REGION Network 22: J_Button_1
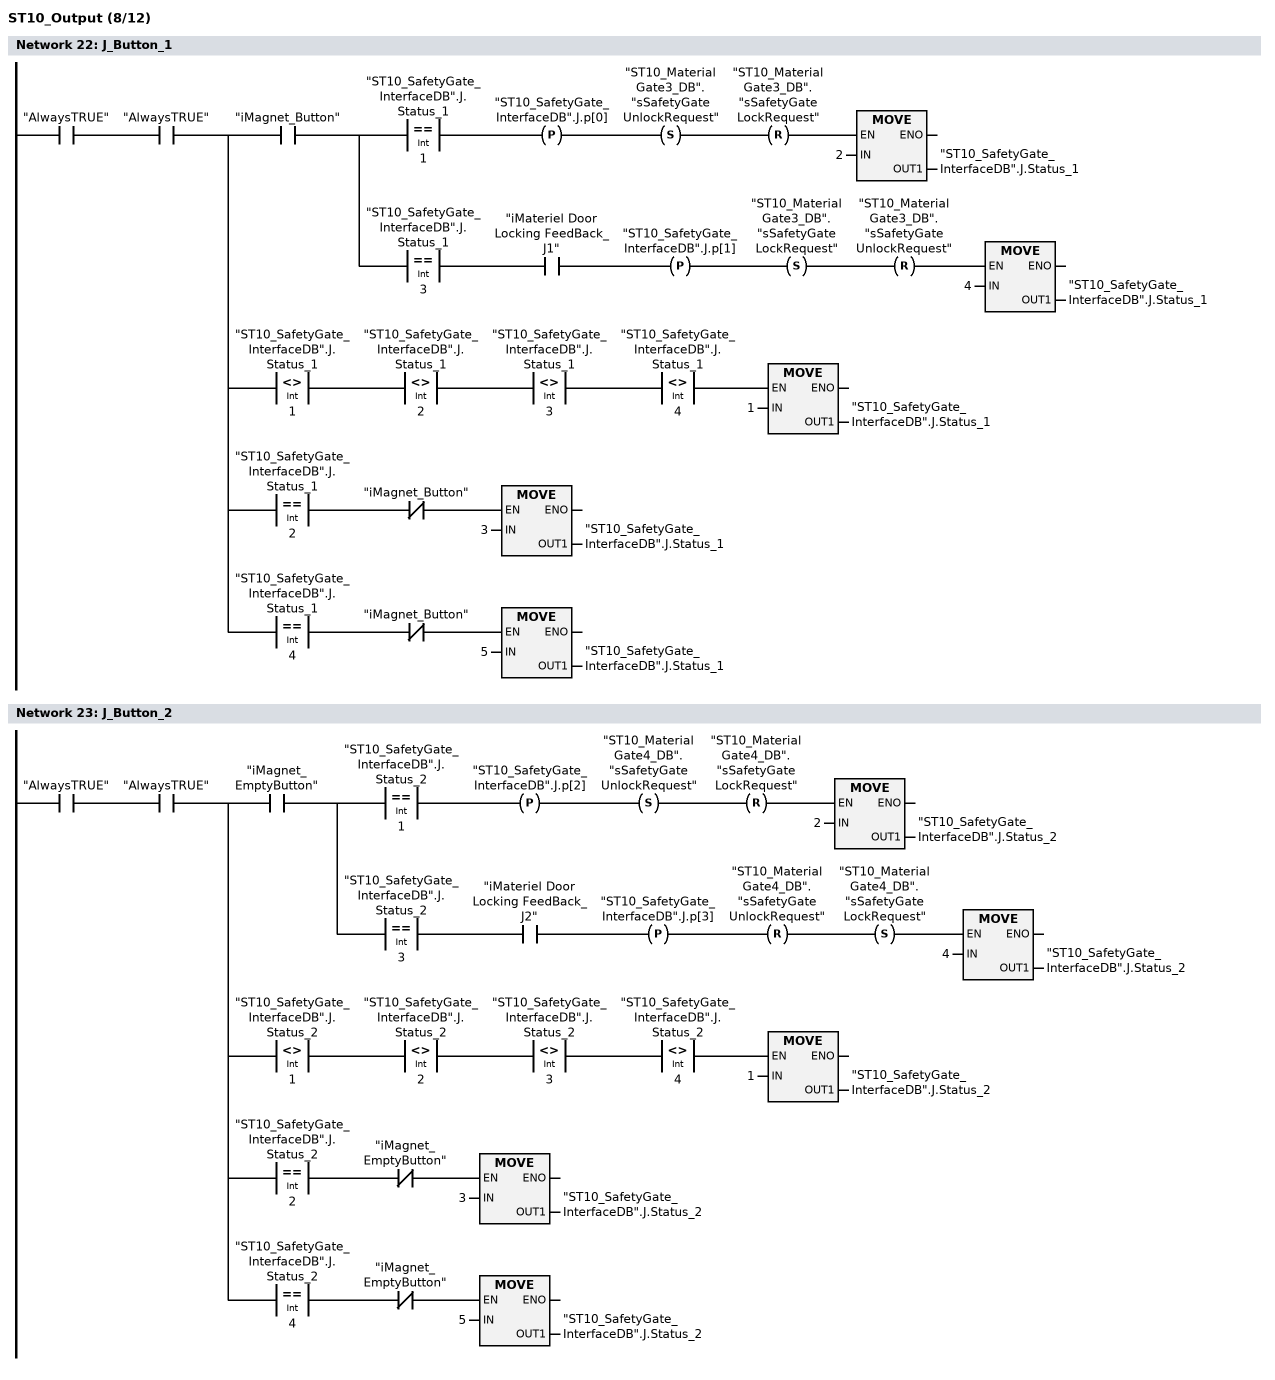
   RUNG wire#powerrail
      Contact( "AlwaysTRUE" )
      Contact( "AlwaysTRUE" )
      wire#w1
      Contact( "iMagnet_Button" )
      wire#w2
      { S7_Templates := "SrcType := Int" } EQ_Contact(in1 := "ST10_SafetyGate_InterfaceDB".J.Status_1, in2 := 1)
      P_Trig( "ST10_SafetyGate_InterfaceDB".J.p[0] )
      S_Coil( "ST10_MaterialGate3_DB"."sSafetyGate UnlockRequest" )
      R_Coil( "ST10_MaterialGate3_DB"."sSafetyGate LockRequest" )
      Move(in := 2, out1 => "ST10_SafetyGate_InterfaceDB".J.Status_1)
   END_RUNG
   RUNG wire#w2
      { S7_Templates := "SrcType := Int" } EQ_Contact(in1 := "ST10_SafetyGate_InterfaceDB".J.Status_1, in2 := 3)
      Contact( "iMateriel Door Locking FeedBack_J1" )
      P_Trig( "ST10_SafetyGate_InterfaceDB".J.p[1] )
      S_Coil( "ST10_MaterialGate3_DB"."sSafetyGate LockRequest" )
      R_Coil( "ST10_MaterialGate3_DB"."sSafetyGate UnlockRequest" )
      Move(in := 4, out1 => "ST10_SafetyGate_InterfaceDB".J.Status_1)
   END_RUNG
   RUNG wire#w1
      { S7_Templates := "SrcType := Int" } NE_Contact(in1 := "ST10_SafetyGate_InterfaceDB".J.Status_1, in2 := 1)
      { S7_Templates := "SrcType := Int" } NE_Contact(in1 := "ST10_SafetyGate_InterfaceDB".J.Status_1, in2 := 2)
      { S7_Templates := "SrcType := Int" } NE_Contact(in1 := "ST10_SafetyGate_InterfaceDB".J.Status_1, in2 := 3)
      { S7_Templates := "SrcType := Int" } NE_Contact(in1 := "ST10_SafetyGate_InterfaceDB".J.Status_1, in2 := 4)
      Move(in := 1, out1 => "ST10_SafetyGate_InterfaceDB".J.Status_1)
   END_RUNG
   RUNG wire#w1
      { S7_Templates := "SrcType := Int" } EQ_Contact(in1 := "ST10_SafetyGate_InterfaceDB".J.Status_1, in2 := 2)
      I_Contact( "iMagnet_Button" )
      Move(in := 3, out1 => "ST10_SafetyGate_InterfaceDB".J.Status_1)
   END_RUNG
   RUNG wire#w1
      { S7_Templates := "SrcType := Int" } EQ_Contact(in1 := "ST10_SafetyGate_InterfaceDB".J.Status_1, in2 := 4)
      I_Contact( "iMagnet_Button" )
      Move(in := 5, out1 => "ST10_SafetyGate_InterfaceDB".J.Status_1)
   END_RUNG
   // the same network as SCL:
   #_w1 := "AlwaysTRUE" AND "AlwaysTRUE";
   #_w2 := #_w1 AND "iMagnet_Button";
   #_w3 := #_w2 AND ("ST10_SafetyGate_InterfaceDB".J.Status_1 = 1);
   #_w4 := #_w3 AND NOT "ST10_SafetyGate_InterfaceDB".J.p[0];   // rising edge
   "ST10_SafetyGate_InterfaceDB".J.p[0] := #_w3;
   IF #_w4 THEN
       "ST10_MaterialGate3_DB"."sSafetyGate UnlockRequest" := TRUE;
       "ST10_MaterialGate3_DB"."sSafetyGate LockRequest" := FALSE;
       "ST10_SafetyGate_InterfaceDB".J.Status_1 := 2;
   END_IF;
   #_w5 := #_w2 AND ("ST10_SafetyGate_InterfaceDB".J.Status_1 = 3) AND "iMateriel Door Locking FeedBack_J1";
   #_w6 := #_w5 AND NOT "ST10_SafetyGate_InterfaceDB".J.p[1];   // rising edge
   "ST10_SafetyGate_InterfaceDB".J.p[1] := #_w5;
   IF #_w6 THEN
       "ST10_MaterialGate3_DB"."sSafetyGate LockRequest" := TRUE;
       "ST10_MaterialGate3_DB"."sSafetyGate UnlockRequest" := FALSE;
       "ST10_SafetyGate_InterfaceDB".J.Status_1 := 4;
   END_IF;
   IF #_w1 AND ("ST10_SafetyGate_InterfaceDB".J.Status_1 <> 1) AND ("ST10_SafetyGate_InterfaceDB".J.Status_1 <> 2) AND ("ST10_SafetyGate_InterfaceDB".J.Status_1 <> 3) AND ("ST10_SafetyGate_InterfaceDB".J.Status_1 <> 4) THEN
       "ST10_SafetyGate_InterfaceDB".J.Status_1 := 1;
   END_IF;
   IF #_w1 AND ("ST10_SafetyGate_InterfaceDB".J.Status_1 = 2) AND NOT "iMagnet_Button" THEN
       "ST10_SafetyGate_InterfaceDB".J.Status_1 := 3;
   END_IF;
   IF #_w1 AND ("ST10_SafetyGate_InterfaceDB".J.Status_1 = 4) AND NOT "iMagnet_Button" THEN
       "ST10_SafetyGate_InterfaceDB".J.Status_1 := 5;
   END_IF;
END_REGION

REGION Network 23: J_Button_2
   RUNG wire#powerrail
      Contact( "AlwaysTRUE" )
      Contact( "AlwaysTRUE" )
      wire#w1
      Contact( "iMagnet_EmptyButton" )
      wire#w2
      { S7_Templates := "SrcType := Int" } EQ_Contact(in1 := "ST10_SafetyGate_InterfaceDB".J.Status_2, in2 := 1)
      P_Trig( "ST10_SafetyGate_InterfaceDB".J.p[2] )
      S_Coil( "ST10_MaterialGate4_DB"."sSafetyGate UnlockRequest" )
      R_Coil( "ST10_MaterialGate4_DB"."sSafetyGate LockRequest" )
      Move(in := 2, out1 => "ST10_SafetyGate_InterfaceDB".J.Status_2)
   END_RUNG
   RUNG wire#w2
      { S7_Templates := "SrcType := Int" } EQ_Contact(in1 := "ST10_SafetyGate_InterfaceDB".J.Status_2, in2 := 3)
      Contact( "iMateriel Door Locking FeedBack_J2" )
      P_Trig( "ST10_SafetyGate_InterfaceDB".J.p[3] )
      R_Coil( "ST10_MaterialGate4_DB"."sSafetyGate UnlockRequest" )
      S_Coil( "ST10_MaterialGate4_DB"."sSafetyGate LockRequest" )
      Move(in := 4, out1 => "ST10_SafetyGate_InterfaceDB".J.Status_2)
   END_RUNG
   RUNG wire#w1
      { S7_Templates := "SrcType := Int" } NE_Contact(in1 := "ST10_SafetyGate_InterfaceDB".J.Status_2, in2 := 1)
      { S7_Templates := "SrcType := Int" } NE_Contact(in1 := "ST10_SafetyGate_InterfaceDB".J.Status_2, in2 := 2)
      { S7_Templates := "SrcType := Int" } NE_Contact(in1 := "ST10_SafetyGate_InterfaceDB".J.Status_2, in2 := 3)
      { S7_Templates := "SrcType := Int" } NE_Contact(in1 := "ST10_SafetyGate_InterfaceDB".J.Status_2, in2 := 4)
      Move(in := 1, out1 => "ST10_SafetyGate_InterfaceDB".J.Status_2)
   END_RUNG
   RUNG wire#w1
      { S7_Templates := "SrcType := Int" } EQ_Contact(in1 := "ST10_SafetyGate_InterfaceDB".J.Status_2, in2 := 2)
      I_Contact( "iMagnet_EmptyButton" )
      Move(in := 3, out1 => "ST10_SafetyGate_InterfaceDB".J.Status_2)
   END_RUNG
   RUNG wire#w1
      { S7_Templates := "SrcType := Int" } EQ_Contact(in1 := "ST10_SafetyGate_InterfaceDB".J.Status_2, in2 := 4)
      I_Contact( "iMagnet_EmptyButton" )
      Move(in := 5, out1 => "ST10_SafetyGate_InterfaceDB".J.Status_2)
   END_RUNG
   // the same network as SCL:
   #_w1 := "AlwaysTRUE" AND "AlwaysTRUE";
   #_w2 := #_w1 AND "iMagnet_EmptyButton";
   #_w3 := #_w2 AND ("ST10_SafetyGate_InterfaceDB".J.Status_2 = 1);
   #_w4 := #_w3 AND NOT "ST10_SafetyGate_InterfaceDB".J.p[2];   // rising edge
   "ST10_SafetyGate_InterfaceDB".J.p[2] := #_w3;
   IF #_w4 THEN
       "ST10_MaterialGate4_DB"."sSafetyGate UnlockRequest" := TRUE;
       "ST10_MaterialGate4_DB"."sSafetyGate LockRequest" := FALSE;
       "ST10_SafetyGate_InterfaceDB".J.Status_2 := 2;
   END_IF;
   #_w5 := #_w2 AND ("ST10_SafetyGate_InterfaceDB".J.Status_2 = 3) AND "iMateriel Door Locking FeedBack_J2";
   #_w6 := #_w5 AND NOT "ST10_SafetyGate_InterfaceDB".J.p[3];   // rising edge
   "ST10_SafetyGate_InterfaceDB".J.p[3] := #_w5;
   IF #_w6 THEN
       "ST10_MaterialGate4_DB"."sSafetyGate UnlockRequest" := FALSE;
       "ST10_MaterialGate4_DB"."sSafetyGate LockRequest" := TRUE;
       "ST10_SafetyGate_InterfaceDB".J.Status_2 := 4;
   END_IF;
   IF #_w1 AND ("ST10_SafetyGate_InterfaceDB".J.Status_2 <> 1) AND ("ST10_SafetyGate_InterfaceDB".J.Status_2 <> 2) AND ("ST10_SafetyGate_InterfaceDB".J.Status_2 <> 3) AND ("ST10_SafetyGate_InterfaceDB".J.Status_2 <> 4) THEN
       "ST10_SafetyGate_InterfaceDB".J.Status_2 := 1;
   END_IF;
   IF #_w1 AND ("ST10_SafetyGate_InterfaceDB".J.Status_2 = 2) AND NOT "iMagnet_EmptyButton" THEN
       "ST10_SafetyGate_InterfaceDB".J.Status_2 := 3;
   END_IF;
   IF #_w1 AND ("ST10_SafetyGate_InterfaceDB".J.Status_2 = 4) AND NOT "iMagnet_EmptyButton" THEN
       "ST10_SafetyGate_InterfaceDB".J.Status_2 := 5;
   END_IF;
END_REGION

REGION Network 24: J_Button_3 DOOR7
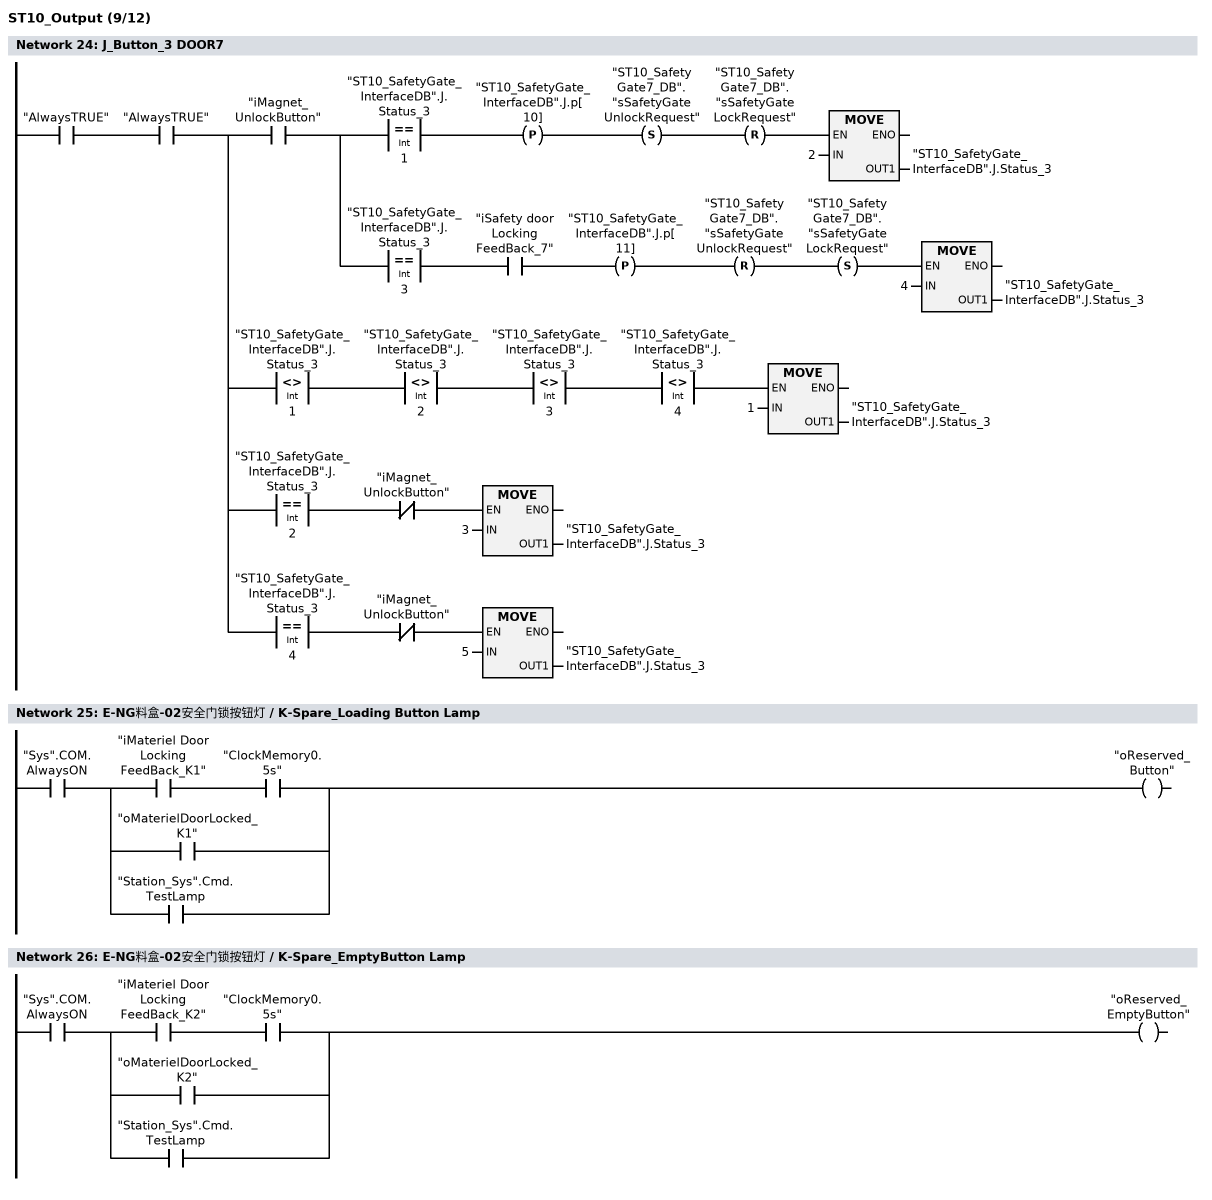
   RUNG wire#powerrail
      Contact( "AlwaysTRUE" )
      Contact( "AlwaysTRUE" )
      wire#w1
      Contact( "iMagnet_UnlockButton" )
      wire#w2
      { S7_Templates := "SrcType := Int" } EQ_Contact(in1 := "ST10_SafetyGate_InterfaceDB".J.Status_3, in2 := 1)
      P_Trig( "ST10_SafetyGate_InterfaceDB".J.p[10] )
      S_Coil( "ST10_SafetyGate7_DB"."sSafetyGate UnlockRequest" )
      R_Coil( "ST10_SafetyGate7_DB"."sSafetyGate LockRequest" )
      Move(in := 2, out1 => "ST10_SafetyGate_InterfaceDB".J.Status_3)
   END_RUNG
   RUNG wire#w2
      { S7_Templates := "SrcType := Int" } EQ_Contact(in1 := "ST10_SafetyGate_InterfaceDB".J.Status_3, in2 := 3)
      Contact( "iSafety door Locking FeedBack_7" )
      P_Trig( "ST10_SafetyGate_InterfaceDB".J.p[11] )
      R_Coil( "ST10_SafetyGate7_DB"."sSafetyGate UnlockRequest" )
      S_Coil( "ST10_SafetyGate7_DB"."sSafetyGate LockRequest" )
      Move(in := 4, out1 => "ST10_SafetyGate_InterfaceDB".J.Status_3)
   END_RUNG
   RUNG wire#w1
      { S7_Templates := "SrcType := Int" } NE_Contact(in1 := "ST10_SafetyGate_InterfaceDB".J.Status_3, in2 := 1)
      { S7_Templates := "SrcType := Int" } NE_Contact(in1 := "ST10_SafetyGate_InterfaceDB".J.Status_3, in2 := 2)
      { S7_Templates := "SrcType := Int" } NE_Contact(in1 := "ST10_SafetyGate_InterfaceDB".J.Status_3, in2 := 3)
      { S7_Templates := "SrcType := Int" } NE_Contact(in1 := "ST10_SafetyGate_InterfaceDB".J.Status_3, in2 := 4)
      Move(in := 1, out1 => "ST10_SafetyGate_InterfaceDB".J.Status_3)
   END_RUNG
   RUNG wire#w1
      { S7_Templates := "SrcType := Int" } EQ_Contact(in1 := "ST10_SafetyGate_InterfaceDB".J.Status_3, in2 := 2)
      I_Contact( "iMagnet_UnlockButton" )
      Move(in := 3, out1 => "ST10_SafetyGate_InterfaceDB".J.Status_3)
   END_RUNG
   RUNG wire#w1
      { S7_Templates := "SrcType := Int" } EQ_Contact(in1 := "ST10_SafetyGate_InterfaceDB".J.Status_3, in2 := 4)
      I_Contact( "iMagnet_UnlockButton" )
      Move(in := 5, out1 => "ST10_SafetyGate_InterfaceDB".J.Status_3)
   END_RUNG
   // the same network as SCL:
   #_w1 := "AlwaysTRUE" AND "AlwaysTRUE";
   #_w2 := #_w1 AND "iMagnet_UnlockButton";
   #_w3 := #_w2 AND ("ST10_SafetyGate_InterfaceDB".J.Status_3 = 1);
   #_w4 := #_w3 AND NOT "ST10_SafetyGate_InterfaceDB".J.p[10];   // rising edge
   "ST10_SafetyGate_InterfaceDB".J.p[10] := #_w3;
   IF #_w4 THEN
       "ST10_SafetyGate7_DB"."sSafetyGate UnlockRequest" := TRUE;
       "ST10_SafetyGate7_DB"."sSafetyGate LockRequest" := FALSE;
       "ST10_SafetyGate_InterfaceDB".J.Status_3 := 2;
   END_IF;
   #_w5 := #_w2 AND ("ST10_SafetyGate_InterfaceDB".J.Status_3 = 3) AND "iSafety door Locking FeedBack_7";
   #_w6 := #_w5 AND NOT "ST10_SafetyGate_InterfaceDB".J.p[11];   // rising edge
   "ST10_SafetyGate_InterfaceDB".J.p[11] := #_w5;
   IF #_w6 THEN
       "ST10_SafetyGate7_DB"."sSafetyGate UnlockRequest" := FALSE;
       "ST10_SafetyGate7_DB"."sSafetyGate LockRequest" := TRUE;
       "ST10_SafetyGate_InterfaceDB".J.Status_3 := 4;
   END_IF;
   IF #_w1 AND ("ST10_SafetyGate_InterfaceDB".J.Status_3 <> 1) AND ("ST10_SafetyGate_InterfaceDB".J.Status_3 <> 2) AND ("ST10_SafetyGate_InterfaceDB".J.Status_3 <> 3) AND ("ST10_SafetyGate_InterfaceDB".J.Status_3 <> 4) THEN
       "ST10_SafetyGate_InterfaceDB".J.Status_3 := 1;
   END_IF;
   IF #_w1 AND ("ST10_SafetyGate_InterfaceDB".J.Status_3 = 2) AND NOT "iMagnet_UnlockButton" THEN
       "ST10_SafetyGate_InterfaceDB".J.Status_3 := 3;
   END_IF;
   IF #_w1 AND ("ST10_SafetyGate_InterfaceDB".J.Status_3 = 4) AND NOT "iMagnet_UnlockButton" THEN
       "ST10_SafetyGate_InterfaceDB".J.Status_3 := 5;
   END_IF;
END_REGION

REGION Network 25: E-NG料盒-02安全门锁按钮灯 / K-Spare_Loading Button Lamp
   RUNG wire#powerrail
      Contact( "Sys".COM.AlwaysON )
      wire#w1
      Contact( "iMateriel Door Locking FeedBack_K1" )
      Contact( "ClockMemory0.5s" )
      wire#w2
      Coil( "oReserved_Button" )
   END_RUNG
   RUNG wire#w1
      Contact( "oMaterielDoorLocked_K1" )
   END_RUNG wire#w2
   RUNG wire#w1
      Contact( "Station_Sys".Cmd.TestLamp )
   END_RUNG wire#w2
   // the same network as SCL:
   "oReserved_Button" := "Sys".COM.AlwaysON AND (("iMateriel Door Locking FeedBack_K1" AND "ClockMemory0.5s") OR "oMaterielDoorLocked_K1" OR "Station_Sys".Cmd.TestLamp);
END_REGION

REGION Network 26: E-NG料盒-02安全门锁按钮灯 / K-Spare_EmptyButton Lamp
   RUNG wire#powerrail
      Contact( "Sys".COM.AlwaysON )
      wire#w1
      Contact( "iMateriel Door Locking FeedBack_K2" )
      Contact( "ClockMemory0.5s" )
      wire#w2
      Coil( "oReserved_EmptyButton" )
   END_RUNG
   RUNG wire#w1
      Contact( "oMaterielDoorLocked_K2" )
   END_RUNG wire#w2
   RUNG wire#w1
      Contact( "Station_Sys".Cmd.TestLamp )
   END_RUNG wire#w2
   // the same network as SCL:
   "oReserved_EmptyButton" := "Sys".COM.AlwaysON AND (("iMateriel Door Locking FeedBack_K2" AND "ClockMemory0.5s") OR "oMaterielDoorLocked_K2" OR "Station_Sys".Cmd.TestLamp);
END_REGION

REGION Network 27: E-NG料盒-02安全门锁按钮灯 / K_Loading DoorButton Lamp 8
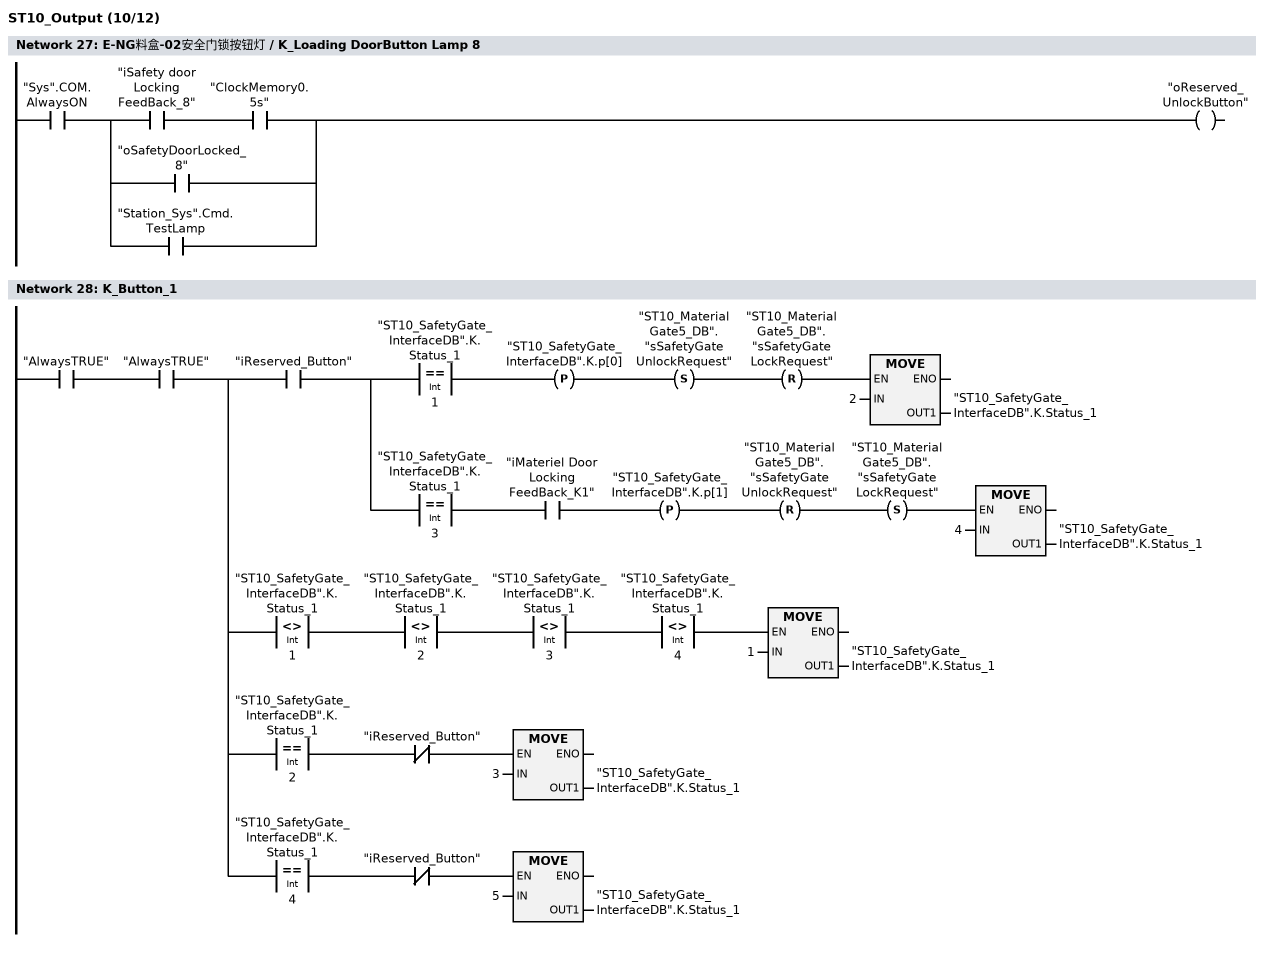
   RUNG wire#powerrail
      Contact( "Sys".COM.AlwaysON )
      wire#w1
      Contact( "iSafety door Locking FeedBack_8" )
      Contact( "ClockMemory0.5s" )
      wire#w2
      Coil( "oReserved_UnlockButton" )
   END_RUNG
   RUNG wire#w1
      Contact( "oSafetyDoorLocked_8" )
   END_RUNG wire#w2
   RUNG wire#w1
      Contact( "Station_Sys".Cmd.TestLamp )
   END_RUNG wire#w2
   // the same network as SCL:
   "oReserved_UnlockButton" := "Sys".COM.AlwaysON AND (("iSafety door Locking FeedBack_8" AND "ClockMemory0.5s") OR "oSafetyDoorLocked_8" OR "Station_Sys".Cmd.TestLamp);
END_REGION

REGION Network 28: K_Button_1
   RUNG wire#powerrail
      Contact( "AlwaysTRUE" )
      Contact( "AlwaysTRUE" )
      wire#w1
      Contact( "iReserved_Button" )
      wire#w2
      { S7_Templates := "SrcType := Int" } EQ_Contact(in1 := "ST10_SafetyGate_InterfaceDB".K.Status_1, in2 := 1)
      P_Trig( "ST10_SafetyGate_InterfaceDB".K.p[0] )
      S_Coil( "ST10_MaterialGate5_DB"."sSafetyGate UnlockRequest" )
      R_Coil( "ST10_MaterialGate5_DB"."sSafetyGate LockRequest" )
      Move(in := 2, out1 => "ST10_SafetyGate_InterfaceDB".K.Status_1)
   END_RUNG
   RUNG wire#w2
      { S7_Templates := "SrcType := Int" } EQ_Contact(in1 := "ST10_SafetyGate_InterfaceDB".K.Status_1, in2 := 3)
      Contact( "iMateriel Door Locking FeedBack_K1" )
      P_Trig( "ST10_SafetyGate_InterfaceDB".K.p[1] )
      R_Coil( "ST10_MaterialGate5_DB"."sSafetyGate UnlockRequest" )
      S_Coil( "ST10_MaterialGate5_DB"."sSafetyGate LockRequest" )
      Move(in := 4, out1 => "ST10_SafetyGate_InterfaceDB".K.Status_1)
   END_RUNG
   RUNG wire#w1
      { S7_Templates := "SrcType := Int" } NE_Contact(in1 := "ST10_SafetyGate_InterfaceDB".K.Status_1, in2 := 1)
      { S7_Templates := "SrcType := Int" } NE_Contact(in1 := "ST10_SafetyGate_InterfaceDB".K.Status_1, in2 := 2)
      { S7_Templates := "SrcType := Int" } NE_Contact(in1 := "ST10_SafetyGate_InterfaceDB".K.Status_1, in2 := 3)
      { S7_Templates := "SrcType := Int" } NE_Contact(in1 := "ST10_SafetyGate_InterfaceDB".K.Status_1, in2 := 4)
      Move(in := 1, out1 => "ST10_SafetyGate_InterfaceDB".K.Status_1)
   END_RUNG
   RUNG wire#w1
      { S7_Templates := "SrcType := Int" } EQ_Contact(in1 := "ST10_SafetyGate_InterfaceDB".K.Status_1, in2 := 2)
      I_Contact( "iReserved_Button" )
      Move(in := 3, out1 => "ST10_SafetyGate_InterfaceDB".K.Status_1)
   END_RUNG
   RUNG wire#w1
      { S7_Templates := "SrcType := Int" } EQ_Contact(in1 := "ST10_SafetyGate_InterfaceDB".K.Status_1, in2 := 4)
      I_Contact( "iReserved_Button" )
      Move(in := 5, out1 => "ST10_SafetyGate_InterfaceDB".K.Status_1)
   END_RUNG
   // the same network as SCL:
   #_w1 := "AlwaysTRUE" AND "AlwaysTRUE";
   #_w2 := #_w1 AND "iReserved_Button";
   #_w3 := #_w2 AND ("ST10_SafetyGate_InterfaceDB".K.Status_1 = 1);
   #_w4 := #_w3 AND NOT "ST10_SafetyGate_InterfaceDB".K.p[0];   // rising edge
   "ST10_SafetyGate_InterfaceDB".K.p[0] := #_w3;
   IF #_w4 THEN
       "ST10_MaterialGate5_DB"."sSafetyGate UnlockRequest" := TRUE;
       "ST10_MaterialGate5_DB"."sSafetyGate LockRequest" := FALSE;
       "ST10_SafetyGate_InterfaceDB".K.Status_1 := 2;
   END_IF;
   #_w5 := #_w2 AND ("ST10_SafetyGate_InterfaceDB".K.Status_1 = 3) AND "iMateriel Door Locking FeedBack_K1";
   #_w6 := #_w5 AND NOT "ST10_SafetyGate_InterfaceDB".K.p[1];   // rising edge
   "ST10_SafetyGate_InterfaceDB".K.p[1] := #_w5;
   IF #_w6 THEN
       "ST10_MaterialGate5_DB"."sSafetyGate UnlockRequest" := FALSE;
       "ST10_MaterialGate5_DB"."sSafetyGate LockRequest" := TRUE;
       "ST10_SafetyGate_InterfaceDB".K.Status_1 := 4;
   END_IF;
   IF #_w1 AND ("ST10_SafetyGate_InterfaceDB".K.Status_1 <> 1) AND ("ST10_SafetyGate_InterfaceDB".K.Status_1 <> 2) AND ("ST10_SafetyGate_InterfaceDB".K.Status_1 <> 3) AND ("ST10_SafetyGate_InterfaceDB".K.Status_1 <> 4) THEN
       "ST10_SafetyGate_InterfaceDB".K.Status_1 := 1;
   END_IF;
   IF #_w1 AND ("ST10_SafetyGate_InterfaceDB".K.Status_1 = 2) AND NOT "iReserved_Button" THEN
       "ST10_SafetyGate_InterfaceDB".K.Status_1 := 3;
   END_IF;
   IF #_w1 AND ("ST10_SafetyGate_InterfaceDB".K.Status_1 = 4) AND NOT "iReserved_Button" THEN
       "ST10_SafetyGate_InterfaceDB".K.Status_1 := 5;
   END_IF;
END_REGION

REGION Network 29: K_Button_2
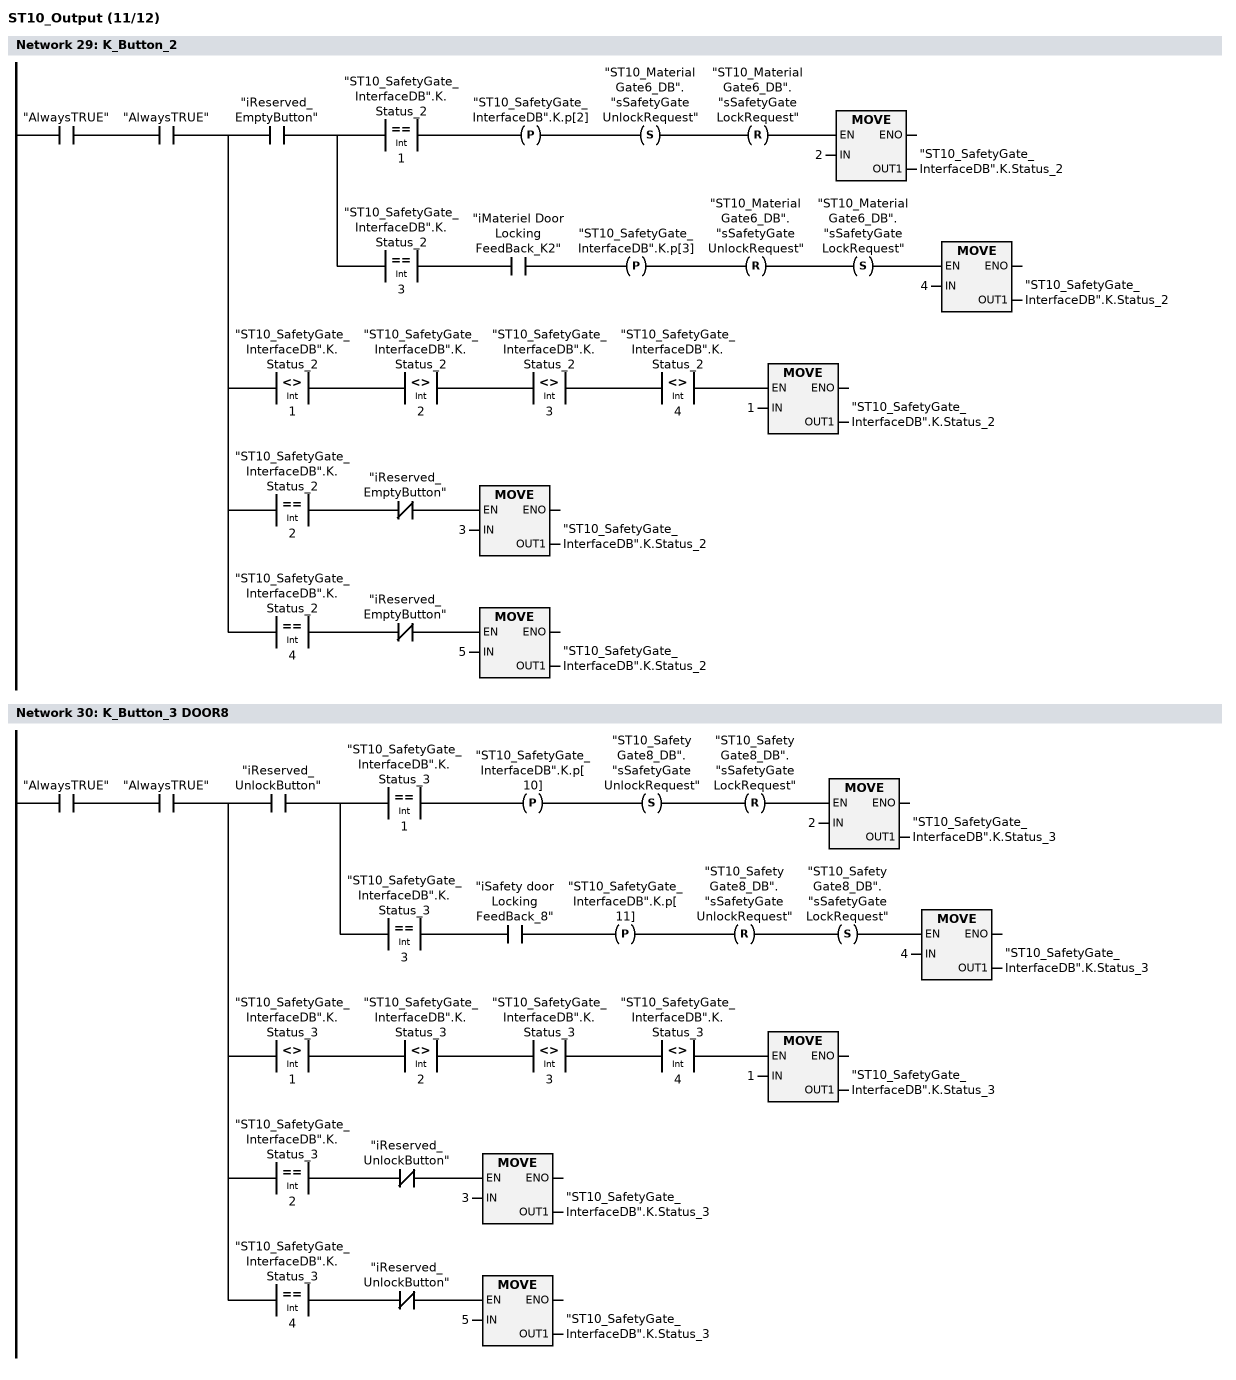
   RUNG wire#powerrail
      Contact( "AlwaysTRUE" )
      Contact( "AlwaysTRUE" )
      wire#w1
      Contact( "iReserved_EmptyButton" )
      wire#w2
      { S7_Templates := "SrcType := Int" } EQ_Contact(in1 := "ST10_SafetyGate_InterfaceDB".K.Status_2, in2 := 1)
      P_Trig( "ST10_SafetyGate_InterfaceDB".K.p[2] )
      S_Coil( "ST10_MaterialGate6_DB"."sSafetyGate UnlockRequest" )
      R_Coil( "ST10_MaterialGate6_DB"."sSafetyGate LockRequest" )
      Move(in := 2, out1 => "ST10_SafetyGate_InterfaceDB".K.Status_2)
   END_RUNG
   RUNG wire#w2
      { S7_Templates := "SrcType := Int" } EQ_Contact(in1 := "ST10_SafetyGate_InterfaceDB".K.Status_2, in2 := 3)
      Contact( "iMateriel Door Locking FeedBack_K2" )
      P_Trig( "ST10_SafetyGate_InterfaceDB".K.p[3] )
      R_Coil( "ST10_MaterialGate6_DB"."sSafetyGate UnlockRequest" )
      S_Coil( "ST10_MaterialGate6_DB"."sSafetyGate LockRequest" )
      Move(in := 4, out1 => "ST10_SafetyGate_InterfaceDB".K.Status_2)
   END_RUNG
   RUNG wire#w1
      { S7_Templates := "SrcType := Int" } NE_Contact(in1 := "ST10_SafetyGate_InterfaceDB".K.Status_2, in2 := 1)
      { S7_Templates := "SrcType := Int" } NE_Contact(in1 := "ST10_SafetyGate_InterfaceDB".K.Status_2, in2 := 2)
      { S7_Templates := "SrcType := Int" } NE_Contact(in1 := "ST10_SafetyGate_InterfaceDB".K.Status_2, in2 := 3)
      { S7_Templates := "SrcType := Int" } NE_Contact(in1 := "ST10_SafetyGate_InterfaceDB".K.Status_2, in2 := 4)
      Move(in := 1, out1 => "ST10_SafetyGate_InterfaceDB".K.Status_2)
   END_RUNG
   RUNG wire#w1
      { S7_Templates := "SrcType := Int" } EQ_Contact(in1 := "ST10_SafetyGate_InterfaceDB".K.Status_2, in2 := 2)
      I_Contact( "iReserved_EmptyButton" )
      Move(in := 3, out1 => "ST10_SafetyGate_InterfaceDB".K.Status_2)
   END_RUNG
   RUNG wire#w1
      { S7_Templates := "SrcType := Int" } EQ_Contact(in1 := "ST10_SafetyGate_InterfaceDB".K.Status_2, in2 := 4)
      I_Contact( "iReserved_EmptyButton" )
      Move(in := 5, out1 => "ST10_SafetyGate_InterfaceDB".K.Status_2)
   END_RUNG
   // the same network as SCL:
   #_w1 := "AlwaysTRUE" AND "AlwaysTRUE";
   #_w2 := #_w1 AND "iReserved_EmptyButton";
   #_w3 := #_w2 AND ("ST10_SafetyGate_InterfaceDB".K.Status_2 = 1);
   #_w4 := #_w3 AND NOT "ST10_SafetyGate_InterfaceDB".K.p[2];   // rising edge
   "ST10_SafetyGate_InterfaceDB".K.p[2] := #_w3;
   IF #_w4 THEN
       "ST10_MaterialGate6_DB"."sSafetyGate UnlockRequest" := TRUE;
       "ST10_MaterialGate6_DB"."sSafetyGate LockRequest" := FALSE;
       "ST10_SafetyGate_InterfaceDB".K.Status_2 := 2;
   END_IF;
   #_w5 := #_w2 AND ("ST10_SafetyGate_InterfaceDB".K.Status_2 = 3) AND "iMateriel Door Locking FeedBack_K2";
   #_w6 := #_w5 AND NOT "ST10_SafetyGate_InterfaceDB".K.p[3];   // rising edge
   "ST10_SafetyGate_InterfaceDB".K.p[3] := #_w5;
   IF #_w6 THEN
       "ST10_MaterialGate6_DB"."sSafetyGate UnlockRequest" := FALSE;
       "ST10_MaterialGate6_DB"."sSafetyGate LockRequest" := TRUE;
       "ST10_SafetyGate_InterfaceDB".K.Status_2 := 4;
   END_IF;
   IF #_w1 AND ("ST10_SafetyGate_InterfaceDB".K.Status_2 <> 1) AND ("ST10_SafetyGate_InterfaceDB".K.Status_2 <> 2) AND ("ST10_SafetyGate_InterfaceDB".K.Status_2 <> 3) AND ("ST10_SafetyGate_InterfaceDB".K.Status_2 <> 4) THEN
       "ST10_SafetyGate_InterfaceDB".K.Status_2 := 1;
   END_IF;
   IF #_w1 AND ("ST10_SafetyGate_InterfaceDB".K.Status_2 = 2) AND NOT "iReserved_EmptyButton" THEN
       "ST10_SafetyGate_InterfaceDB".K.Status_2 := 3;
   END_IF;
   IF #_w1 AND ("ST10_SafetyGate_InterfaceDB".K.Status_2 = 4) AND NOT "iReserved_EmptyButton" THEN
       "ST10_SafetyGate_InterfaceDB".K.Status_2 := 5;
   END_IF;
END_REGION

REGION Network 30: K_Button_3 DOOR8
   RUNG wire#powerrail
      Contact( "AlwaysTRUE" )
      Contact( "AlwaysTRUE" )
      wire#w1
      Contact( "iReserved_UnlockButton" )
      wire#w2
      { S7_Templates := "SrcType := Int" } EQ_Contact(in1 := "ST10_SafetyGate_InterfaceDB".K.Status_3, in2 := 1)
      P_Trig( "ST10_SafetyGate_InterfaceDB".K.p[10] )
      S_Coil( "ST10_SafetyGate8_DB"."sSafetyGate UnlockRequest" )
      R_Coil( "ST10_SafetyGate8_DB"."sSafetyGate LockRequest" )
      Move(in := 2, out1 => "ST10_SafetyGate_InterfaceDB".K.Status_3)
   END_RUNG
   RUNG wire#w2
      { S7_Templates := "SrcType := Int" } EQ_Contact(in1 := "ST10_SafetyGate_InterfaceDB".K.Status_3, in2 := 3)
      Contact( "iSafety door Locking FeedBack_8" )
      P_Trig( "ST10_SafetyGate_InterfaceDB".K.p[11] )
      R_Coil( "ST10_SafetyGate8_DB"."sSafetyGate UnlockRequest" )
      S_Coil( "ST10_SafetyGate8_DB"."sSafetyGate LockRequest" )
      Move(in := 4, out1 => "ST10_SafetyGate_InterfaceDB".K.Status_3)
   END_RUNG
   RUNG wire#w1
      { S7_Templates := "SrcType := Int" } NE_Contact(in1 := "ST10_SafetyGate_InterfaceDB".K.Status_3, in2 := 1)
      { S7_Templates := "SrcType := Int" } NE_Contact(in1 := "ST10_SafetyGate_InterfaceDB".K.Status_3, in2 := 2)
      { S7_Templates := "SrcType := Int" } NE_Contact(in1 := "ST10_SafetyGate_InterfaceDB".K.Status_3, in2 := 3)
      { S7_Templates := "SrcType := Int" } NE_Contact(in1 := "ST10_SafetyGate_InterfaceDB".K.Status_3, in2 := 4)
      Move(in := 1, out1 => "ST10_SafetyGate_InterfaceDB".K.Status_3)
   END_RUNG
   RUNG wire#w1
      { S7_Templates := "SrcType := Int" } EQ_Contact(in1 := "ST10_SafetyGate_InterfaceDB".K.Status_3, in2 := 2)
      I_Contact( "iReserved_UnlockButton" )
      Move(in := 3, out1 => "ST10_SafetyGate_InterfaceDB".K.Status_3)
   END_RUNG
   RUNG wire#w1
      { S7_Templates := "SrcType := Int" } EQ_Contact(in1 := "ST10_SafetyGate_InterfaceDB".K.Status_3, in2 := 4)
      I_Contact( "iReserved_UnlockButton" )
      Move(in := 5, out1 => "ST10_SafetyGate_InterfaceDB".K.Status_3)
   END_RUNG
   // the same network as SCL:
   #_w1 := "AlwaysTRUE" AND "AlwaysTRUE";
   #_w2 := #_w1 AND "iReserved_UnlockButton";
   #_w3 := #_w2 AND ("ST10_SafetyGate_InterfaceDB".K.Status_3 = 1);
   #_w4 := #_w3 AND NOT "ST10_SafetyGate_InterfaceDB".K.p[10];   // rising edge
   "ST10_SafetyGate_InterfaceDB".K.p[10] := #_w3;
   IF #_w4 THEN
       "ST10_SafetyGate8_DB"."sSafetyGate UnlockRequest" := TRUE;
       "ST10_SafetyGate8_DB"."sSafetyGate LockRequest" := FALSE;
       "ST10_SafetyGate_InterfaceDB".K.Status_3 := 2;
   END_IF;
   #_w5 := #_w2 AND ("ST10_SafetyGate_InterfaceDB".K.Status_3 = 3) AND "iSafety door Locking FeedBack_8";
   #_w6 := #_w5 AND NOT "ST10_SafetyGate_InterfaceDB".K.p[11];   // rising edge
   "ST10_SafetyGate_InterfaceDB".K.p[11] := #_w5;
   IF #_w6 THEN
       "ST10_SafetyGate8_DB"."sSafetyGate UnlockRequest" := FALSE;
       "ST10_SafetyGate8_DB"."sSafetyGate LockRequest" := TRUE;
       "ST10_SafetyGate_InterfaceDB".K.Status_3 := 4;
   END_IF;
   IF #_w1 AND ("ST10_SafetyGate_InterfaceDB".K.Status_3 <> 1) AND ("ST10_SafetyGate_InterfaceDB".K.Status_3 <> 2) AND ("ST10_SafetyGate_InterfaceDB".K.Status_3 <> 3) AND ("ST10_SafetyGate_InterfaceDB".K.Status_3 <> 4) THEN
       "ST10_SafetyGate_InterfaceDB".K.Status_3 := 1;
   END_IF;
   IF #_w1 AND ("ST10_SafetyGate_InterfaceDB".K.Status_3 = 2) AND NOT "iReserved_UnlockButton" THEN
       "ST10_SafetyGate_InterfaceDB".K.Status_3 := 3;
   END_IF;
   IF #_w1 AND ("ST10_SafetyGate_InterfaceDB".K.Status_3 = 4) AND NOT "iReserved_UnlockButton" THEN
       "ST10_SafetyGate_InterfaceDB".K.Status_3 := 5;
   END_IF;
END_REGION

REGION Network 31: E-NG料盒-02安全门锁按钮灯 / L-Unloading_LoadingButton Lamp
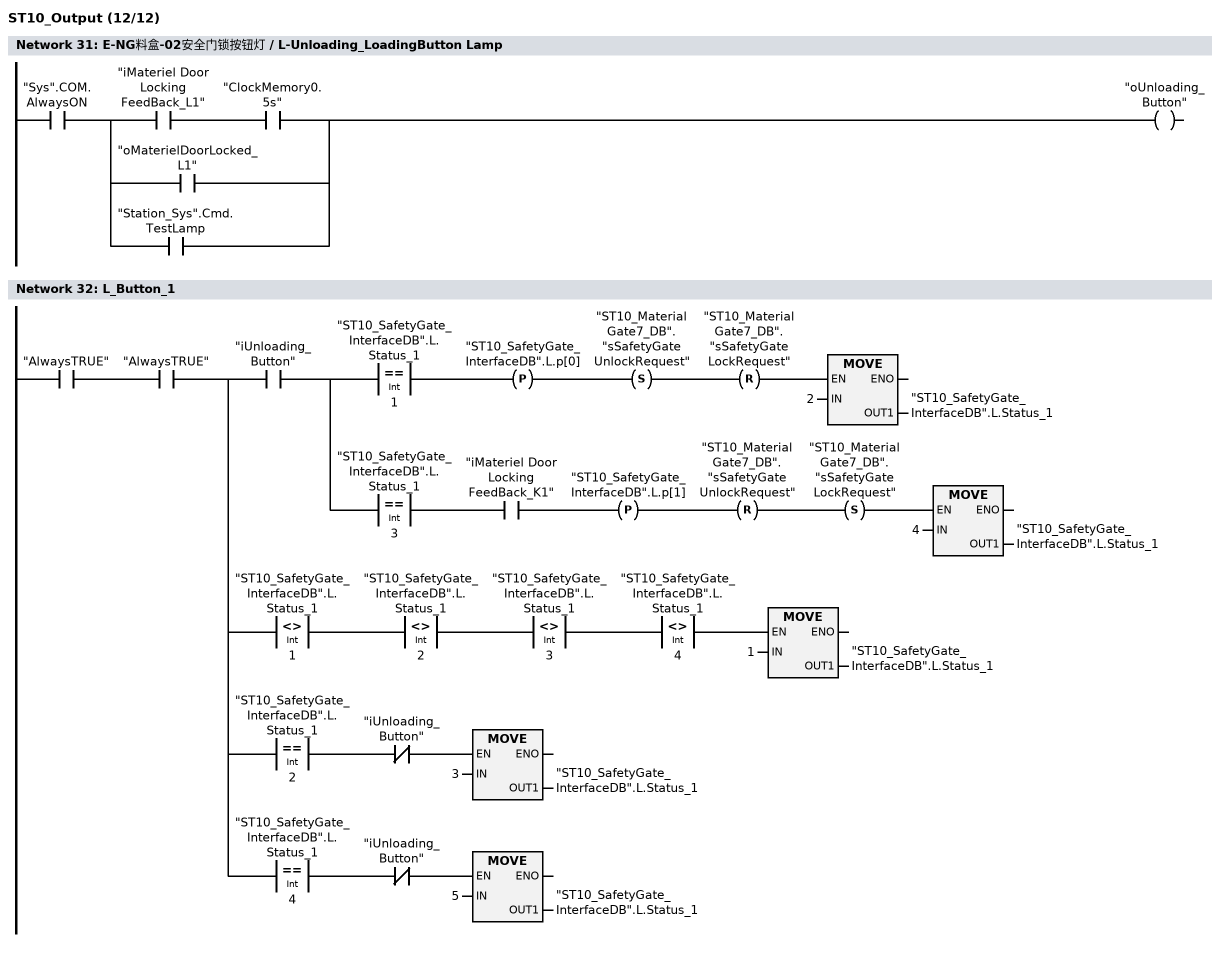
   RUNG wire#powerrail
      Contact( "Sys".COM.AlwaysON )
      wire#w1
      Contact( "iMateriel Door Locking FeedBack_L1" )
      Contact( "ClockMemory0.5s" )
      wire#w2
      Coil( "oUnloading_Button" )
   END_RUNG
   RUNG wire#w1
      Contact( "oMaterielDoorLocked_L1" )
   END_RUNG wire#w2
   RUNG wire#w1
      Contact( "Station_Sys".Cmd.TestLamp )
   END_RUNG wire#w2
   // the same network as SCL:
   "oUnloading_Button" := "Sys".COM.AlwaysON AND (("iMateriel Door Locking FeedBack_L1" AND "ClockMemory0.5s") OR "oMaterielDoorLocked_L1" OR "Station_Sys".Cmd.TestLamp);
END_REGION

REGION Network 32: L_Button_1
   RUNG wire#powerrail
      Contact( "AlwaysTRUE" )
      Contact( "AlwaysTRUE" )
      wire#w1
      Contact( "iUnloading_Button" )
      wire#w2
      { S7_Templates := "SrcType := Int" } EQ_Contact(in1 := "ST10_SafetyGate_InterfaceDB".L.Status_1, in2 := 1)
      P_Trig( "ST10_SafetyGate_InterfaceDB".L.p[0] )
      S_Coil( "ST10_MaterialGate7_DB"."sSafetyGate UnlockRequest" )
      R_Coil( "ST10_MaterialGate7_DB"."sSafetyGate LockRequest" )
      Move(in := 2, out1 => "ST10_SafetyGate_InterfaceDB".L.Status_1)
   END_RUNG
   RUNG wire#w2
      { S7_Templates := "SrcType := Int" } EQ_Contact(in1 := "ST10_SafetyGate_InterfaceDB".L.Status_1, in2 := 3)
      Contact( "iMateriel Door Locking FeedBack_K1" )
      P_Trig( "ST10_SafetyGate_InterfaceDB".L.p[1] )
      R_Coil( "ST10_MaterialGate7_DB"."sSafetyGate UnlockRequest" )
      S_Coil( "ST10_MaterialGate7_DB"."sSafetyGate LockRequest" )
      Move(in := 4, out1 => "ST10_SafetyGate_InterfaceDB".L.Status_1)
   END_RUNG
   RUNG wire#w1
      { S7_Templates := "SrcType := Int" } NE_Contact(in1 := "ST10_SafetyGate_InterfaceDB".L.Status_1, in2 := 1)
      { S7_Templates := "SrcType := Int" } NE_Contact(in1 := "ST10_SafetyGate_InterfaceDB".L.Status_1, in2 := 2)
      { S7_Templates := "SrcType := Int" } NE_Contact(in1 := "ST10_SafetyGate_InterfaceDB".L.Status_1, in2 := 3)
      { S7_Templates := "SrcType := Int" } NE_Contact(in1 := "ST10_SafetyGate_InterfaceDB".L.Status_1, in2 := 4)
      Move(in := 1, out1 => "ST10_SafetyGate_InterfaceDB".L.Status_1)
   END_RUNG
   RUNG wire#w1
      { S7_Templates := "SrcType := Int" } EQ_Contact(in1 := "ST10_SafetyGate_InterfaceDB".L.Status_1, in2 := 2)
      I_Contact( "iUnloading_Button" )
      Move(in := 3, out1 => "ST10_SafetyGate_InterfaceDB".L.Status_1)
   END_RUNG
   RUNG wire#w1
      { S7_Templates := "SrcType := Int" } EQ_Contact(in1 := "ST10_SafetyGate_InterfaceDB".L.Status_1, in2 := 4)
      I_Contact( "iUnloading_Button" )
      Move(in := 5, out1 => "ST10_SafetyGate_InterfaceDB".L.Status_1)
   END_RUNG
   // the same network as SCL:
   #_w1 := "AlwaysTRUE" AND "AlwaysTRUE";
   #_w2 := #_w1 AND "iUnloading_Button";
   #_w3 := #_w2 AND ("ST10_SafetyGate_InterfaceDB".L.Status_1 = 1);
   #_w4 := #_w3 AND NOT "ST10_SafetyGate_InterfaceDB".L.p[0];   // rising edge
   "ST10_SafetyGate_InterfaceDB".L.p[0] := #_w3;
   IF #_w4 THEN
       "ST10_MaterialGate7_DB"."sSafetyGate UnlockRequest" := TRUE;
       "ST10_MaterialGate7_DB"."sSafetyGate LockRequest" := FALSE;
       "ST10_SafetyGate_InterfaceDB".L.Status_1 := 2;
   END_IF;
   #_w5 := #_w2 AND ("ST10_SafetyGate_InterfaceDB".L.Status_1 = 3) AND "iMateriel Door Locking FeedBack_K1";
   #_w6 := #_w5 AND NOT "ST10_SafetyGate_InterfaceDB".L.p[1];   // rising edge
   "ST10_SafetyGate_InterfaceDB".L.p[1] := #_w5;
   IF #_w6 THEN
       "ST10_MaterialGate7_DB"."sSafetyGate UnlockRequest" := FALSE;
       "ST10_MaterialGate7_DB"."sSafetyGate LockRequest" := TRUE;
       "ST10_SafetyGate_InterfaceDB".L.Status_1 := 4;
   END_IF;
   IF #_w1 AND ("ST10_SafetyGate_InterfaceDB".L.Status_1 <> 1) AND ("ST10_SafetyGate_InterfaceDB".L.Status_1 <> 2) AND ("ST10_SafetyGate_InterfaceDB".L.Status_1 <> 3) AND ("ST10_SafetyGate_InterfaceDB".L.Status_1 <> 4) THEN
       "ST10_SafetyGate_InterfaceDB".L.Status_1 := 1;
   END_IF;
   IF #_w1 AND ("ST10_SafetyGate_InterfaceDB".L.Status_1 = 2) AND NOT "iUnloading_Button" THEN
       "ST10_SafetyGate_InterfaceDB".L.Status_1 := 3;
   END_IF;
   IF #_w1 AND ("ST10_SafetyGate_InterfaceDB".L.Status_1 = 4) AND NOT "iUnloading_Button" THEN
       "ST10_SafetyGate_InterfaceDB".L.Status_1 := 5;
   END_IF;
END_REGION

REGION Network 33: H
END_REGION
END_FUNCTION

FUNCTION_BLOCK "FB_Tower_4Lamp"   // FB5050, LAD
{ S7_Optimized_Access := 'TRUE' }
// stored: AutoNumber false, MemoryReserve 100, SetENOAutomatically false
   VAR_INPUT
      iReady : Bool;   // 系统OK
      iManual_Mode : Bool;
      iAuto_Mode : Bool;
      iAuto_Running : Bool;   // 自动运行信号
      iCheck_Mode : Bool;
      iIdle : Bool;   // 自动运行中空闲信号
      iWarning : Bool;
      iFault : Bool;
      "i0.5s_Pulse" : Bool;   // 0.5S脉冲
      i1s_Pulse : Bool;   // 1S脉冲
      i2s_Pulse : Bool;   // 2S脉冲
      iResetButton : Bool;   // 复位按钮
      "iE-StopButtonOK" : Bool;   // 急停按钮未按下
      iSafetyGateClosed : Bool;   // 安全门关闭信号
      iSafetyGateRelayOK : Bool;   // 安全门继电器输出OK
      iPowerOn : Bool;   // 系统上电信号
      iMachineHomePos : Bool;   // 所有设备在原始位
      iWorkAreaLightButton : Bool;   // HMI工作区域照明按钮
      iTest_Lamp : Bool;   // 灯测试按钮
   END_VAR
   VAR_OUTPUT
      oRed_Lamp : Bool;   // 塔灯-红色
      oYellow_Lamp : Bool;   // 塔灯-黄色
      oGreen_Lamp : Bool;   // 塔灯-绿色
      oBlue_Lamp : Bool;   // 塔灯-蓝色 1.蓝灯常亮表示设备在原位;2.蓝灯闪烁表示工位缺料等待上料
      oBuzzer : Bool;   // 塔灯-蜂鸣器
      oPowerOn : Bool;   // 系统上电指示灯
      oResetLamp : Bool;   // 复位按钮指示灯
      oWorkArea1_LightingOn : Bool;   // 工作区域1 照明打开
      oWorkArea2_LightingOn : Bool;   // 工作区域2 照明打开
      oWorkArea3_LightingOn : Bool;   // 工作区域3 照明打开
   END_VAR
   VAR_IN_OUT
      ioStationWaitingLoadPart : Bool;   // 工位等待工位上料
      ioBuzzerON : Bool;   // 蜂鸣器屏蔽开关
      ioBuzzerSetVal : Int;   // 蜂鸣器鸣叫设定值
   END_VAR
   VAR
      TON : Array[0..10] of TON_TIME;
      sRed_Lamp { S7_SetPoint := 'True'} : Bool;
      sResetButtonPressed : Bool;   // 复位按钮已按下
      sBuzzerOnCurrentVal : Int;   // 蜂鸣器鸣叫实际值
      P_TRIG : Array[0..10] of Bool;
      N_TRIG : Array[0..10] of Bool;
   END_VAR
   VAR_TEMP   // added for the SCL form of the ladder/FBD networks
      _w1 : Bool;
      _w2 : Bool;
      _w3 : Bool;
      _w4 : Bool;
      _w5 : Bool;
      _w6 : Bool;
   END_VAR
BEGIN

REGION Network 1: 塔灯-红色 / TowerLamp_Red
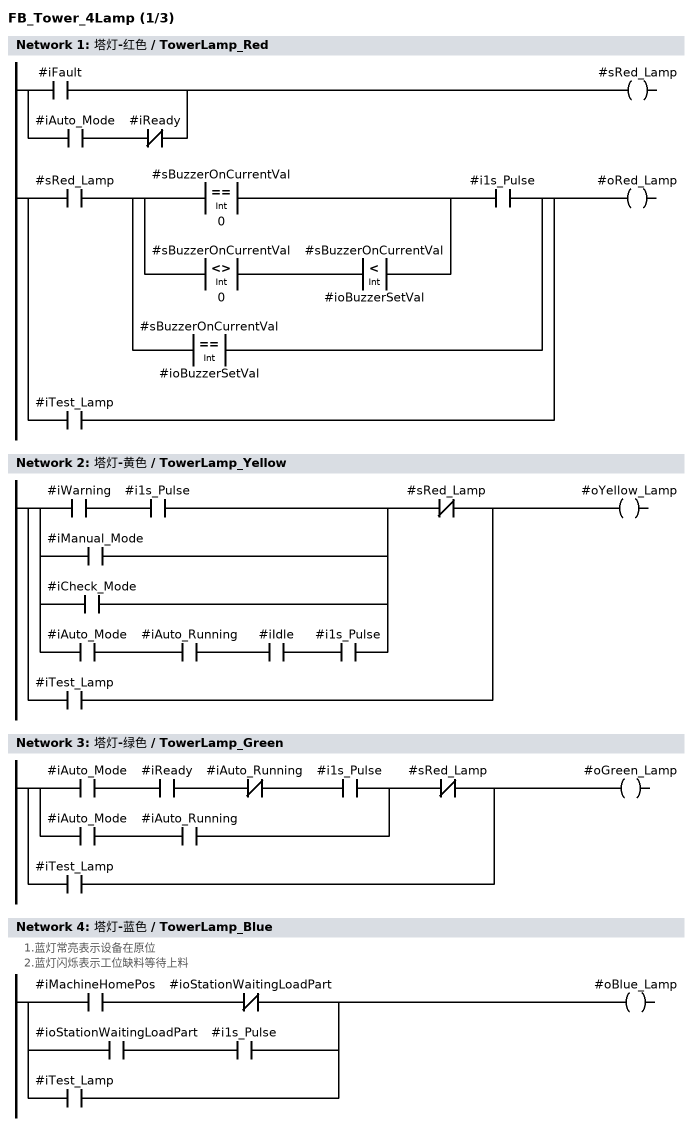
   RUNG wire#powerrail
      Contact( #iFault )
      wire#w1
      Coil( #sRed_Lamp )
   END_RUNG
   RUNG wire#powerrail
      Contact( #iAuto_Mode )
      I_Contact( #iReady )
   END_RUNG wire#w1
   RUNG wire#powerrail
      Contact( #sRed_Lamp )
      wire#w2
      { S7_Templates := "SrcType := Int" } EQ_Contact(in1 := #sBuzzerOnCurrentVal, in2 := 0)
      wire#w3
      Contact( #i1s_Pulse )
      wire#w4
      Coil( #oRed_Lamp )
   END_RUNG
   RUNG wire#w2
      { S7_Templates := "SrcType := Int" } NE_Contact(in1 := #sBuzzerOnCurrentVal, in2 := 0)
      { S7_Templates := "SrcType := Int" } LT_Contact(in1 := #sBuzzerOnCurrentVal, in2 := #ioBuzzerSetVal)
   END_RUNG wire#w3
   RUNG wire#w2
      { S7_Templates := "SrcType := Int" } EQ_Contact(in1 := #sBuzzerOnCurrentVal, in2 := #ioBuzzerSetVal)
   END_RUNG wire#w4
   RUNG wire#powerrail
      Contact( #iTest_Lamp )
   END_RUNG wire#w4
   // the same network as SCL:
   #sRed_Lamp := #iFault OR (#iAuto_Mode AND NOT #iReady);
   #oRed_Lamp := (#sRed_Lamp AND ((((#sBuzzerOnCurrentVal = 0) OR ((#sBuzzerOnCurrentVal <> 0) AND (#sBuzzerOnCurrentVal < #ioBuzzerSetVal))) AND #i1s_Pulse) OR (#sBuzzerOnCurrentVal = #ioBuzzerSetVal))) OR #iTest_Lamp;
END_REGION

REGION Network 2: 塔灯-黄色 / TowerLamp_Yellow
   RUNG wire#powerrail
      Contact( #iWarning )
      Contact( #i1s_Pulse )
      wire#w1
      I_Contact( #sRed_Lamp )
      wire#w2
      Coil( #oYellow_Lamp )
   END_RUNG
   RUNG wire#powerrail
      Contact( #iManual_Mode )
   END_RUNG wire#w1
   RUNG wire#powerrail
      Contact( #iCheck_Mode )
   END_RUNG wire#w1
   RUNG wire#powerrail
      Contact( #iAuto_Mode )
      Contact( #iAuto_Running )
      Contact( #iIdle )
      Contact( #i1s_Pulse )
   END_RUNG wire#w1
   RUNG wire#powerrail
      Contact( #iTest_Lamp )
   END_RUNG wire#w2
   // the same network as SCL:
   #oYellow_Lamp := (((#iWarning AND #i1s_Pulse) OR #iManual_Mode OR #iCheck_Mode OR (#iAuto_Mode AND #iAuto_Running AND #iIdle AND #i1s_Pulse)) AND NOT #sRed_Lamp) OR #iTest_Lamp;
END_REGION

REGION Network 3: 塔灯-绿色 / TowerLamp_Green
   RUNG wire#powerrail
      Contact( #iAuto_Mode )
      Contact( #iReady )
      I_Contact( #iAuto_Running )
      Contact( #i1s_Pulse )
      wire#w1
      I_Contact( #sRed_Lamp )
      wire#w2
      Coil( #oGreen_Lamp )
   END_RUNG
   RUNG wire#powerrail
      Contact( #iAuto_Mode )
      Contact( #iAuto_Running )
   END_RUNG wire#w1
   RUNG wire#powerrail
      Contact( #iTest_Lamp )
   END_RUNG wire#w2
   // the same network as SCL:
   #oGreen_Lamp := (((#iAuto_Mode AND #iReady AND NOT #iAuto_Running AND #i1s_Pulse) OR (#iAuto_Mode AND #iAuto_Running)) AND NOT #sRed_Lamp) OR #iTest_Lamp;
END_REGION

REGION Network 4: 塔灯-蓝色 / TowerLamp_Blue
   // 1.蓝灯常亮表示设备在原位
   // 2.蓝灯闪烁表示工位缺料等待上料
   RUNG wire#powerrail
      Contact( #iMachineHomePos )
      I_Contact( #ioStationWaitingLoadPart )
      wire#w1
      Coil( #oBlue_Lamp )
   END_RUNG
   RUNG wire#powerrail
      Contact( #ioStationWaitingLoadPart )
      Contact( #i1s_Pulse )
   END_RUNG wire#w1
   RUNG wire#powerrail
      Contact( #iTest_Lamp )
   END_RUNG wire#w1
   // the same network as SCL:
   #oBlue_Lamp := (#iMachineHomePos AND NOT #ioStationWaitingLoadPart) OR (#ioStationWaitingLoadPart AND #i1s_Pulse) OR #iTest_Lamp;
END_REGION

REGION Network 5: 蜂鸣器蜂鸣次数 / Number of buzzer buzzes
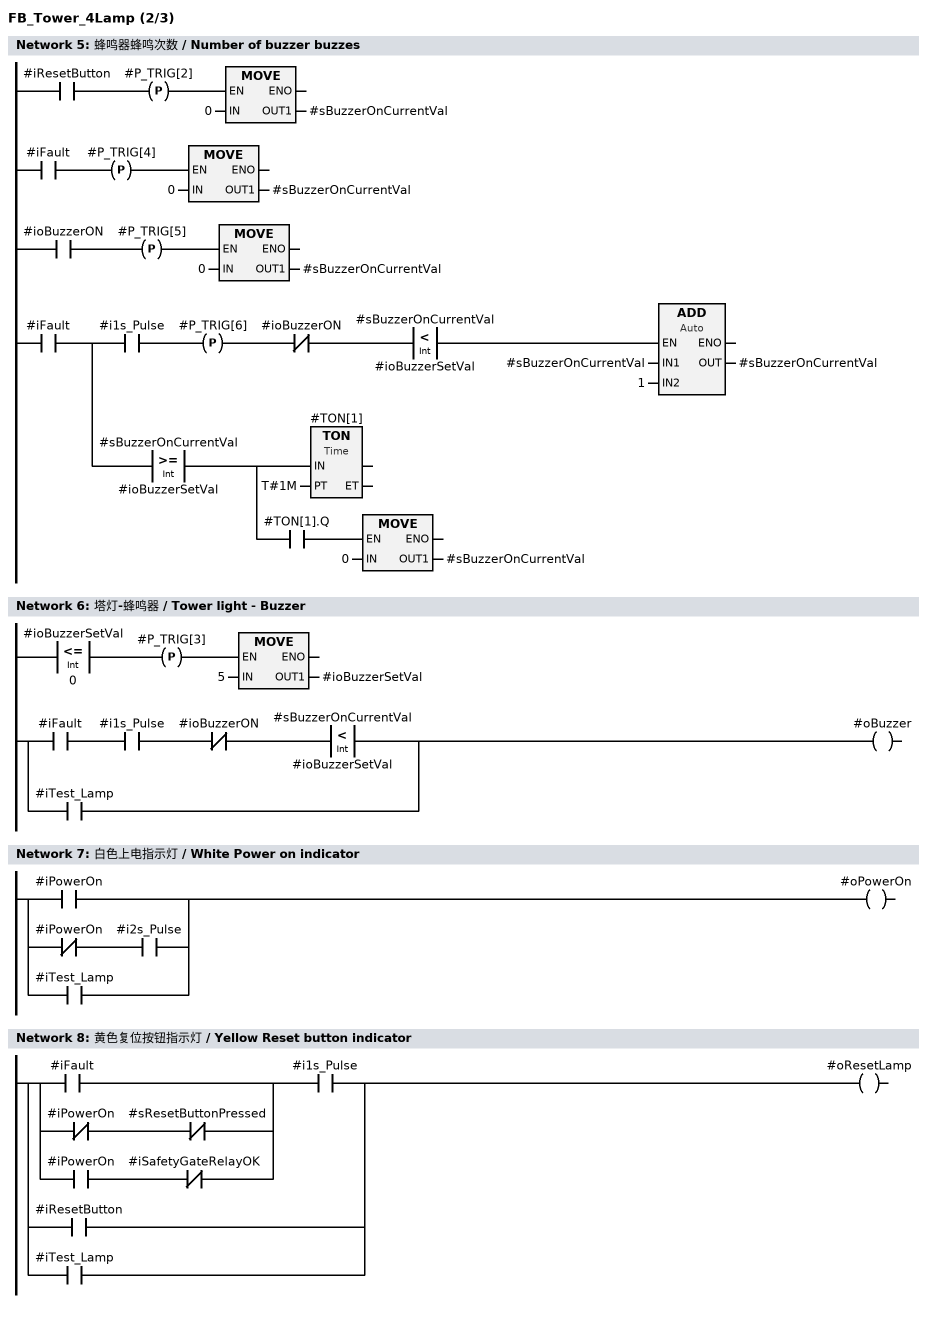
   RUNG wire#powerrail
      Contact( #iResetButton )
      P_Trig( #P_TRIG[2] )
      Move(in := 0, out1 => #sBuzzerOnCurrentVal)
   END_RUNG
   RUNG wire#powerrail
      Contact( #iFault )
      P_Trig( #P_TRIG[4] )
      Move(in := 0, out1 => #sBuzzerOnCurrentVal)
   END_RUNG
   RUNG wire#powerrail
      Contact( #ioBuzzerON )
      P_Trig( #P_TRIG[5] )
      Move(in := 0, out1 => #sBuzzerOnCurrentVal)
   END_RUNG
   RUNG wire#powerrail
      Contact( #iFault )
      wire#w1
      Contact( #i1s_Pulse )
      P_Trig( #P_TRIG[6] )
      I_Contact( #ioBuzzerON )
      { S7_Templates := "SrcType := Int" } LT_Contact(in1 := #sBuzzerOnCurrentVal, in2 := #ioBuzzerSetVal)
      Add(in1 := #sBuzzerOnCurrentVal, in2 := 1, out => #sBuzzerOnCurrentVal)
   END_RUNG
   RUNG wire#w1
      { S7_Templates := "SrcType := Int" } GE_Contact(in1 := #sBuzzerOnCurrentVal, in2 := #ioBuzzerSetVal)
      wire#w2
      { S7_Templates := "time_type := Time" } #TON[1].TON(pt := T#1M, et =>)
   END_RUNG
   RUNG wire#w2
      Contact( #TON[1].Q )
      Move(in := 0, out1 => #sBuzzerOnCurrentVal)
   END_RUNG
   // the same network as SCL:
   #_w1 := #iResetButton AND NOT #P_TRIG[2];   // rising edge
   #P_TRIG[2] := #iResetButton;
   IF #_w1 THEN #sBuzzerOnCurrentVal := 0; END_IF;
   #_w2 := #iFault AND NOT #P_TRIG[4];   // rising edge
   #P_TRIG[4] := #iFault;
   IF #_w2 THEN #sBuzzerOnCurrentVal := 0; END_IF;
   #_w3 := #ioBuzzerON AND NOT #P_TRIG[5];   // rising edge
   #P_TRIG[5] := #ioBuzzerON;
   IF #_w3 THEN #sBuzzerOnCurrentVal := 0; END_IF;
   #_w4 := #iFault AND #i1s_Pulse;
   #_w5 := #_w4 AND NOT #P_TRIG[6];   // rising edge
   #P_TRIG[6] := #_w4;
   IF #_w5 AND NOT #ioBuzzerON AND (#sBuzzerOnCurrentVal < #ioBuzzerSetVal) THEN
       #sBuzzerOnCurrentVal := #sBuzzerOnCurrentVal + 1;
   END_IF;
   #_w6 := #iFault AND (#sBuzzerOnCurrentVal >= #ioBuzzerSetVal);
   #TON[1].TON(IN := #_w6, PT := T#1M);
   IF #_w6 AND #TON[1].Q THEN #sBuzzerOnCurrentVal := 0; END_IF;
END_REGION

REGION Network 6: 塔灯-蜂鸣器 / Tower light - Buzzer
   RUNG wire#powerrail
      { S7_Templates := "SrcType := Int" } LE_Contact(in1 := #ioBuzzerSetVal, in2 := 0)
      P_Trig( #P_TRIG[3] )
      Move(in := 5, out1 => #ioBuzzerSetVal)
   END_RUNG
   RUNG wire#powerrail
      Contact( #iFault )
      Contact( #i1s_Pulse )
      I_Contact( #ioBuzzerON )
      { S7_Templates := "SrcType := Int" } LT_Contact(in1 := #sBuzzerOnCurrentVal, in2 := #ioBuzzerSetVal)
      wire#w1
      Coil( #oBuzzer )
   END_RUNG
   RUNG wire#powerrail
      Contact( #iTest_Lamp )
   END_RUNG wire#w1
   // the same network as SCL:
   #_w1 := #ioBuzzerSetVal <= 0;
   #_w2 := #_w1 AND NOT #P_TRIG[3];   // rising edge
   #P_TRIG[3] := #_w1;
   IF #_w2 THEN #ioBuzzerSetVal := 5; END_IF;
   #oBuzzer := (#iFault AND #i1s_Pulse AND NOT #ioBuzzerON AND (#sBuzzerOnCurrentVal < #ioBuzzerSetVal)) OR #iTest_Lamp;
END_REGION

REGION Network 7: 白色上电指示灯 / White Power on indicator
   RUNG wire#powerrail
      Contact( #iPowerOn )
      wire#w1
      Coil( #oPowerOn )
   END_RUNG
   RUNG wire#powerrail
      I_Contact( #iPowerOn )
      Contact( #i2s_Pulse )
   END_RUNG wire#w1
   RUNG wire#powerrail
      Contact( #iTest_Lamp )
   END_RUNG wire#w1
   // the same network as SCL:
   #oPowerOn := #iPowerOn OR (NOT #iPowerOn AND #i2s_Pulse) OR #iTest_Lamp;
END_REGION

REGION Network 8: 黄色复位按钮指示灯 / Yellow Reset button indicator
   RUNG wire#powerrail
      Contact( #iFault )
      wire#w1
      Contact( #i1s_Pulse )
      wire#w2
      Coil( #oResetLamp )
   END_RUNG
   RUNG wire#powerrail
      I_Contact( #iPowerOn )
      I_Contact( #sResetButtonPressed )
   END_RUNG wire#w1
   RUNG wire#powerrail
      Contact( #iPowerOn )
      I_Contact( #iSafetyGateRelayOK )
   END_RUNG wire#w1
   RUNG wire#powerrail
      Contact( #iResetButton )
   END_RUNG wire#w2
   RUNG wire#powerrail
      Contact( #iTest_Lamp )
   END_RUNG wire#w2
   // the same network as SCL:
   #oResetLamp := ((#iFault OR (NOT #iPowerOn AND NOT #sResetButtonPressed) OR (#iPowerOn AND NOT #iSafetyGateRelayOK)) AND #i1s_Pulse) OR #iResetButton OR #iTest_Lamp;
END_REGION

REGION Network 9: 复位按钮已按下 / The reset button has been pressed
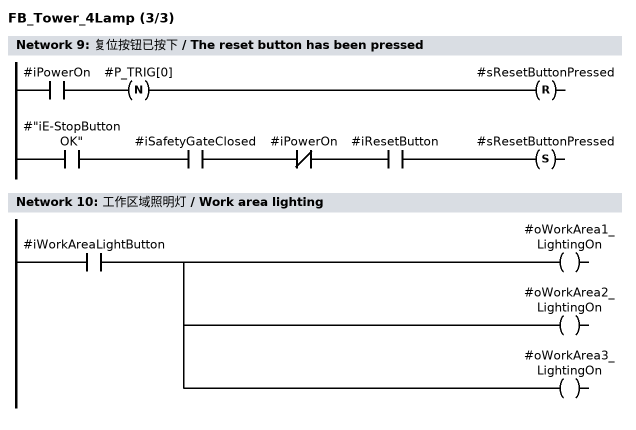
   RUNG wire#powerrail
      Contact( #iPowerOn )
      N_Trig( #P_TRIG[0] )
      R_Coil( #sResetButtonPressed )
   END_RUNG
   RUNG wire#powerrail
      Contact( #"iE-StopButtonOK" )
      Contact( #iSafetyGateClosed )
      I_Contact( #iPowerOn )
      Contact( #iResetButton )
      S_Coil( #sResetButtonPressed )
   END_RUNG
   // the same network as SCL:
   #_w1 := NOT #iPowerOn AND #P_TRIG[0];   // falling edge
   #P_TRIG[0] := #iPowerOn;
   IF #_w1 THEN #sResetButtonPressed := FALSE; END_IF;
   IF #"iE-StopButtonOK" AND #iSafetyGateClosed AND NOT #iPowerOn AND #iResetButton THEN
       #sResetButtonPressed := TRUE;
   END_IF;
END_REGION

REGION Network 10: 工作区域照明灯 / Work area lighting
   RUNG wire#powerrail
      Contact( #iWorkAreaLightButton )
      wire#w1
      Coil( #oWorkArea1_LightingOn )
   END_RUNG
   RUNG wire#w1
      Coil( #oWorkArea2_LightingOn )
   END_RUNG
   RUNG wire#w1
      Coil( #oWorkArea3_LightingOn )
   END_RUNG
   // the same network as SCL:
   #oWorkArea1_LightingOn := #iWorkAreaLightButton;
   #oWorkArea2_LightingOn := #iWorkAreaLightButton;
   #oWorkArea3_LightingOn := #iWorkAreaLightButton;
END_REGION
END_FUNCTION_BLOCK

FUNCTION "ST10_Auto" : Void   // FC1003, LAD
{ S7_Optimized_Access := 'FALSE' }
// stored: AutoNumber false, SetENOAutomatically false
   VAR_INPUT
      iSysMode : "RCS_SysComInterface_V1";
   END_VAR
   VAR_TEMP
      i : Int;
      tBool : Bool;
      FlankWord : Int;
   END_VAR
   VAR_TEMP   // added for the SCL form of the ladder/FBD networks
      _w1 : Bool;
      _w2 : Bool;
      _w3 : Bool;
      _w4 : Bool;
      _w5 : Bool;
      _w6 : Bool;
   END_VAR
BEGIN

REGION Network 1
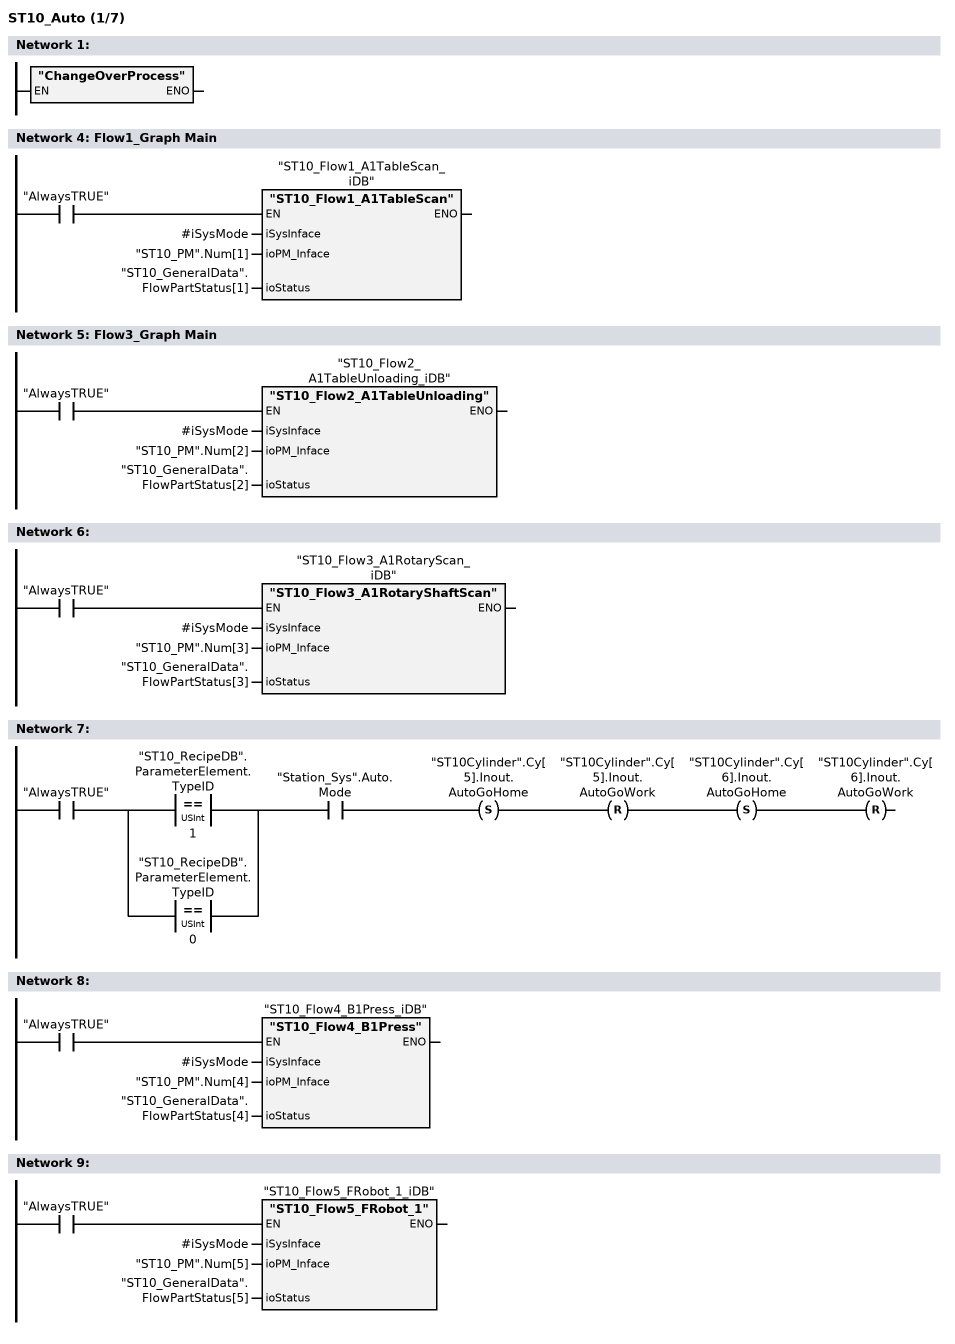
   RUNG wire#powerrail
      "ChangeOverProcess"()
   END_RUNG
   // the same network as SCL:
   "ChangeOverProcess"();
END_REGION

NETWORK
TITLE = AutoMain//自动
//Autorunning is not allowed in manual mode
      A     "Station_Sys".Manual.Mode;
      R     "Station_Sys".Auto.Running;
//one cycle interface
      A     "Station_Sys".Cmd.OneCycle;
      =     "ST10_PM".Num[1].TriggerOneCycle;
      =     "ST10_PM".Num[2].TriggerOneCycle;
      =     "ST10_PM".Num[3].TriggerOneCycle;
      =     "ST10_PM".Num[4].TriggerOneCycle;
      =     "ST10_PM".Num[5].TriggerOneCycle;
      =     "ST10_PM".Num[6].TriggerOneCycle;
      =     "ST10_PM".Num[7].TriggerOneCycle;
      =     "ST10_PM".Num[8].TriggerOneCycle;
      =     "ST10_PM".Num[11].TriggerOneCycle;
      =     "ST10_PM".Num[12].TriggerOneCycle;
      =     "ST10_PM".Num[14].TriggerOneCycle;
      =     "ST10_PM".Num[15].TriggerOneCycle;
      =     "ST10_PM".Num[16].TriggerOneCycle;
      =     "ST10_PM".Num[21].TriggerOneCycle;
      =     "ST10_PM".Num[22].TriggerOneCycle;
      =     "ST10_PM".Num[23].TriggerOneCycle;
      =     "ST10_PM".Num[24].TriggerOneCycle;


NETWORK
TITLE = InitialStatus-初始化状态
//Initilizing
      O     "ST10_PM".Num[1].InitialRun;
      O     "ST10_PM".Num[2].InitialRun;
      O     "ST10_PM".Num[3].InitialRun;
      O     "ST10_PM".Num[4].InitialRun;
      O     "ST10_PM".Num[5].InitialRun;
      O     "ST10_PM".Num[6].InitialRun;
      O     "ST10_PM".Num[7].InitialRun;
      O     "ST10_PM".Num[8].InitialRun;
      O     "ST10_PM".Num[11].InitialRun;
      O     "ST10_PM".Num[12].InitialRun;
      O     "ST10_PM".Num[14].InitialRun;
      O     "ST10_PM".Num[15].InitialRun;
      O     "ST10_PM".Num[21].InitialRun;
      O     "ST10_PM".Num[22].InitialRun;
      O     "ST10_PM".Num[23].InitialRun;
      O     "ST10_PM".Num[24].InitialRun;
      =     "Station_Sys".Initial.Running;
//Initilize ok

      A     "ST10_PM".Num[1].InitialOK;
      A     "ST10_PM".Num[2].InitialOK;
      A     "ST10_PM".Num[3].InitialOK;
      A     "ST10_PM".Num[4].InitialOK;
      A     "ST10_PM".Num[5].InitialOK;
      A     "ST10_PM".Num[6].InitialOK;
      A     "ST10_PM".Num[7].InitialOK;
      A     "ST10_PM".Num[8].InitialOK;
      A     "ST10_PM".Num[11].InitialOK;
      A     "ST10_PM".Num[12].InitialOK;
      A     "ST10_PM".Num[14].InitialOK;
      A     "ST10_PM".Num[15].InitialOK;

      A     "ST10_PM".Num[21].InitialOK;
      A     "ST10_PM".Num[22].InitialOK;
      A     "ST10_PM".Num[23].InitialOK;
      A     "ST10_PM".Num[24].InitialOK;
      =     "Station_Sys".Initial.OK;

//Auto running
      A     "Station_Sys".Auto.Mode;
      A(;
      O     "ST10_PM".Num[1].Running;
      O     "ST10_PM".Num[2].Running;
      O     "ST10_PM".Num[3].Running;
      O     "ST10_PM".Num[4].Running;
      O     "ST10_PM".Num[5].Running;
      O     "ST10_PM".Num[6].Running;
      O     "ST10_PM".Num[7].Running;
      O     "ST10_PM".Num[8].Running;
      O     "ST10_PM".Num[11].Running;
      O     "ST10_PM".Num[12].Running;
      O     "ST10_PM".Num[14].Running;
      O     "ST10_PM".Num[15].Running;

      O     "ST10_PM".Num[21].Running;
      O     "ST10_PM".Num[22].Running;
      O     "ST10_PM".Num[23].Running;
      O     "ST10_PM".Num[24].Running;
      );
// AN    "Station_Sys".Auto.AllRun
      =     "Station_Sys".Auto.Running;
//All run
      A     "ST10_PM".Num[1].Running;
      A     "ST10_PM".Num[2].Running;
      A     "ST10_PM".Num[3].Running;
      A     "ST10_PM".Num[4].Running;
      A     "ST10_PM".Num[5].Running;
      A     "ST10_PM".Num[6].Running;
      A     "ST10_PM".Num[7].Running;
      A     "ST10_PM".Num[8].Running;
      A     "ST10_PM".Num[11].Running;
      A     "ST10_PM".Num[12].Running;
      A     "ST10_PM".Num[14].Running;
      A     "ST10_PM".Num[15].Running;

      A     "ST10_PM".Num[21].Running;
      A     "ST10_PM".Num[22].Running;
      A     "ST10_PM".Num[23].Running;
      A     "ST10_PM".Num[24].Running;
      =     "Station_Sys".Auto.AllRun;




REGION Network 4: Flow1_Graph Main
   RUNG wire#powerrail
      Contact( "AlwaysTRUE" )
      "ST10_Flow1_A1TableScan_iDB"(iSysInface := #iSysMode, ioPM_Inface := "ST10_PM".Num[1], ioStatus := "ST10_GeneralData".FlowPartStatus[1])
   END_RUNG
   // the same network as SCL:
   IF "AlwaysTRUE" THEN
       "ST10_Flow1_A1TableScan_iDB"(iSysInface := #iSysMode,   // "ST10_Flow1_A1TableScan"
                               ioPM_Inface := "ST10_PM".Num[1],
                               ioStatus := "ST10_GeneralData".FlowPartStatus[1]);
   END_IF;
END_REGION

REGION Network 5: Flow3_Graph Main
   RUNG wire#powerrail
      Contact( "AlwaysTRUE" )
      "ST10_Flow2_A1TableUnloading_iDB"(iSysInface := #iSysMode, ioPM_Inface := "ST10_PM".Num[2], ioStatus := "ST10_GeneralData".FlowPartStatus[2])
   END_RUNG
   // the same network as SCL:
   IF "AlwaysTRUE" THEN
       "ST10_Flow2_A1TableUnloading_iDB"(iSysInface := #iSysMode,   // "ST10_Flow2_A1TableUnloading"
                               ioPM_Inface := "ST10_PM".Num[2],
                               ioStatus := "ST10_GeneralData".FlowPartStatus[2]);
   END_IF;
END_REGION

REGION Network 6
   RUNG wire#powerrail
      Contact( "AlwaysTRUE" )
      "ST10_Flow3_A1RotaryScan_iDB"(iSysInface := #iSysMode, ioPM_Inface := "ST10_PM".Num[3], ioStatus := "ST10_GeneralData".FlowPartStatus[3])
   END_RUNG
   // the same network as SCL:
   IF "AlwaysTRUE" THEN
       "ST10_Flow3_A1RotaryScan_iDB"(iSysInface := #iSysMode,   // "ST10_Flow3_A1RotaryShaftScan"
                               ioPM_Inface := "ST10_PM".Num[3],
                               ioStatus := "ST10_GeneralData".FlowPartStatus[3]);
   END_IF;
END_REGION

REGION Network 7
   RUNG wire#powerrail
      Contact( "AlwaysTRUE" )
      wire#w1
      { S7_Templates := "SrcType := USInt" } EQ_Contact(in1 := "ST10_RecipeDB".ParameterElement.TypeID, in2 := 1)
      wire#w2
      Contact( "Station_Sys".Auto.Mode )
      S_Coil( "ST10Cylinder".Cy[5].Inout.AutoGoHome )
      R_Coil( "ST10Cylinder".Cy[5].Inout.AutoGoWork )
      S_Coil( "ST10Cylinder".Cy[6].Inout.AutoGoHome )
      R_Coil( "ST10Cylinder".Cy[6].Inout.AutoGoWork )
   END_RUNG
   RUNG wire#w1
      { S7_Templates := "SrcType := USInt" } EQ_Contact(in1 := "ST10_RecipeDB".ParameterElement.TypeID, in2 := 0)
   END_RUNG wire#w2
   // the same network as SCL:
   IF "AlwaysTRUE" AND (("ST10_RecipeDB".ParameterElement.TypeID = 1) OR ("ST10_RecipeDB".ParameterElement.TypeID = 0)) AND "Station_Sys".Auto.Mode THEN
       "ST10Cylinder".Cy[5].Inout.AutoGoHome := TRUE;
       "ST10Cylinder".Cy[5].Inout.AutoGoWork := FALSE;
       "ST10Cylinder".Cy[6].Inout.AutoGoHome := TRUE;
       "ST10Cylinder".Cy[6].Inout.AutoGoWork := FALSE;
   END_IF;
END_REGION

REGION Network 8
   RUNG wire#powerrail
      Contact( "AlwaysTRUE" )
      "ST10_Flow4_B1Press_iDB"(iSysInface := #iSysMode, ioPM_Inface := "ST10_PM".Num[4], ioStatus := "ST10_GeneralData".FlowPartStatus[4])
   END_RUNG
   // the same network as SCL:
   IF "AlwaysTRUE" THEN
       "ST10_Flow4_B1Press_iDB"(iSysInface := #iSysMode,   // "ST10_Flow4_B1Press"
                               ioPM_Inface := "ST10_PM".Num[4],
                               ioStatus := "ST10_GeneralData".FlowPartStatus[4]);
   END_IF;
END_REGION

REGION Network 9
   RUNG wire#powerrail
      Contact( "AlwaysTRUE" )
      "ST10_Flow5_FRobot_1_iDB"(iSysInface := #iSysMode, ioPM_Inface := "ST10_PM".Num[5], ioStatus := "ST10_GeneralData".FlowPartStatus[5])
   END_RUNG
   // the same network as SCL:
   IF "AlwaysTRUE" THEN
       "ST10_Flow5_FRobot_1_iDB"(iSysInface := #iSysMode,   // "ST10_Flow5_FRobot_1"
                               ioPM_Inface := "ST10_PM".Num[5],
                               ioStatus := "ST10_GeneralData".FlowPartStatus[5]);
   END_IF;
END_REGION

REGION Network 10
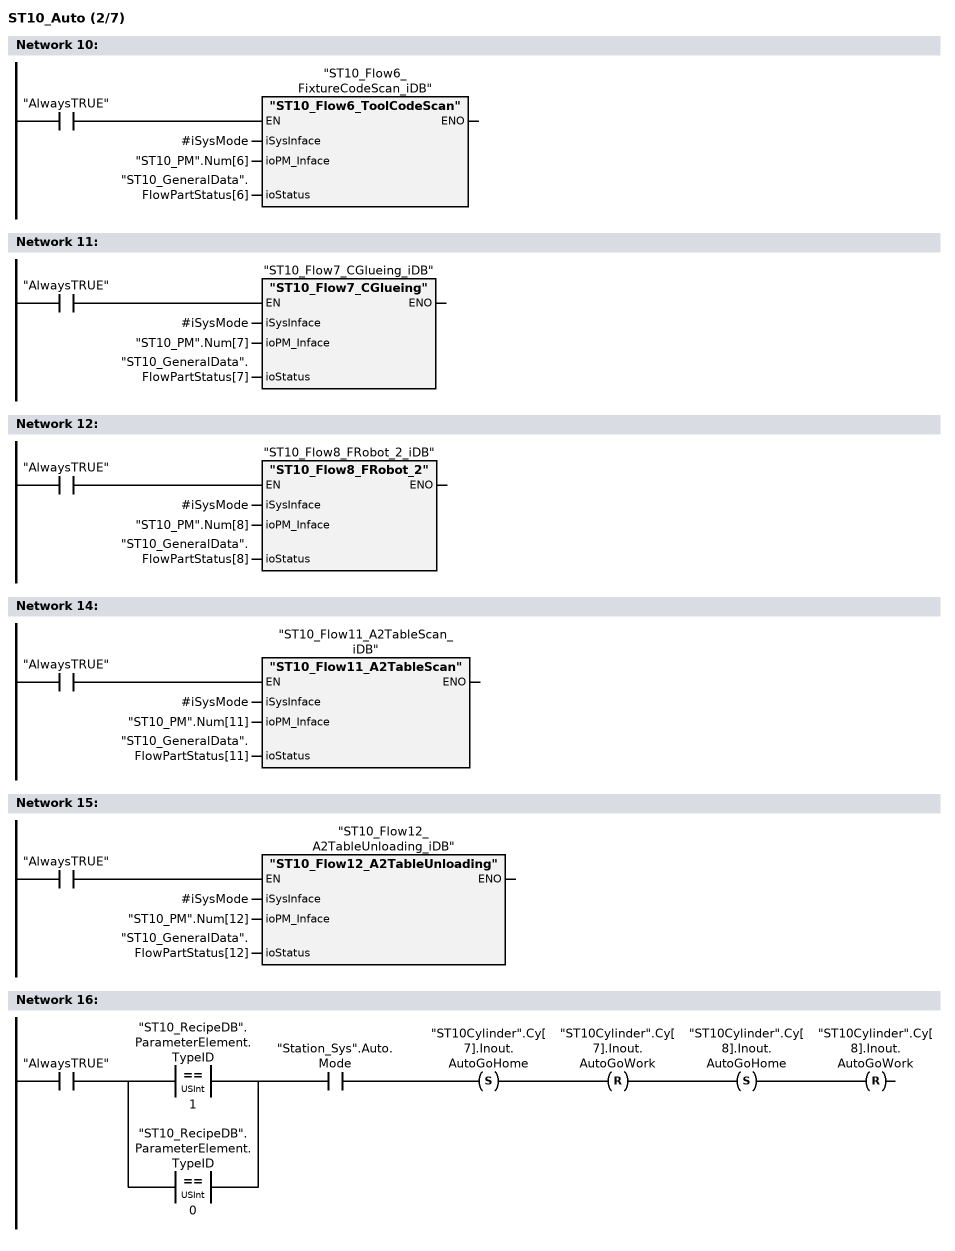
   RUNG wire#powerrail
      Contact( "AlwaysTRUE" )
      "ST10_Flow6_FixtureCodeScan_iDB"(iSysInface := #iSysMode, ioPM_Inface := "ST10_PM".Num[6], ioStatus := "ST10_GeneralData".FlowPartStatus[6])
   END_RUNG
   // the same network as SCL:
   IF "AlwaysTRUE" THEN
       "ST10_Flow6_FixtureCodeScan_iDB"(iSysInface := #iSysMode,   // "ST10_Flow6_ToolCodeScan"
                               ioPM_Inface := "ST10_PM".Num[6],
                               ioStatus := "ST10_GeneralData".FlowPartStatus[6]);
   END_IF;
END_REGION

REGION Network 11
   RUNG wire#powerrail
      Contact( "AlwaysTRUE" )
      "ST10_Flow7_CGlueing_iDB"(iSysInface := #iSysMode, ioPM_Inface := "ST10_PM".Num[7], ioStatus := "ST10_GeneralData".FlowPartStatus[7])
   END_RUNG
   // the same network as SCL:
   IF "AlwaysTRUE" THEN
       "ST10_Flow7_CGlueing_iDB"(iSysInface := #iSysMode,   // "ST10_Flow7_CGlueing"
                               ioPM_Inface := "ST10_PM".Num[7],
                               ioStatus := "ST10_GeneralData".FlowPartStatus[7]);
   END_IF;
END_REGION

REGION Network 12
   RUNG wire#powerrail
      Contact( "AlwaysTRUE" )
      "ST10_Flow8_FRobot_2_iDB"(iSysInface := #iSysMode, ioPM_Inface := "ST10_PM".Num[8], ioStatus := "ST10_GeneralData".FlowPartStatus[8])
   END_RUNG
   // the same network as SCL:
   IF "AlwaysTRUE" THEN
       "ST10_Flow8_FRobot_2_iDB"(iSysInface := #iSysMode,   // "ST10_Flow8_FRobot_2"
                               ioPM_Inface := "ST10_PM".Num[8],
                               ioStatus := "ST10_GeneralData".FlowPartStatus[8]);
   END_IF;
END_REGION

REGION Network 14
   RUNG wire#powerrail
      Contact( "AlwaysTRUE" )
      "ST10_Flow11_A2TableScan_iDB"(iSysInface := #iSysMode, ioPM_Inface := "ST10_PM".Num[11], ioStatus := "ST10_GeneralData".FlowPartStatus[11])
   END_RUNG
   // the same network as SCL:
   IF "AlwaysTRUE" THEN
       "ST10_Flow11_A2TableScan_iDB"(iSysInface := #iSysMode,   // "ST10_Flow11_A2TableScan"
                               ioPM_Inface := "ST10_PM".Num[11],
                               ioStatus := "ST10_GeneralData".FlowPartStatus[11]);
   END_IF;
END_REGION

REGION Network 15
   RUNG wire#powerrail
      Contact( "AlwaysTRUE" )
      "ST10_Flow12_A2TableUnloading_iDB"(iSysInface := #iSysMode, ioPM_Inface := "ST10_PM".Num[12], ioStatus := "ST10_GeneralData".FlowPartStatus[12])
   END_RUNG
   // the same network as SCL:
   IF "AlwaysTRUE" THEN
       "ST10_Flow12_A2TableUnloading_iDB"(iSysInface := #iSysMode,   // "ST10_Flow12_A2TableUnloading"
                               ioPM_Inface := "ST10_PM".Num[12],
                               ioStatus := "ST10_GeneralData".FlowPartStatus[12]);
   END_IF;
END_REGION

REGION Network 16
   RUNG wire#powerrail
      Contact( "AlwaysTRUE" )
      wire#w1
      { S7_Templates := "SrcType := USInt" } EQ_Contact(in1 := "ST10_RecipeDB".ParameterElement.TypeID, in2 := 1)
      wire#w2
      Contact( "Station_Sys".Auto.Mode )
      S_Coil( "ST10Cylinder".Cy[7].Inout.AutoGoHome )
      R_Coil( "ST10Cylinder".Cy[7].Inout.AutoGoWork )
      S_Coil( "ST10Cylinder".Cy[8].Inout.AutoGoHome )
      R_Coil( "ST10Cylinder".Cy[8].Inout.AutoGoWork )
   END_RUNG
   RUNG wire#w1
      { S7_Templates := "SrcType := USInt" } EQ_Contact(in1 := "ST10_RecipeDB".ParameterElement.TypeID, in2 := 0)
   END_RUNG wire#w2
   // the same network as SCL:
   IF "AlwaysTRUE" AND (("ST10_RecipeDB".ParameterElement.TypeID = 1) OR ("ST10_RecipeDB".ParameterElement.TypeID = 0)) AND "Station_Sys".Auto.Mode THEN
       "ST10Cylinder".Cy[7].Inout.AutoGoHome := TRUE;
       "ST10Cylinder".Cy[7].Inout.AutoGoWork := FALSE;
       "ST10Cylinder".Cy[8].Inout.AutoGoHome := TRUE;
       "ST10Cylinder".Cy[8].Inout.AutoGoWork := FALSE;
   END_IF;
END_REGION

REGION Network 17
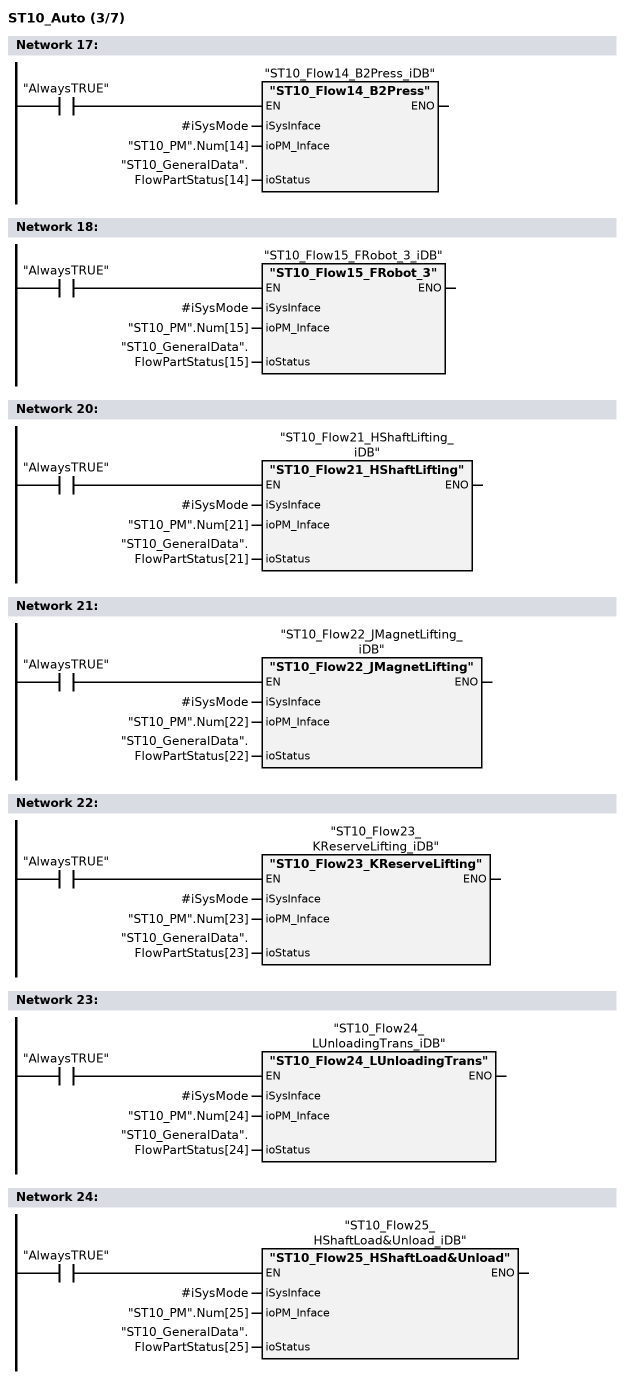
   RUNG wire#powerrail
      Contact( "AlwaysTRUE" )
      "ST10_Flow14_B2Press_iDB"(iSysInface := #iSysMode, ioPM_Inface := "ST10_PM".Num[14], ioStatus := "ST10_GeneralData".FlowPartStatus[14])
   END_RUNG
   // the same network as SCL:
   IF "AlwaysTRUE" THEN
       "ST10_Flow14_B2Press_iDB"(iSysInface := #iSysMode,   // "ST10_Flow14_B2Press"
                               ioPM_Inface := "ST10_PM".Num[14],
                               ioStatus := "ST10_GeneralData".FlowPartStatus[14]);
   END_IF;
END_REGION

REGION Network 18
   RUNG wire#powerrail
      Contact( "AlwaysTRUE" )
      "ST10_Flow15_FRobot_3_iDB"(iSysInface := #iSysMode, ioPM_Inface := "ST10_PM".Num[15], ioStatus := "ST10_GeneralData".FlowPartStatus[15])
   END_RUNG
   // the same network as SCL:
   IF "AlwaysTRUE" THEN
       "ST10_Flow15_FRobot_3_iDB"(iSysInface := #iSysMode,   // "ST10_Flow15_FRobot_3"
                               ioPM_Inface := "ST10_PM".Num[15],
                               ioStatus := "ST10_GeneralData".FlowPartStatus[15]);
   END_IF;
END_REGION

REGION Network 20
   RUNG wire#powerrail
      Contact( "AlwaysTRUE" )
      "ST10_Flow21_HShaftLifting_iDB"(iSysInface := #iSysMode, ioPM_Inface := "ST10_PM".Num[21], ioStatus := "ST10_GeneralData".FlowPartStatus[21])
   END_RUNG
   // the same network as SCL:
   IF "AlwaysTRUE" THEN
       "ST10_Flow21_HShaftLifting_iDB"(iSysInface := #iSysMode,   // "ST10_Flow21_HShaftLifting"
                               ioPM_Inface := "ST10_PM".Num[21],
                               ioStatus := "ST10_GeneralData".FlowPartStatus[21]);
   END_IF;
END_REGION

REGION Network 21
   RUNG wire#powerrail
      Contact( "AlwaysTRUE" )
      "ST10_Flow22_JMagnetLifting_iDB"(iSysInface := #iSysMode, ioPM_Inface := "ST10_PM".Num[22], ioStatus := "ST10_GeneralData".FlowPartStatus[22])
   END_RUNG
   // the same network as SCL:
   IF "AlwaysTRUE" THEN
       "ST10_Flow22_JMagnetLifting_iDB"(iSysInface := #iSysMode,   // "ST10_Flow22_JMagnetLifting"
                               ioPM_Inface := "ST10_PM".Num[22],
                               ioStatus := "ST10_GeneralData".FlowPartStatus[22]);
   END_IF;
END_REGION

REGION Network 22
   RUNG wire#powerrail
      Contact( "AlwaysTRUE" )
      "ST10_Flow23_KReserveLifting_iDB"(iSysInface := #iSysMode, ioPM_Inface := "ST10_PM".Num[23], ioStatus := "ST10_GeneralData".FlowPartStatus[23])
   END_RUNG
   // the same network as SCL:
   IF "AlwaysTRUE" THEN
       "ST10_Flow23_KReserveLifting_iDB"(iSysInface := #iSysMode,   // "ST10_Flow23_KReserveLifting"
                               ioPM_Inface := "ST10_PM".Num[23],
                               ioStatus := "ST10_GeneralData".FlowPartStatus[23]);
   END_IF;
END_REGION

REGION Network 23
   RUNG wire#powerrail
      Contact( "AlwaysTRUE" )
      "ST10_Flow24_LUnloadingTrans_iDB"(iSysInface := #iSysMode, ioPM_Inface := "ST10_PM".Num[24], ioStatus := "ST10_GeneralData".FlowPartStatus[24])
   END_RUNG
   // the same network as SCL:
   IF "AlwaysTRUE" THEN
       "ST10_Flow24_LUnloadingTrans_iDB"(iSysInface := #iSysMode,   // "ST10_Flow24_LUnloadingTrans"
                               ioPM_Inface := "ST10_PM".Num[24],
                               ioStatus := "ST10_GeneralData".FlowPartStatus[24]);
   END_IF;
END_REGION

REGION Network 24
   RUNG wire#powerrail
      Contact( "AlwaysTRUE" )
      "ST10_Flow25_HShaftLoad&Unload_iDB"(iSysInface := #iSysMode, ioPM_Inface := "ST10_PM".Num[25], ioStatus := "ST10_GeneralData".FlowPartStatus[25])
   END_RUNG
   // the same network as SCL:
   IF "AlwaysTRUE" THEN
       "ST10_Flow25_HShaftLoad&Unload_iDB"(iSysInface := #iSysMode,   // "ST10_Flow25_HShaftLoad&Unload"
                               ioPM_Inface := "ST10_PM".Num[25],
                               ioStatus := "ST10_GeneralData".FlowPartStatus[25]);
   END_IF;
END_REGION

REGION Network 25
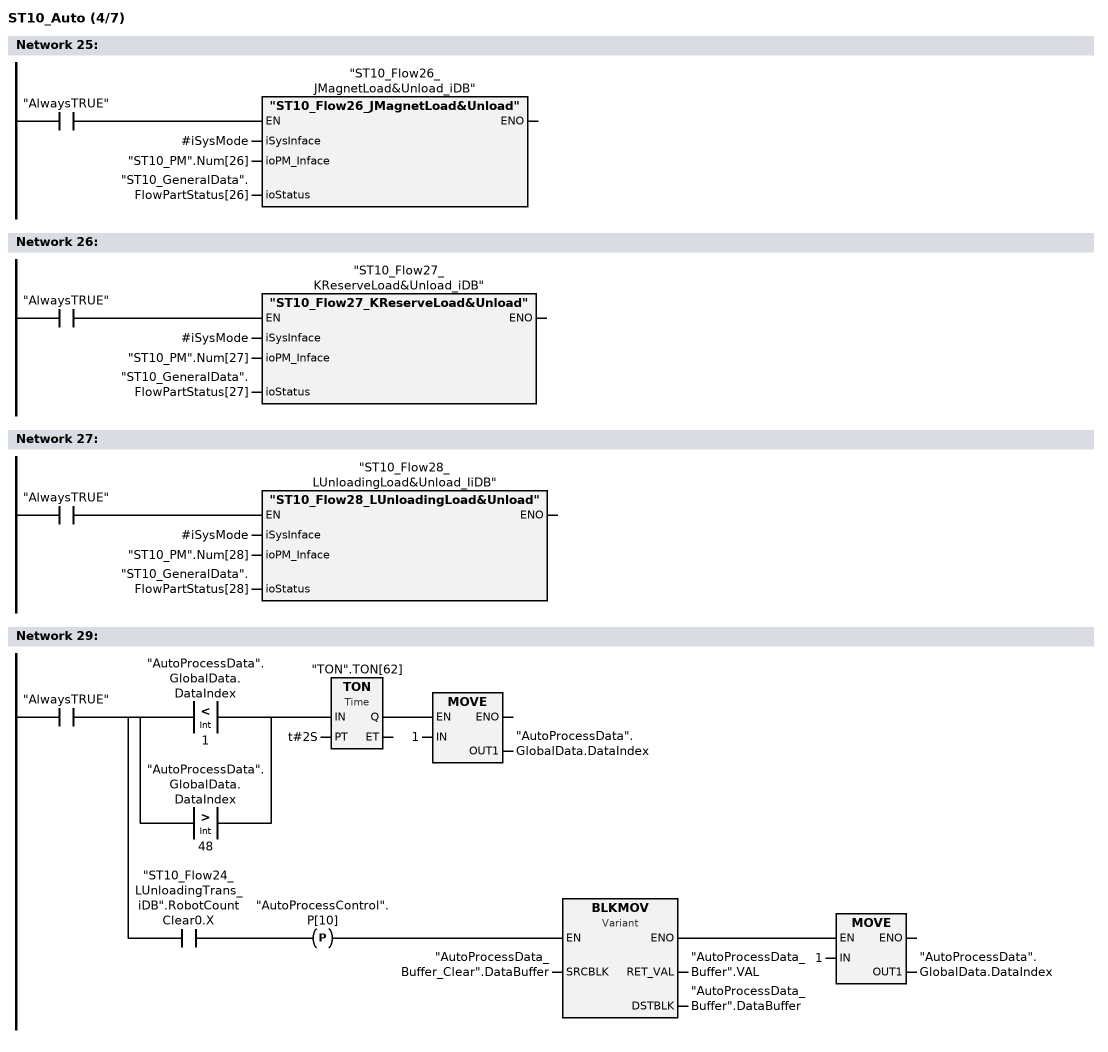
   RUNG wire#powerrail
      Contact( "AlwaysTRUE" )
      "ST10_Flow26_JMagnetLoad&Unload_iDB"(iSysInface := #iSysMode, ioPM_Inface := "ST10_PM".Num[26], ioStatus := "ST10_GeneralData".FlowPartStatus[26])
   END_RUNG
   // the same network as SCL:
   IF "AlwaysTRUE" THEN
       "ST10_Flow26_JMagnetLoad&Unload_iDB"(iSysInface := #iSysMode,   // "ST10_Flow26_JMagnetLoad&Unload"
                               ioPM_Inface := "ST10_PM".Num[26],
                               ioStatus := "ST10_GeneralData".FlowPartStatus[26]);
   END_IF;
END_REGION

REGION Network 26
   RUNG wire#powerrail
      Contact( "AlwaysTRUE" )
      "ST10_Flow27_KReserveLoad&Unload_iDB"(iSysInface := #iSysMode, ioPM_Inface := "ST10_PM".Num[27], ioStatus := "ST10_GeneralData".FlowPartStatus[27])
   END_RUNG
   // the same network as SCL:
   IF "AlwaysTRUE" THEN
       "ST10_Flow27_KReserveLoad&Unload_iDB"(iSysInface := #iSysMode,   // "ST10_Flow27_KReserveLoad&Unload"
                               ioPM_Inface := "ST10_PM".Num[27],
                               ioStatus := "ST10_GeneralData".FlowPartStatus[27]);
   END_IF;
END_REGION

REGION Network 27
   RUNG wire#powerrail
      Contact( "AlwaysTRUE" )
      "ST10_Flow28_LUnloadingLoad&Unload_IiDB"(iSysInface := #iSysMode, ioPM_Inface := "ST10_PM".Num[28], ioStatus := "ST10_GeneralData".FlowPartStatus[28])
   END_RUNG
   // the same network as SCL:
   IF "AlwaysTRUE" THEN
       "ST10_Flow28_LUnloadingLoad&Unload_IiDB"(iSysInface := #iSysMode,   // "ST10_Flow28_LUnloadingLoad&Unload"
                               ioPM_Inface := "ST10_PM".Num[28],
                               ioStatus := "ST10_GeneralData".FlowPartStatus[28]);
   END_IF;
END_REGION

REGION Network 29
   RUNG wire#powerrail
      Contact( "AlwaysTRUE" )
      wire#w1
      { S7_Templates := "SrcType := Int" } LT_Contact(in1 := "AutoProcessData".GlobalData.DataIndex, in2 := 1)
      wire#w2
      { S7_Templates := "time_type := Time" } "TON".TON[62].TON(pt := t#2S, et =>)
      Move(in := 1, out1 => "AutoProcessData".GlobalData.DataIndex)
   END_RUNG
   RUNG wire#w1
      { S7_Templates := "SrcType := Int" } GT_Contact(in1 := "AutoProcessData".GlobalData.DataIndex, in2 := 48)
   END_RUNG wire#w2
   RUNG wire#w1
      Contact( "ST10_Flow24_LUnloadingTrans_iDB".RobotCountClear0.X )
      P_Trig( "AutoProcessControl".P[10] )
      { S7_Templates := "blk_type := Variant" } BLKMOV(SRCBLK := "AutoProcessData_Buffer_Clear".DataBuffer, RET_VAL => "AutoProcessData_Buffer".VAL, DSTBLK => "AutoProcessData_Buffer".DataBuffer)
      Move(in := 1, out1 => "AutoProcessData".GlobalData.DataIndex)
   END_RUNG
   // the same network as SCL:
   "TON".TON[62].TON(IN := "AlwaysTRUE" AND (("AutoProcessData".GlobalData.DataIndex < 1) OR ("AutoProcessData".GlobalData.DataIndex > 48)),
                     PT := t#2S);
   IF "TON".TON[62].Q THEN "AutoProcessData".GlobalData.DataIndex := 1; END_IF;
   #_w1 := "AlwaysTRUE" AND "ST10_Flow24_LUnloadingTrans_iDB".RobotCountClear0.X;
   #_w2 := #_w1 AND NOT "AutoProcessControl".P[10];   // rising edge
   "AutoProcessControl".P[10] := #_w1;
   "AutoProcessData_Buffer".VAL := BLKMOV(EN := #_w2,
                           SRCBLK := "AutoProcessData_Buffer_Clear".DataBuffer,
                           DSTBLK => "AutoProcessData_Buffer".DataBuffer,
                           ENO => #_w3);
   IF #_w3 THEN "AutoProcessData".GlobalData.DataIndex := 1; END_IF;
END_REGION

REGION Network 30
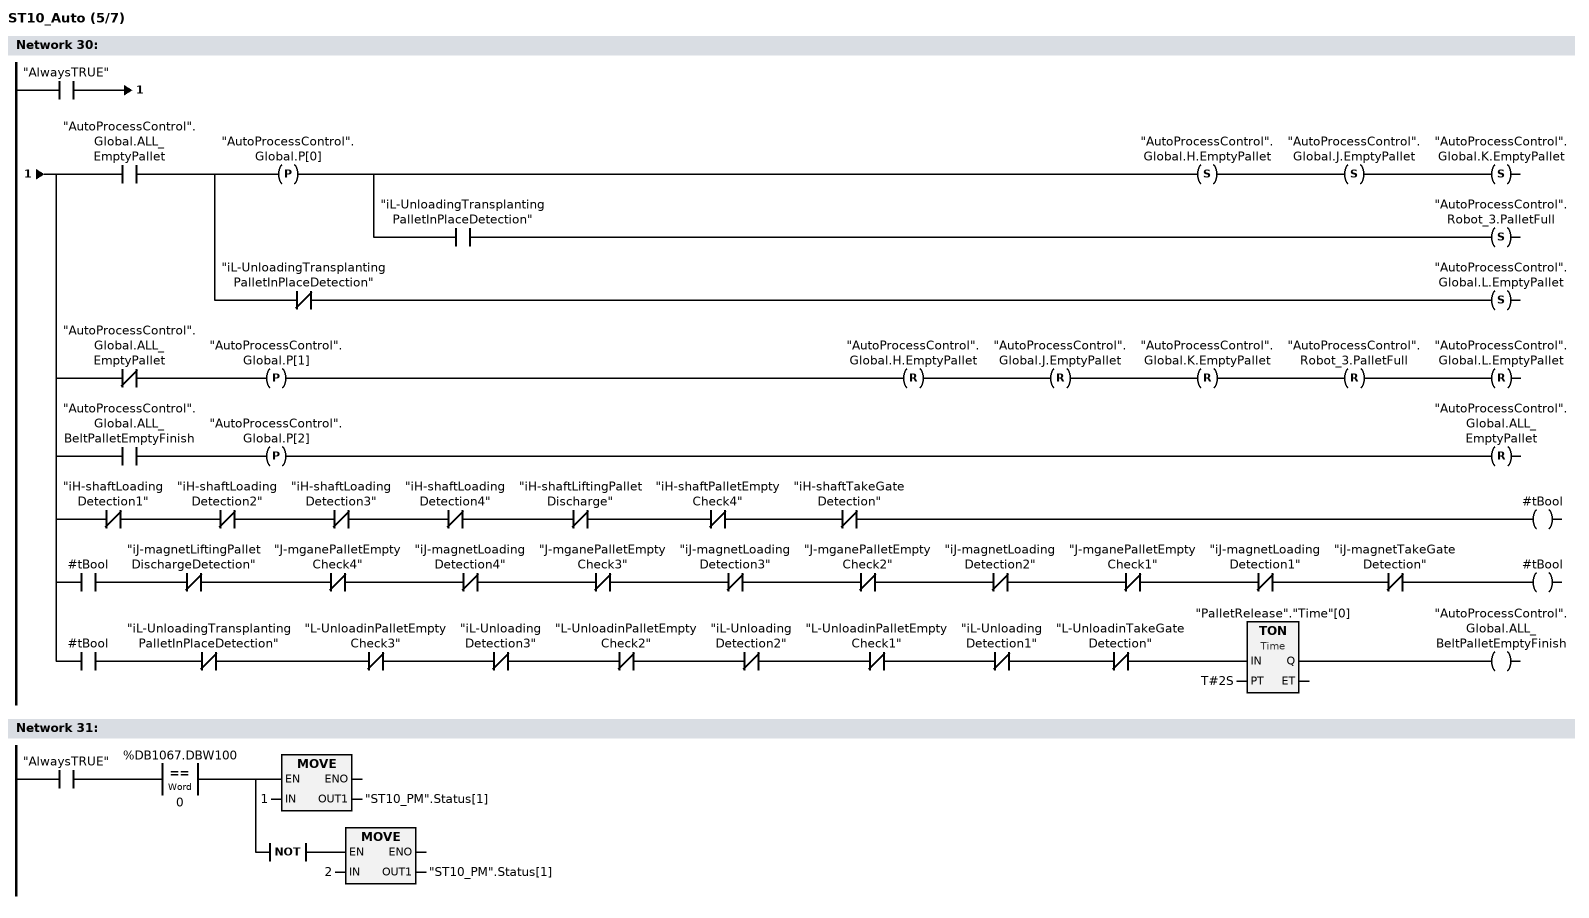
   RUNG wire#powerrail
      Contact( "AlwaysTRUE" )
      wire#w1
      Contact( "AutoProcessControl".Global.ALL_EmptyPallet )
      wire#w2
      P_Trig( "AutoProcessControl".Global.P[0] )
      wire#w3
      S_Coil( "AutoProcessControl".Global.H.EmptyPallet )
      S_Coil( "AutoProcessControl".Global.J.EmptyPallet )
      S_Coil( "AutoProcessControl".Global.K.EmptyPallet )
   END_RUNG
   RUNG wire#w3
      Contact( "iL-UnloadingTransplantingPalletInPlaceDetection" )
      S_Coil( "AutoProcessControl".Robot_3.PalletFull )
   END_RUNG
   RUNG wire#w2
      I_Contact( "iL-UnloadingTransplantingPalletInPlaceDetection" )
      S_Coil( "AutoProcessControl".Global.L.EmptyPallet )
   END_RUNG
   RUNG wire#w1
      I_Contact( "AutoProcessControl".Global.ALL_EmptyPallet )
      P_Trig( "AutoProcessControl".Global.P[1] )
      R_Coil( "AutoProcessControl".Global.H.EmptyPallet )
      R_Coil( "AutoProcessControl".Global.J.EmptyPallet )
      R_Coil( "AutoProcessControl".Global.K.EmptyPallet )
      R_Coil( "AutoProcessControl".Robot_3.PalletFull )
      R_Coil( "AutoProcessControl".Global.L.EmptyPallet )
   END_RUNG
   RUNG wire#w1
      Contact( "AutoProcessControl".Global.ALL_BeltPalletEmptyFinish )
      P_Trig( "AutoProcessControl".Global.P[2] )
      R_Coil( "AutoProcessControl".Global.ALL_EmptyPallet )
   END_RUNG
   RUNG wire#w1
      I_Contact( "iH-shaftLoadingDetection1" )
      I_Contact( "iH-shaftLoadingDetection2" )
      I_Contact( "iH-shaftLoadingDetection3" )
      I_Contact( "iH-shaftLoadingDetection4" )
      I_Contact( "iH-shaftLiftingPalletDischarge" )
      I_Contact( "iH-shaftPalletEmptyCheck4" )
      I_Contact( "iH-shaftTakeGateDetection" )
      Coil( #tBool )
   END_RUNG
   RUNG wire#w1
      Contact( #tBool )
      I_Contact( "iJ-magnetLiftingPalletDischargeDetection" )
      I_Contact( "J-mganePalletEmptyCheck4" )
      I_Contact( "iJ-magnetLoadingDetection4" )
      I_Contact( "J-mganePalletEmptyCheck3" )
      I_Contact( "iJ-magnetLoadingDetection3" )
      I_Contact( "J-mganePalletEmptyCheck2" )
      I_Contact( "iJ-magnetLoadingDetection2" )
      I_Contact( "J-mganePalletEmptyCheck1" )
      I_Contact( "iJ-magnetLoadingDetection1" )
      I_Contact( "iJ-magnetTakeGateDetection" )
      Coil( #tBool )
   END_RUNG
   RUNG wire#w1
      Contact( #tBool )
      I_Contact( "iL-UnloadingTransplantingPalletInPlaceDetection" )
      I_Contact( "L-UnloadinPalletEmptyCheck3" )
      I_Contact( "iL-UnloadingDetection3" )
      I_Contact( "L-UnloadinPalletEmptyCheck2" )
      I_Contact( "iL-UnloadingDetection2" )
      I_Contact( "L-UnloadinPalletEmptyCheck1" )
      I_Contact( "iL-UnloadingDetection1" )
      I_Contact( "L-UnloadinTakeGateDetection" )
      { S7_Templates := "time_type := Time" } "PalletRelease"."Time"[0].TON(pt := T#2S, et =>)
      Coil( "AutoProcessControl".Global.ALL_BeltPalletEmptyFinish )
   END_RUNG
   // the same network as SCL:
   #_w1 := "AlwaysTRUE" AND "AutoProcessControl".Global.ALL_EmptyPallet;
   #_w2 := #_w1 AND NOT "AutoProcessControl".Global.P[0];   // rising edge
   "AutoProcessControl".Global.P[0] := #_w1;
   IF #_w2 THEN
       "AutoProcessControl".Global.H.EmptyPallet := TRUE;
       "AutoProcessControl".Global.J.EmptyPallet := TRUE;
       "AutoProcessControl".Global.K.EmptyPallet := TRUE;
   END_IF;
   IF #_w2 AND "iL-UnloadingTransplantingPalletInPlaceDetection" THEN
       "AutoProcessControl".Robot_3.PalletFull := TRUE;
   END_IF;
   IF #_w1 AND NOT "iL-UnloadingTransplantingPalletInPlaceDetection" THEN
       "AutoProcessControl".Global.L.EmptyPallet := TRUE;
   END_IF;
   #_w3 := "AlwaysTRUE" AND NOT "AutoProcessControl".Global.ALL_EmptyPallet;
   #_w4 := #_w3 AND NOT "AutoProcessControl".Global.P[1];   // rising edge
   "AutoProcessControl".Global.P[1] := #_w3;
   IF #_w4 THEN
       "AutoProcessControl".Global.H.EmptyPallet := FALSE;
       "AutoProcessControl".Global.J.EmptyPallet := FALSE;
       "AutoProcessControl".Global.K.EmptyPallet := FALSE;
       "AutoProcessControl".Robot_3.PalletFull := FALSE;
       "AutoProcessControl".Global.L.EmptyPallet := FALSE;
   END_IF;
   #_w5 := "AlwaysTRUE" AND "AutoProcessControl".Global.ALL_BeltPalletEmptyFinish;
   #_w6 := #_w5 AND NOT "AutoProcessControl".Global.P[2];   // rising edge
   "AutoProcessControl".Global.P[2] := #_w5;
   IF #_w6 THEN "AutoProcessControl".Global.ALL_EmptyPallet := FALSE; END_IF;
   #tBool := "AlwaysTRUE" AND NOT "iH-shaftLoadingDetection1" AND NOT "iH-shaftLoadingDetection2" AND NOT "iH-shaftLoadingDetection3" AND NOT "iH-shaftLoadingDetection4" AND NOT "iH-shaftLiftingPalletDischarge" AND NOT "iH-shaftPalletEmptyCheck4" AND NOT "iH-shaftTakeGateDetection";
   #tBool := "AlwaysTRUE" AND #tBool AND NOT "iJ-magnetLiftingPalletDischargeDetection" AND NOT "J-mganePalletEmptyCheck4" AND NOT "iJ-magnetLoadingDetection4" AND NOT "J-mganePalletEmptyCheck3" AND NOT "iJ-magnetLoadingDetection3" AND NOT "J-mganePalletEmptyCheck2" AND NOT "iJ-magnetLoadingDetection2" AND NOT "J-mganePalletEmptyCheck1" AND NOT "iJ-magnetLoadingDetection1" AND NOT "iJ-magnetTakeGateDetection";
   "PalletRelease"."Time"[0].TON(IN := "AlwaysTRUE" AND #tBool AND NOT "iL-UnloadingTransplantingPalletInPlaceDetection" AND NOT "L-UnloadinPalletEmptyCheck3" AND NOT "iL-UnloadingDetection3" AND NOT "L-UnloadinPalletEmptyCheck2" AND NOT "iL-UnloadingDetection2" AND NOT "L-UnloadinPalletEmptyCheck1" AND NOT "iL-UnloadingDetection1" AND NOT "L-UnloadinTakeGateDetection",
                           PT := T#2S);
   "AutoProcessControl".Global.ALL_BeltPalletEmptyFinish := "PalletRelease"."Time"[0].Q;
END_REGION

REGION Network 31
   RUNG wire#powerrail
      Contact( "AlwaysTRUE" )
      { S7_Templates := "SrcType := Word" } EQ_Contact(in1 := %DB1067.DBW100, in2 := 0)
      wire#w1
      Move(in := 1, out1 => "ST10_PM".Status[1])
   END_RUNG
   RUNG wire#w1
      Not()
      Move(in := 2, out1 => "ST10_PM".Status[1])
   END_RUNG
   // the same network as SCL:
   #_w1 := "AlwaysTRUE" AND (%DB1067.DBW100 = 0);
   IF #_w1 THEN "ST10_PM".Status[1] := 1; END_IF;
   IF NOT #_w1 THEN "ST10_PM".Status[1] := 2; END_IF;
END_REGION

REGION Network 33
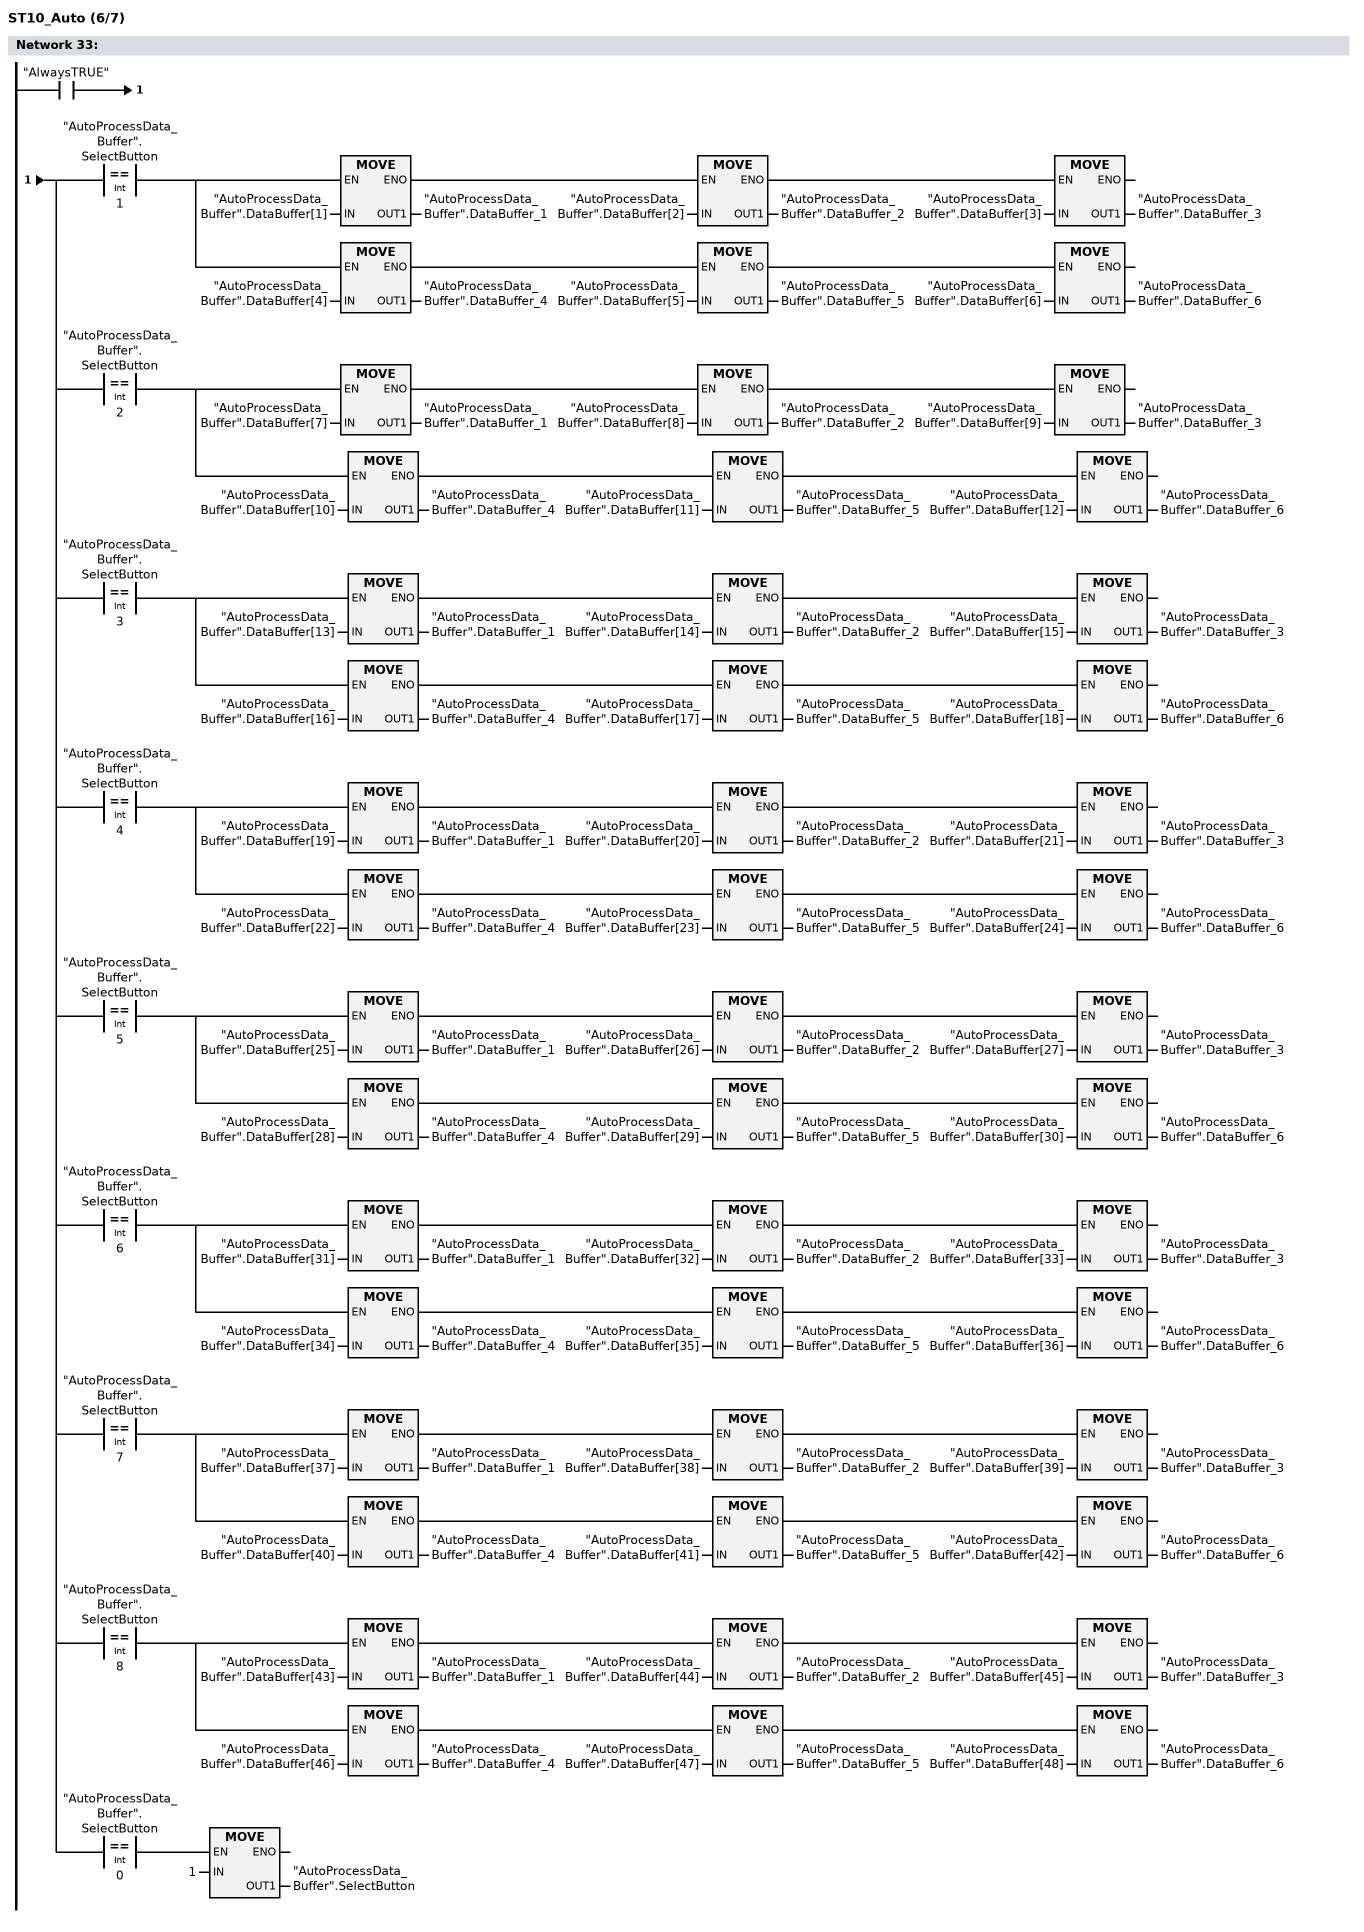
   RUNG wire#powerrail
      Contact( "AlwaysTRUE" )
      wire#w1
      { S7_Templates := "SrcType := Int" } EQ_Contact(in1 := "AutoProcessData_Buffer".SelectButton, in2 := 1)
      wire#w2
      Move(in := "AutoProcessData_Buffer".DataBuffer[1], out1 => "AutoProcessData_Buffer".DataBuffer_1)
      Move(in := "AutoProcessData_Buffer".DataBuffer[2], out1 => "AutoProcessData_Buffer".DataBuffer_2)
      Move(in := "AutoProcessData_Buffer".DataBuffer[3], out1 => "AutoProcessData_Buffer".DataBuffer_3)
   END_RUNG
   RUNG wire#w2
      Move(in := "AutoProcessData_Buffer".DataBuffer[4], out1 => "AutoProcessData_Buffer".DataBuffer_4)
      Move(in := "AutoProcessData_Buffer".DataBuffer[5], out1 => "AutoProcessData_Buffer".DataBuffer_5)
      Move(in := "AutoProcessData_Buffer".DataBuffer[6], out1 => "AutoProcessData_Buffer".DataBuffer_6)
   END_RUNG
   RUNG wire#w1
      { S7_Templates := "SrcType := Int" } EQ_Contact(in1 := "AutoProcessData_Buffer".SelectButton, in2 := 2)
      wire#w3
      Move(in := "AutoProcessData_Buffer".DataBuffer[7], out1 => "AutoProcessData_Buffer".DataBuffer_1)
      Move(in := "AutoProcessData_Buffer".DataBuffer[8], out1 => "AutoProcessData_Buffer".DataBuffer_2)
      Move(in := "AutoProcessData_Buffer".DataBuffer[9], out1 => "AutoProcessData_Buffer".DataBuffer_3)
   END_RUNG
   RUNG wire#w3
      Move(in := "AutoProcessData_Buffer".DataBuffer[10], out1 => "AutoProcessData_Buffer".DataBuffer_4)
      Move(in := "AutoProcessData_Buffer".DataBuffer[11], out1 => "AutoProcessData_Buffer".DataBuffer_5)
      Move(in := "AutoProcessData_Buffer".DataBuffer[12], out1 => "AutoProcessData_Buffer".DataBuffer_6)
   END_RUNG
   RUNG wire#w1
      { S7_Templates := "SrcType := Int" } EQ_Contact(in1 := "AutoProcessData_Buffer".SelectButton, in2 := 3)
      wire#w4
      Move(in := "AutoProcessData_Buffer".DataBuffer[13], out1 => "AutoProcessData_Buffer".DataBuffer_1)
      Move(in := "AutoProcessData_Buffer".DataBuffer[14], out1 => "AutoProcessData_Buffer".DataBuffer_2)
      Move(in := "AutoProcessData_Buffer".DataBuffer[15], out1 => "AutoProcessData_Buffer".DataBuffer_3)
   END_RUNG
   RUNG wire#w4
      Move(in := "AutoProcessData_Buffer".DataBuffer[16], out1 => "AutoProcessData_Buffer".DataBuffer_4)
      Move(in := "AutoProcessData_Buffer".DataBuffer[17], out1 => "AutoProcessData_Buffer".DataBuffer_5)
      Move(in := "AutoProcessData_Buffer".DataBuffer[18], out1 => "AutoProcessData_Buffer".DataBuffer_6)
   END_RUNG
   RUNG wire#w1
      { S7_Templates := "SrcType := Int" } EQ_Contact(in1 := "AutoProcessData_Buffer".SelectButton, in2 := 4)
      wire#w5
      Move(in := "AutoProcessData_Buffer".DataBuffer[19], out1 => "AutoProcessData_Buffer".DataBuffer_1)
      Move(in := "AutoProcessData_Buffer".DataBuffer[20], out1 => "AutoProcessData_Buffer".DataBuffer_2)
      Move(in := "AutoProcessData_Buffer".DataBuffer[21], out1 => "AutoProcessData_Buffer".DataBuffer_3)
   END_RUNG
   RUNG wire#w5
      Move(in := "AutoProcessData_Buffer".DataBuffer[22], out1 => "AutoProcessData_Buffer".DataBuffer_4)
      Move(in := "AutoProcessData_Buffer".DataBuffer[23], out1 => "AutoProcessData_Buffer".DataBuffer_5)
      Move(in := "AutoProcessData_Buffer".DataBuffer[24], out1 => "AutoProcessData_Buffer".DataBuffer_6)
   END_RUNG
   RUNG wire#w1
      { S7_Templates := "SrcType := Int" } EQ_Contact(in1 := "AutoProcessData_Buffer".SelectButton, in2 := 5)
      wire#w6
      Move(in := "AutoProcessData_Buffer".DataBuffer[25], out1 => "AutoProcessData_Buffer".DataBuffer_1)
      Move(in := "AutoProcessData_Buffer".DataBuffer[26], out1 => "AutoProcessData_Buffer".DataBuffer_2)
      Move(in := "AutoProcessData_Buffer".DataBuffer[27], out1 => "AutoProcessData_Buffer".DataBuffer_3)
   END_RUNG
   RUNG wire#w6
      Move(in := "AutoProcessData_Buffer".DataBuffer[28], out1 => "AutoProcessData_Buffer".DataBuffer_4)
      Move(in := "AutoProcessData_Buffer".DataBuffer[29], out1 => "AutoProcessData_Buffer".DataBuffer_5)
      Move(in := "AutoProcessData_Buffer".DataBuffer[30], out1 => "AutoProcessData_Buffer".DataBuffer_6)
   END_RUNG
   RUNG wire#w1
      { S7_Templates := "SrcType := Int" } EQ_Contact(in1 := "AutoProcessData_Buffer".SelectButton, in2 := 6)
      wire#w7
      Move(in := "AutoProcessData_Buffer".DataBuffer[31], out1 => "AutoProcessData_Buffer".DataBuffer_1)
      Move(in := "AutoProcessData_Buffer".DataBuffer[32], out1 => "AutoProcessData_Buffer".DataBuffer_2)
      Move(in := "AutoProcessData_Buffer".DataBuffer[33], out1 => "AutoProcessData_Buffer".DataBuffer_3)
   END_RUNG
   RUNG wire#w7
      Move(in := "AutoProcessData_Buffer".DataBuffer[34], out1 => "AutoProcessData_Buffer".DataBuffer_4)
      Move(in := "AutoProcessData_Buffer".DataBuffer[35], out1 => "AutoProcessData_Buffer".DataBuffer_5)
      Move(in := "AutoProcessData_Buffer".DataBuffer[36], out1 => "AutoProcessData_Buffer".DataBuffer_6)
   END_RUNG
   RUNG wire#w1
      { S7_Templates := "SrcType := Int" } EQ_Contact(in1 := "AutoProcessData_Buffer".SelectButton, in2 := 7)
      wire#w8
      Move(in := "AutoProcessData_Buffer".DataBuffer[37], out1 => "AutoProcessData_Buffer".DataBuffer_1)
      Move(in := "AutoProcessData_Buffer".DataBuffer[38], out1 => "AutoProcessData_Buffer".DataBuffer_2)
      Move(in := "AutoProcessData_Buffer".DataBuffer[39], out1 => "AutoProcessData_Buffer".DataBuffer_3)
   END_RUNG
   RUNG wire#w8
      Move(in := "AutoProcessData_Buffer".DataBuffer[40], out1 => "AutoProcessData_Buffer".DataBuffer_4)
      Move(in := "AutoProcessData_Buffer".DataBuffer[41], out1 => "AutoProcessData_Buffer".DataBuffer_5)
      Move(in := "AutoProcessData_Buffer".DataBuffer[42], out1 => "AutoProcessData_Buffer".DataBuffer_6)
   END_RUNG
   RUNG wire#w1
      { S7_Templates := "SrcType := Int" } EQ_Contact(in1 := "AutoProcessData_Buffer".SelectButton, in2 := 8)
      wire#w9
      Move(in := "AutoProcessData_Buffer".DataBuffer[43], out1 => "AutoProcessData_Buffer".DataBuffer_1)
      Move(in := "AutoProcessData_Buffer".DataBuffer[44], out1 => "AutoProcessData_Buffer".DataBuffer_2)
      Move(in := "AutoProcessData_Buffer".DataBuffer[45], out1 => "AutoProcessData_Buffer".DataBuffer_3)
   END_RUNG
   RUNG wire#w9
      Move(in := "AutoProcessData_Buffer".DataBuffer[46], out1 => "AutoProcessData_Buffer".DataBuffer_4)
      Move(in := "AutoProcessData_Buffer".DataBuffer[47], out1 => "AutoProcessData_Buffer".DataBuffer_5)
      Move(in := "AutoProcessData_Buffer".DataBuffer[48], out1 => "AutoProcessData_Buffer".DataBuffer_6)
   END_RUNG
   RUNG wire#w1
      { S7_Templates := "SrcType := Int" } EQ_Contact(in1 := "AutoProcessData_Buffer".SelectButton, in2 := 0)
      Move(in := 1, out1 => "AutoProcessData_Buffer".SelectButton)
   END_RUNG
   // the same network as SCL:
   IF "AlwaysTRUE" AND ("AutoProcessData_Buffer".SelectButton = 1) THEN
       "AutoProcessData_Buffer".DataBuffer_1 := "AutoProcessData_Buffer".DataBuffer[1];
       "AutoProcessData_Buffer".DataBuffer_2 := "AutoProcessData_Buffer".DataBuffer[2];
       "AutoProcessData_Buffer".DataBuffer_3 := "AutoProcessData_Buffer".DataBuffer[3];
       "AutoProcessData_Buffer".DataBuffer_4 := "AutoProcessData_Buffer".DataBuffer[4];
       "AutoProcessData_Buffer".DataBuffer_5 := "AutoProcessData_Buffer".DataBuffer[5];
       "AutoProcessData_Buffer".DataBuffer_6 := "AutoProcessData_Buffer".DataBuffer[6];
   END_IF;
   IF "AlwaysTRUE" AND ("AutoProcessData_Buffer".SelectButton = 2) THEN
       "AutoProcessData_Buffer".DataBuffer_1 := "AutoProcessData_Buffer".DataBuffer[7];
       "AutoProcessData_Buffer".DataBuffer_2 := "AutoProcessData_Buffer".DataBuffer[8];
       "AutoProcessData_Buffer".DataBuffer_3 := "AutoProcessData_Buffer".DataBuffer[9];
       "AutoProcessData_Buffer".DataBuffer_4 := "AutoProcessData_Buffer".DataBuffer[10];
       "AutoProcessData_Buffer".DataBuffer_5 := "AutoProcessData_Buffer".DataBuffer[11];
       "AutoProcessData_Buffer".DataBuffer_6 := "AutoProcessData_Buffer".DataBuffer[12];
   END_IF;
   IF "AlwaysTRUE" AND ("AutoProcessData_Buffer".SelectButton = 3) THEN
       "AutoProcessData_Buffer".DataBuffer_1 := "AutoProcessData_Buffer".DataBuffer[13];
       "AutoProcessData_Buffer".DataBuffer_2 := "AutoProcessData_Buffer".DataBuffer[14];
       "AutoProcessData_Buffer".DataBuffer_3 := "AutoProcessData_Buffer".DataBuffer[15];
       "AutoProcessData_Buffer".DataBuffer_4 := "AutoProcessData_Buffer".DataBuffer[16];
       "AutoProcessData_Buffer".DataBuffer_5 := "AutoProcessData_Buffer".DataBuffer[17];
       "AutoProcessData_Buffer".DataBuffer_6 := "AutoProcessData_Buffer".DataBuffer[18];
   END_IF;
   IF "AlwaysTRUE" AND ("AutoProcessData_Buffer".SelectButton = 4) THEN
       "AutoProcessData_Buffer".DataBuffer_1 := "AutoProcessData_Buffer".DataBuffer[19];
       "AutoProcessData_Buffer".DataBuffer_2 := "AutoProcessData_Buffer".DataBuffer[20];
       "AutoProcessData_Buffer".DataBuffer_3 := "AutoProcessData_Buffer".DataBuffer[21];
       "AutoProcessData_Buffer".DataBuffer_4 := "AutoProcessData_Buffer".DataBuffer[22];
       "AutoProcessData_Buffer".DataBuffer_5 := "AutoProcessData_Buffer".DataBuffer[23];
       "AutoProcessData_Buffer".DataBuffer_6 := "AutoProcessData_Buffer".DataBuffer[24];
   END_IF;
   IF "AlwaysTRUE" AND ("AutoProcessData_Buffer".SelectButton = 5) THEN
       "AutoProcessData_Buffer".DataBuffer_1 := "AutoProcessData_Buffer".DataBuffer[25];
       "AutoProcessData_Buffer".DataBuffer_2 := "AutoProcessData_Buffer".DataBuffer[26];
       "AutoProcessData_Buffer".DataBuffer_3 := "AutoProcessData_Buffer".DataBuffer[27];
       "AutoProcessData_Buffer".DataBuffer_4 := "AutoProcessData_Buffer".DataBuffer[28];
       "AutoProcessData_Buffer".DataBuffer_5 := "AutoProcessData_Buffer".DataBuffer[29];
       "AutoProcessData_Buffer".DataBuffer_6 := "AutoProcessData_Buffer".DataBuffer[30];
   END_IF;
   IF "AlwaysTRUE" AND ("AutoProcessData_Buffer".SelectButton = 6) THEN
       "AutoProcessData_Buffer".DataBuffer_1 := "AutoProcessData_Buffer".DataBuffer[31];
       "AutoProcessData_Buffer".DataBuffer_2 := "AutoProcessData_Buffer".DataBuffer[32];
       "AutoProcessData_Buffer".DataBuffer_3 := "AutoProcessData_Buffer".DataBuffer[33];
       "AutoProcessData_Buffer".DataBuffer_4 := "AutoProcessData_Buffer".DataBuffer[34];
       "AutoProcessData_Buffer".DataBuffer_5 := "AutoProcessData_Buffer".DataBuffer[35];
       "AutoProcessData_Buffer".DataBuffer_6 := "AutoProcessData_Buffer".DataBuffer[36];
   END_IF;
   IF "AlwaysTRUE" AND ("AutoProcessData_Buffer".SelectButton = 7) THEN
       "AutoProcessData_Buffer".DataBuffer_1 := "AutoProcessData_Buffer".DataBuffer[37];
       "AutoProcessData_Buffer".DataBuffer_2 := "AutoProcessData_Buffer".DataBuffer[38];
       "AutoProcessData_Buffer".DataBuffer_3 := "AutoProcessData_Buffer".DataBuffer[39];
       "AutoProcessData_Buffer".DataBuffer_4 := "AutoProcessData_Buffer".DataBuffer[40];
       "AutoProcessData_Buffer".DataBuffer_5 := "AutoProcessData_Buffer".DataBuffer[41];
       "AutoProcessData_Buffer".DataBuffer_6 := "AutoProcessData_Buffer".DataBuffer[42];
   END_IF;
   IF "AlwaysTRUE" AND ("AutoProcessData_Buffer".SelectButton = 8) THEN
       "AutoProcessData_Buffer".DataBuffer_1 := "AutoProcessData_Buffer".DataBuffer[43];
       "AutoProcessData_Buffer".DataBuffer_2 := "AutoProcessData_Buffer".DataBuffer[44];
       "AutoProcessData_Buffer".DataBuffer_3 := "AutoProcessData_Buffer".DataBuffer[45];
       "AutoProcessData_Buffer".DataBuffer_4 := "AutoProcessData_Buffer".DataBuffer[46];
       "AutoProcessData_Buffer".DataBuffer_5 := "AutoProcessData_Buffer".DataBuffer[47];
       "AutoProcessData_Buffer".DataBuffer_6 := "AutoProcessData_Buffer".DataBuffer[48];
   END_IF;
   IF "AlwaysTRUE" AND ("AutoProcessData_Buffer".SelectButton = 0) THEN
       "AutoProcessData_Buffer".SelectButton := 1;
   END_IF;
END_REGION

REGION Network 34
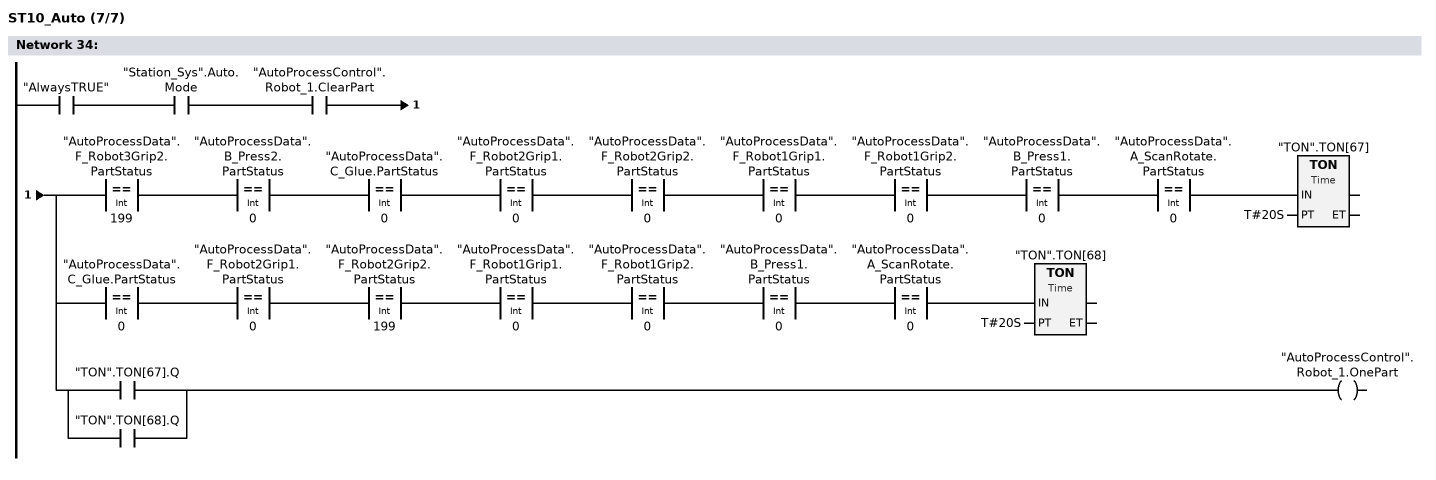
   RUNG wire#powerrail
      Contact( "AlwaysTRUE" )
      Contact( "Station_Sys".Auto.Mode )
      Contact( "AutoProcessControl".Robot_1.ClearPart )
      wire#w1
      { S7_Templates := "SrcType := Int" } EQ_Contact(in1 := "AutoProcessData".F_Robot3Grip2.PartStatus, in2 := 199)
      { S7_Templates := "SrcType := Int" } EQ_Contact(in1 := "AutoProcessData".B_Press2.PartStatus, in2 := 0)
      { S7_Templates := "SrcType := Int" } EQ_Contact(in1 := "AutoProcessData".C_Glue.PartStatus, in2 := 0)
      { S7_Templates := "SrcType := Int" } EQ_Contact(in1 := "AutoProcessData".F_Robot2Grip1.PartStatus, in2 := 0)
      { S7_Templates := "SrcType := Int" } EQ_Contact(in1 := "AutoProcessData".F_Robot2Grip2.PartStatus, in2 := 0)
      { S7_Templates := "SrcType := Int" } EQ_Contact(in1 := "AutoProcessData".F_Robot1Grip1.PartStatus, in2 := 0)
      { S7_Templates := "SrcType := Int" } EQ_Contact(in1 := "AutoProcessData".F_Robot1Grip2.PartStatus, in2 := 0)
      { S7_Templates := "SrcType := Int" } EQ_Contact(in1 := "AutoProcessData".B_Press1.PartStatus, in2 := 0)
      { S7_Templates := "SrcType := Int" } EQ_Contact(in1 := "AutoProcessData".A_ScanRotate.PartStatus, in2 := 0)
      { S7_Templates := "time_type := Time" } "TON".TON[67].TON(pt := T#20S, et =>)
   END_RUNG
   RUNG wire#w1
      { S7_Templates := "SrcType := Int" } EQ_Contact(in1 := "AutoProcessData".C_Glue.PartStatus, in2 := 0)
      { S7_Templates := "SrcType := Int" } EQ_Contact(in1 := "AutoProcessData".F_Robot2Grip1.PartStatus, in2 := 0)
      { S7_Templates := "SrcType := Int" } EQ_Contact(in1 := "AutoProcessData".F_Robot2Grip2.PartStatus, in2 := 199)
      { S7_Templates := "SrcType := Int" } EQ_Contact(in1 := "AutoProcessData".F_Robot1Grip1.PartStatus, in2 := 0)
      { S7_Templates := "SrcType := Int" } EQ_Contact(in1 := "AutoProcessData".F_Robot1Grip2.PartStatus, in2 := 0)
      { S7_Templates := "SrcType := Int" } EQ_Contact(in1 := "AutoProcessData".B_Press1.PartStatus, in2 := 0)
      { S7_Templates := "SrcType := Int" } EQ_Contact(in1 := "AutoProcessData".A_ScanRotate.PartStatus, in2 := 0)
      { S7_Templates := "time_type := Time" } "TON".TON[68].TON(pt := T#20S, et =>)
   END_RUNG
   RUNG wire#w1
      Contact( "TON".TON[67].Q )
      wire#w2
      Coil( "AutoProcessControl".Robot_1.OnePart )
   END_RUNG
   RUNG wire#w1
      Contact( "TON".TON[68].Q )
   END_RUNG wire#w2
   // the same network as SCL:
   #_w1 := "AlwaysTRUE" AND "Station_Sys".Auto.Mode AND "AutoProcessControl".Robot_1.ClearPart;
   "TON".TON[67].TON(IN := #_w1 AND ("AutoProcessData".F_Robot3Grip2.PartStatus = 199) AND ("AutoProcessData".B_Press2.PartStatus = 0) AND ("AutoProcessData".C_Glue.PartStatus = 0) AND ("AutoProcessData".F_Robot2Grip1.PartStatus = 0) AND ("AutoProcessData".F_Robot2Grip2.PartStatus = 0) AND ("AutoProcessData".F_Robot1Grip1.PartStatus = 0) AND ("AutoProcessData".F_Robot1Grip2.PartStatus = 0) AND ("AutoProcessData".B_Press1.PartStatus = 0) AND ("AutoProcessData".A_ScanRotate.PartStatus = 0),
                     PT := T#20S);
   "TON".TON[68].TON(IN := #_w1 AND ("AutoProcessData".C_Glue.PartStatus = 0) AND ("AutoProcessData".F_Robot2Grip1.PartStatus = 0) AND ("AutoProcessData".F_Robot2Grip2.PartStatus = 199) AND ("AutoProcessData".F_Robot1Grip1.PartStatus = 0) AND ("AutoProcessData".F_Robot1Grip2.PartStatus = 0) AND ("AutoProcessData".B_Press1.PartStatus = 0) AND ("AutoProcessData".A_ScanRotate.PartStatus = 0),
                     PT := T#20S);
   "AutoProcessControl".Robot_1.OnePart := #_w1 AND ("TON".TON[67].Q OR "TON".TON[68].Q);
END_REGION

REGION Network 36 (SCL)
   IF "Station_Sys".Initial.Running THEN
       FOR #FlankWord := 1 TO 99 DO
           "GeneralDebug".Debug[#FlankWord] := false;
       END_FOR;
   END_IF;
END_REGION
END_FUNCTION

FUNCTION "ChangeOverProcess" : Void   // FC1000, LAD
{ S7_Optimized_Access := 'TRUE' }
// stored: AutoNumber false, SetENOAutomatically false
   VAR_TEMP
      tBool : Bool;
   END_VAR
   VAR_TEMP   // added for the SCL form of the ladder/FBD networks
      _w1 : Bool;
      _w2 : Bool;
      _w3 : Bool;
      _w4 : Bool;
      _w5 : Bool;
      _w6 : Bool;
      _w7 : Bool;
      _w8 : Bool;
   END_VAR
BEGIN

REGION Network 1: HMI ChangeOver Confirm
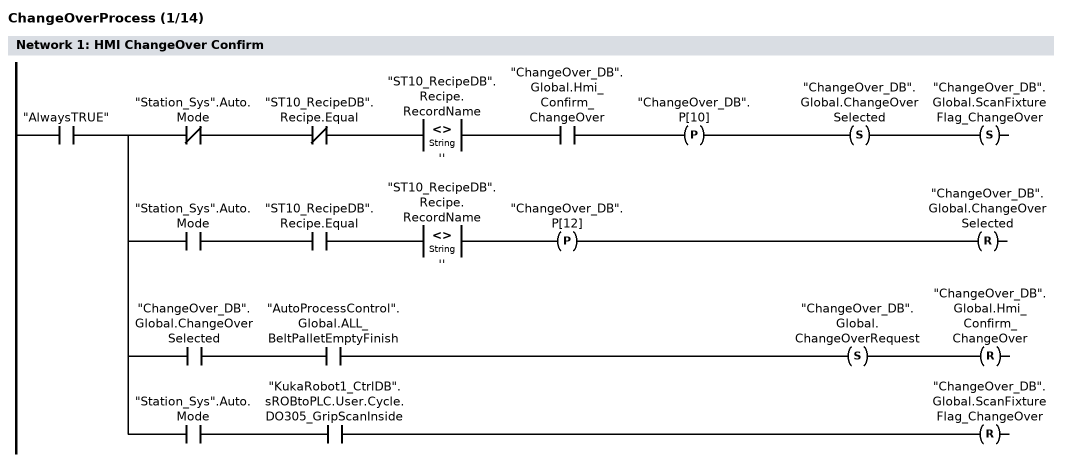
   RUNG wire#powerrail
      Contact( "AlwaysTRUE" )
      wire#w1
      I_Contact( "Station_Sys".Auto.Mode )
      I_Contact( "ST10_RecipeDB".Recipe.Equal )
      { S7_Templates := "SrcType := String" } NE_Contact(in1 := "ST10_RecipeDB".Recipe.RecordName, in2 := '')
      Contact( "ChangeOver_DB".Global.Hmi_Confirm_ChangeOver )
      P_Trig( "ChangeOver_DB".P[10] )
      S_Coil( "ChangeOver_DB".Global.ChangeOverSelected )
      S_Coil( "ChangeOver_DB".Global.ScanFixtureFlag_ChangeOver )
   END_RUNG
   RUNG wire#w1
      Contact( "Station_Sys".Auto.Mode )
      Contact( "ST10_RecipeDB".Recipe.Equal )
      { S7_Templates := "SrcType := String" } NE_Contact(in1 := "ST10_RecipeDB".Recipe.RecordName, in2 := '')
      P_Trig( "ChangeOver_DB".P[12] )
      R_Coil( "ChangeOver_DB".Global.ChangeOverSelected )
   END_RUNG
   RUNG wire#w1
      Contact( "ChangeOver_DB".Global.ChangeOverSelected )
      Contact( "AutoProcessControl".Global.ALL_BeltPalletEmptyFinish )
      S_Coil( "ChangeOver_DB".Global.ChangeOverRequest )
      R_Coil( "ChangeOver_DB".Global.Hmi_Confirm_ChangeOver )
   END_RUNG
   RUNG wire#w1
      Contact( "Station_Sys".Auto.Mode )
      Contact( "KukaRobot1_CtrlDB".sROBtoPLC.User.Cycle.DO305_GripScanInside )
      R_Coil( "ChangeOver_DB".Global.ScanFixtureFlag_ChangeOver )
   END_RUNG
   // the same network as SCL:
   #_w1 := "AlwaysTRUE" AND NOT "Station_Sys".Auto.Mode AND NOT "ST10_RecipeDB".Recipe.Equal AND ("ST10_RecipeDB".Recipe.RecordName <> '') AND "ChangeOver_DB".Global.Hmi_Confirm_ChangeOver;
   #_w2 := #_w1 AND NOT "ChangeOver_DB".P[10];   // rising edge
   "ChangeOver_DB".P[10] := #_w1;
   IF #_w2 THEN
       "ChangeOver_DB".Global.ChangeOverSelected := TRUE;
       "ChangeOver_DB".Global.ScanFixtureFlag_ChangeOver := TRUE;
   END_IF;
   #_w3 := "AlwaysTRUE" AND "Station_Sys".Auto.Mode AND "ST10_RecipeDB".Recipe.Equal AND ("ST10_RecipeDB".Recipe.RecordName <> '');
   #_w4 := #_w3 AND NOT "ChangeOver_DB".P[12];   // rising edge
   "ChangeOver_DB".P[12] := #_w3;
   IF #_w4 THEN "ChangeOver_DB".Global.ChangeOverSelected := FALSE; END_IF;
   IF "AlwaysTRUE" AND "ChangeOver_DB".Global.ChangeOverSelected AND "AutoProcessControl".Global.ALL_BeltPalletEmptyFinish THEN
       "ChangeOver_DB".Global.ChangeOverRequest := TRUE;
       "ChangeOver_DB".Global.Hmi_Confirm_ChangeOver := FALSE;
   END_IF;
   IF "AlwaysTRUE" AND "Station_Sys".Auto.Mode AND "KukaRobot1_CtrlDB".sROBtoPLC.User.Cycle.DO305_GripScanInside THEN
       "ChangeOver_DB".Global.ScanFixtureFlag_ChangeOver := FALSE;
   END_IF;
END_REGION

REGION Network 2: ChangeOverFinish Reset
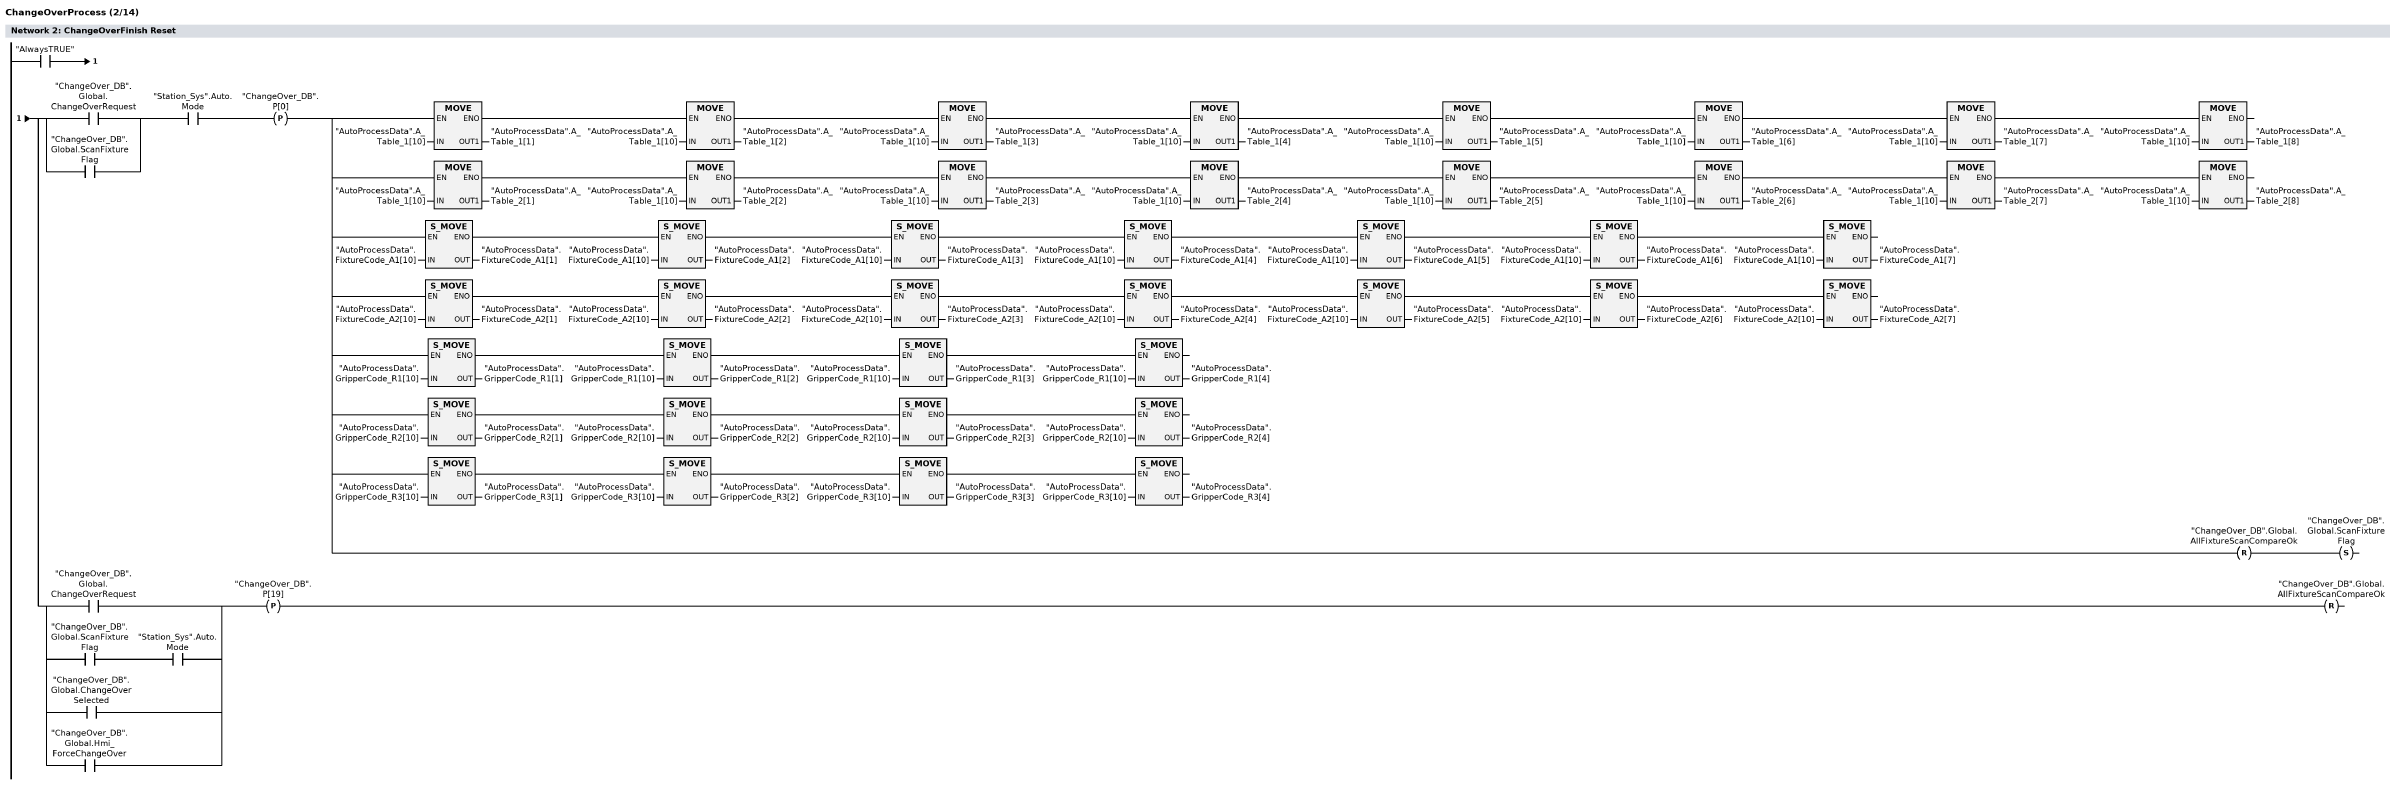
   RUNG wire#powerrail
      Contact( "AlwaysTRUE" )
      wire#w1
      Contact( "ChangeOver_DB".Global.ChangeOverRequest )
      wire#w2
      Contact( "Station_Sys".Auto.Mode )
      P_Trig( "ChangeOver_DB".P[0] )
      wire#w3
      Move(in := "AutoProcessData".A_Table_1[10], out1 => "AutoProcessData".A_Table_1[1])
      Move(in := "AutoProcessData".A_Table_1[10], out1 => "AutoProcessData".A_Table_1[2])
      Move(in := "AutoProcessData".A_Table_1[10], out1 => "AutoProcessData".A_Table_1[3])
      Move(in := "AutoProcessData".A_Table_1[10], out1 => "AutoProcessData".A_Table_1[4])
      Move(in := "AutoProcessData".A_Table_1[10], out1 => "AutoProcessData".A_Table_1[5])
      Move(in := "AutoProcessData".A_Table_1[10], out1 => "AutoProcessData".A_Table_1[6])
      Move(in := "AutoProcessData".A_Table_1[10], out1 => "AutoProcessData".A_Table_1[7])
      Move(in := "AutoProcessData".A_Table_1[10], out1 => "AutoProcessData".A_Table_1[8])
   END_RUNG
   RUNG wire#w1
      Contact( "ChangeOver_DB".Global.ScanFixtureFlag )
   END_RUNG wire#w2
   RUNG wire#w3
      Move(in := "AutoProcessData".A_Table_1[10], out1 => "AutoProcessData".A_Table_2[1])
      Move(in := "AutoProcessData".A_Table_1[10], out1 => "AutoProcessData".A_Table_2[2])
      Move(in := "AutoProcessData".A_Table_1[10], out1 => "AutoProcessData".A_Table_2[3])
      Move(in := "AutoProcessData".A_Table_1[10], out1 => "AutoProcessData".A_Table_2[4])
      Move(in := "AutoProcessData".A_Table_1[10], out1 => "AutoProcessData".A_Table_2[5])
      Move(in := "AutoProcessData".A_Table_1[10], out1 => "AutoProcessData".A_Table_2[6])
      Move(in := "AutoProcessData".A_Table_1[10], out1 => "AutoProcessData".A_Table_2[7])
      Move(in := "AutoProcessData".A_Table_1[10], out1 => "AutoProcessData".A_Table_2[8])
   END_RUNG
   RUNG wire#w3
      S_Move(in := "AutoProcessData".FixtureCode_A1[10], out => "AutoProcessData".FixtureCode_A1[1])
      S_Move(in := "AutoProcessData".FixtureCode_A1[10], out => "AutoProcessData".FixtureCode_A1[2])
      S_Move(in := "AutoProcessData".FixtureCode_A1[10], out => "AutoProcessData".FixtureCode_A1[3])
      S_Move(in := "AutoProcessData".FixtureCode_A1[10], out => "AutoProcessData".FixtureCode_A1[4])
      S_Move(in := "AutoProcessData".FixtureCode_A1[10], out => "AutoProcessData".FixtureCode_A1[5])
      S_Move(in := "AutoProcessData".FixtureCode_A1[10], out => "AutoProcessData".FixtureCode_A1[6])
      S_Move(in := "AutoProcessData".FixtureCode_A1[10], out => "AutoProcessData".FixtureCode_A1[7])
   END_RUNG
   RUNG wire#w3
      S_Move(in := "AutoProcessData".FixtureCode_A2[10], out => "AutoProcessData".FixtureCode_A2[1])
      S_Move(in := "AutoProcessData".FixtureCode_A2[10], out => "AutoProcessData".FixtureCode_A2[2])
      S_Move(in := "AutoProcessData".FixtureCode_A2[10], out => "AutoProcessData".FixtureCode_A2[3])
      S_Move(in := "AutoProcessData".FixtureCode_A2[10], out => "AutoProcessData".FixtureCode_A2[4])
      S_Move(in := "AutoProcessData".FixtureCode_A2[10], out => "AutoProcessData".FixtureCode_A2[5])
      S_Move(in := "AutoProcessData".FixtureCode_A2[10], out => "AutoProcessData".FixtureCode_A2[6])
      S_Move(in := "AutoProcessData".FixtureCode_A2[10], out => "AutoProcessData".FixtureCode_A2[7])
   END_RUNG
   RUNG wire#w3
      S_Move(in := "AutoProcessData".GripperCode_R1[10], out => "AutoProcessData".GripperCode_R1[1])
      S_Move(in := "AutoProcessData".GripperCode_R1[10], out => "AutoProcessData".GripperCode_R1[2])
      S_Move(in := "AutoProcessData".GripperCode_R1[10], out => "AutoProcessData".GripperCode_R1[3])
      S_Move(in := "AutoProcessData".GripperCode_R1[10], out => "AutoProcessData".GripperCode_R1[4])
   END_RUNG
   RUNG wire#w3
      S_Move(in := "AutoProcessData".GripperCode_R2[10], out => "AutoProcessData".GripperCode_R2[1])
      S_Move(in := "AutoProcessData".GripperCode_R2[10], out => "AutoProcessData".GripperCode_R2[2])
      S_Move(in := "AutoProcessData".GripperCode_R2[10], out => "AutoProcessData".GripperCode_R2[3])
      S_Move(in := "AutoProcessData".GripperCode_R2[10], out => "AutoProcessData".GripperCode_R2[4])
   END_RUNG
   RUNG wire#w3
      S_Move(in := "AutoProcessData".GripperCode_R3[10], out => "AutoProcessData".GripperCode_R3[1])
      S_Move(in := "AutoProcessData".GripperCode_R3[10], out => "AutoProcessData".GripperCode_R3[2])
      S_Move(in := "AutoProcessData".GripperCode_R3[10], out => "AutoProcessData".GripperCode_R3[3])
      S_Move(in := "AutoProcessData".GripperCode_R3[10], out => "AutoProcessData".GripperCode_R3[4])
   END_RUNG
   RUNG wire#w3
      R_Coil( "ChangeOver_DB".Global.AllFixtureScanCompareOk )
      S_Coil( "ChangeOver_DB".Global.ScanFixtureFlag )
   END_RUNG
   RUNG wire#w1
      Contact( "ChangeOver_DB".Global.ChangeOverRequest )
      wire#w4
      P_Trig( "ChangeOver_DB".P[19] )
      R_Coil( "ChangeOver_DB".Global.AllFixtureScanCompareOk )
   END_RUNG
   RUNG wire#w1
      Contact( "ChangeOver_DB".Global.ScanFixtureFlag )
      Contact( "Station_Sys".Auto.Mode )
   END_RUNG wire#w4
   RUNG wire#w1
      Contact( "ChangeOver_DB".Global.ChangeOverSelected )
   END_RUNG wire#w4
   RUNG wire#w1
      Contact( "ChangeOver_DB".Global.Hmi_ForceChangeOver )
   END_RUNG wire#w4
   // the same network as SCL:
   #_w1 := "AlwaysTRUE" AND ("ChangeOver_DB".Global.ChangeOverRequest OR "ChangeOver_DB".Global.ScanFixtureFlag) AND "Station_Sys".Auto.Mode;
   #_w2 := #_w1 AND NOT "ChangeOver_DB".P[0];   // rising edge
   "ChangeOver_DB".P[0] := #_w1;
   IF #_w2 THEN
       "AutoProcessData".A_Table_1[1] := "AutoProcessData".A_Table_1[10];
       "AutoProcessData".A_Table_1[2] := "AutoProcessData".A_Table_1[10];
       "AutoProcessData".A_Table_1[3] := "AutoProcessData".A_Table_1[10];
       "AutoProcessData".A_Table_1[4] := "AutoProcessData".A_Table_1[10];
       "AutoProcessData".A_Table_1[5] := "AutoProcessData".A_Table_1[10];
       "AutoProcessData".A_Table_1[6] := "AutoProcessData".A_Table_1[10];
       "AutoProcessData".A_Table_1[7] := "AutoProcessData".A_Table_1[10];
       "AutoProcessData".A_Table_1[8] := "AutoProcessData".A_Table_1[10];
       "AutoProcessData".A_Table_2[1] := "AutoProcessData".A_Table_1[10];
       "AutoProcessData".A_Table_2[2] := "AutoProcessData".A_Table_1[10];
       "AutoProcessData".A_Table_2[3] := "AutoProcessData".A_Table_1[10];
       "AutoProcessData".A_Table_2[4] := "AutoProcessData".A_Table_1[10];
       "AutoProcessData".A_Table_2[5] := "AutoProcessData".A_Table_1[10];
       "AutoProcessData".A_Table_2[6] := "AutoProcessData".A_Table_1[10];
       "AutoProcessData".A_Table_2[7] := "AutoProcessData".A_Table_1[10];
       "AutoProcessData".A_Table_2[8] := "AutoProcessData".A_Table_1[10];
       "AutoProcessData".FixtureCode_A1[1] := "AutoProcessData".FixtureCode_A1[10];
       "AutoProcessData".FixtureCode_A1[2] := "AutoProcessData".FixtureCode_A1[10];
       "AutoProcessData".FixtureCode_A1[3] := "AutoProcessData".FixtureCode_A1[10];
       "AutoProcessData".FixtureCode_A1[4] := "AutoProcessData".FixtureCode_A1[10];
       "AutoProcessData".FixtureCode_A1[5] := "AutoProcessData".FixtureCode_A1[10];
       "AutoProcessData".FixtureCode_A1[6] := "AutoProcessData".FixtureCode_A1[10];
       "AutoProcessData".FixtureCode_A1[7] := "AutoProcessData".FixtureCode_A1[10];
       "AutoProcessData".FixtureCode_A2[1] := "AutoProcessData".FixtureCode_A2[10];
       "AutoProcessData".FixtureCode_A2[2] := "AutoProcessData".FixtureCode_A2[10];
       "AutoProcessData".FixtureCode_A2[3] := "AutoProcessData".FixtureCode_A2[10];
       "AutoProcessData".FixtureCode_A2[4] := "AutoProcessData".FixtureCode_A2[10];
       "AutoProcessData".FixtureCode_A2[5] := "AutoProcessData".FixtureCode_A2[10];
       "AutoProcessData".FixtureCode_A2[6] := "AutoProcessData".FixtureCode_A2[10];
       "AutoProcessData".FixtureCode_A2[7] := "AutoProcessData".FixtureCode_A2[10];
       "AutoProcessData".GripperCode_R1[1] := "AutoProcessData".GripperCode_R1[10];
       "AutoProcessData".GripperCode_R1[2] := "AutoProcessData".GripperCode_R1[10];
       "AutoProcessData".GripperCode_R1[3] := "AutoProcessData".GripperCode_R1[10];
       "AutoProcessData".GripperCode_R1[4] := "AutoProcessData".GripperCode_R1[10];
       "AutoProcessData".GripperCode_R2[1] := "AutoProcessData".GripperCode_R2[10];
       "AutoProcessData".GripperCode_R2[2] := "AutoProcessData".GripperCode_R2[10];
       "AutoProcessData".GripperCode_R2[3] := "AutoProcessData".GripperCode_R2[10];
       "AutoProcessData".GripperCode_R2[4] := "AutoProcessData".GripperCode_R2[10];
       "AutoProcessData".GripperCode_R3[1] := "AutoProcessData".GripperCode_R3[10];
       "AutoProcessData".GripperCode_R3[2] := "AutoProcessData".GripperCode_R3[10];
       "AutoProcessData".GripperCode_R3[3] := "AutoProcessData".GripperCode_R3[10];
       "AutoProcessData".GripperCode_R3[4] := "AutoProcessData".GripperCode_R3[10];
       "ChangeOver_DB".Global.AllFixtureScanCompareOk := FALSE;
       "ChangeOver_DB".Global.ScanFixtureFlag := TRUE;
   END_IF;
   #_w3 := "AlwaysTRUE" AND ("ChangeOver_DB".Global.ChangeOverRequest OR ("ChangeOver_DB".Global.ScanFixtureFlag AND "Station_Sys".Auto.Mode) OR "ChangeOver_DB".Global.ChangeOverSelected OR "ChangeOver_DB".Global.Hmi_ForceChangeOver);
   #_w4 := #_w3 AND NOT "ChangeOver_DB".P[19];   // rising edge
   "ChangeOver_DB".P[19] := #_w3;
   IF #_w4 THEN "ChangeOver_DB".Global.AllFixtureScanCompareOk := FALSE; END_IF;
END_REGION

REGION Network 3: ManualModeFlag
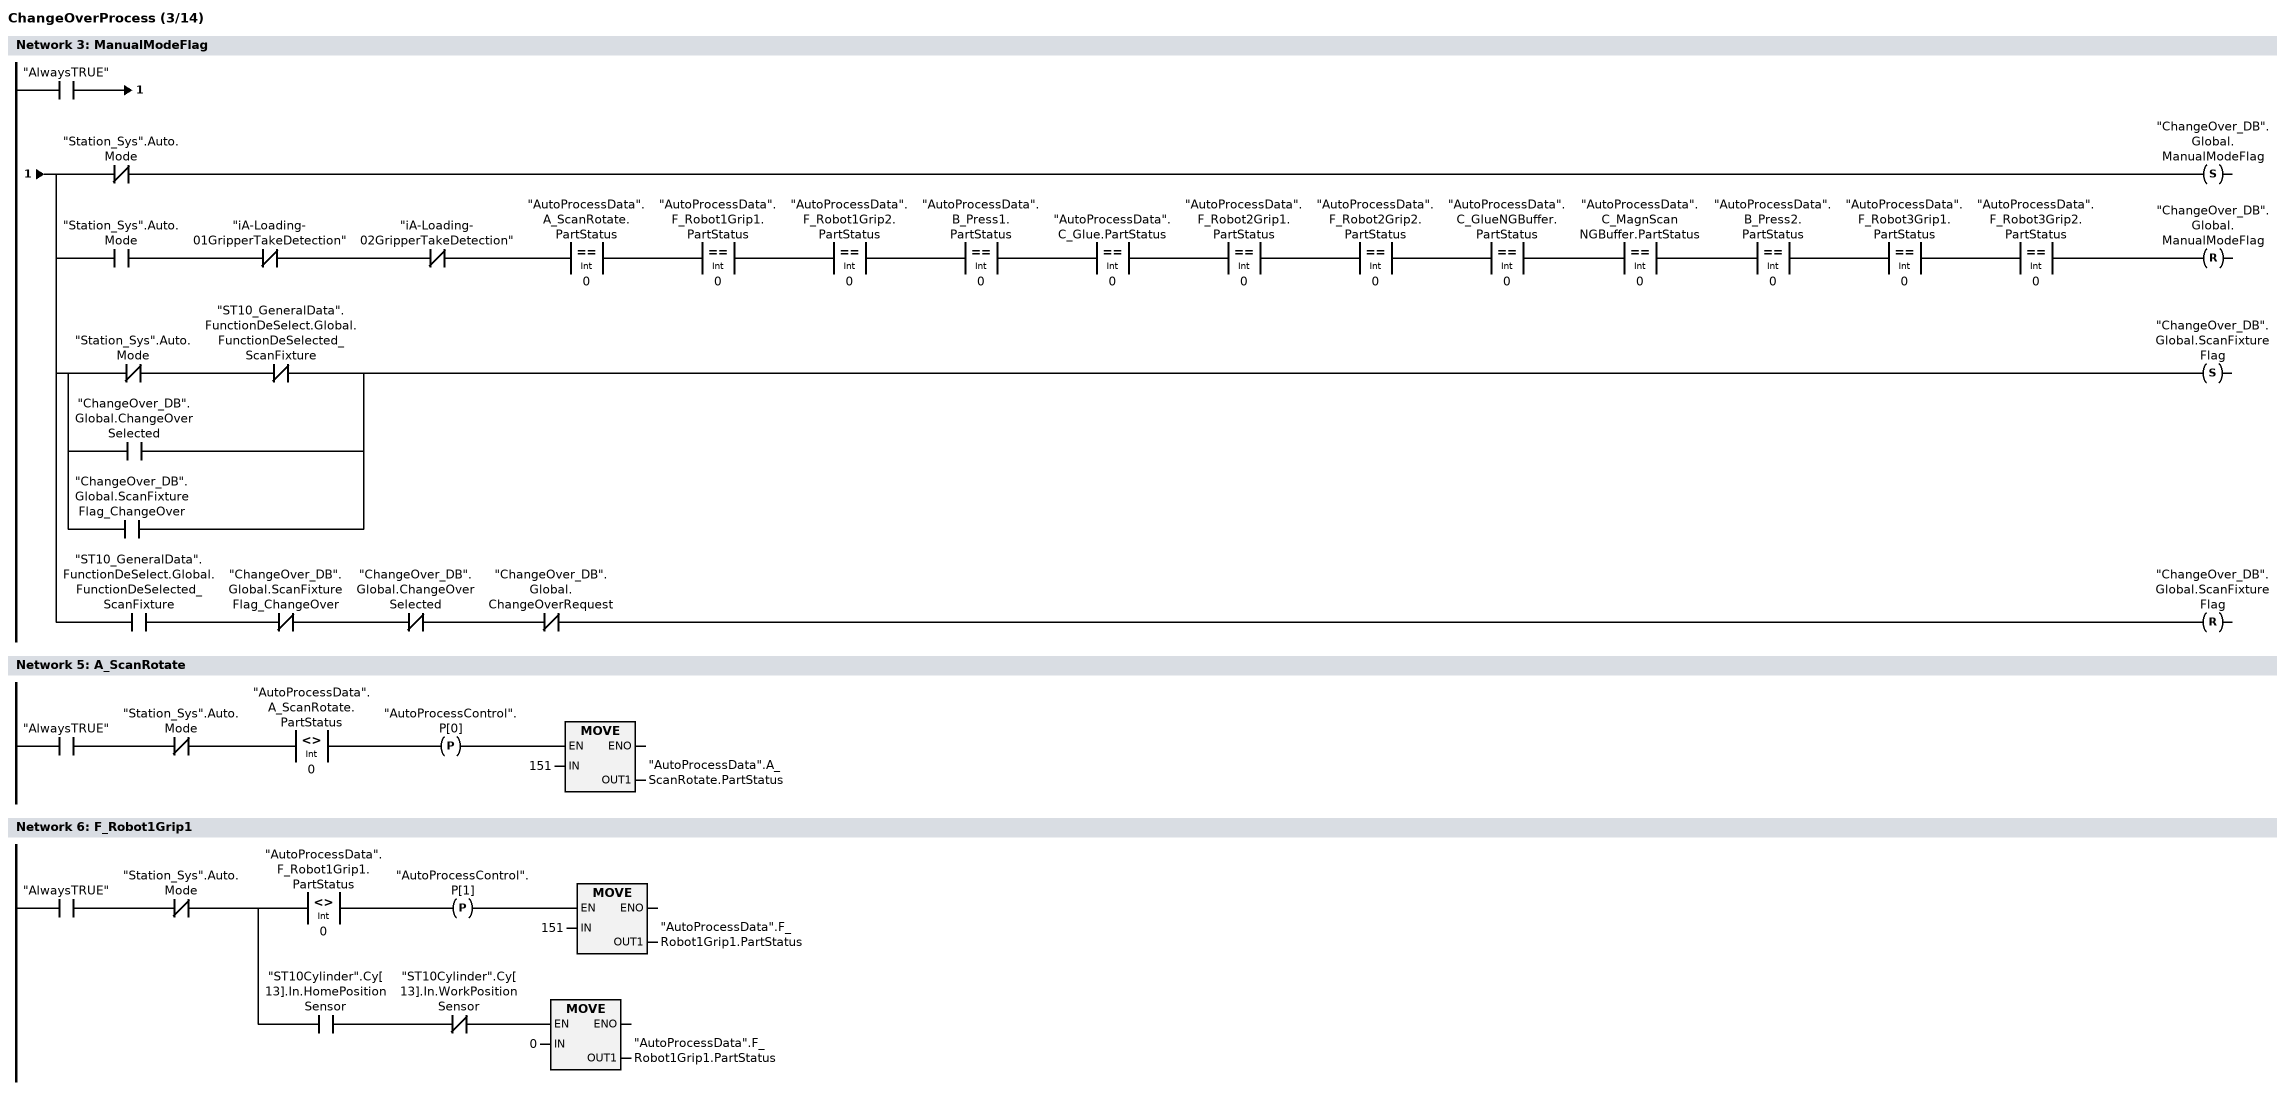
   RUNG wire#powerrail
      Contact( "AlwaysTRUE" )
      wire#w1
      I_Contact( "Station_Sys".Auto.Mode )
      S_Coil( "ChangeOver_DB".Global.ManualModeFlag )
   END_RUNG
   RUNG wire#w1
      Contact( "Station_Sys".Auto.Mode )
      I_Contact( "iA-Loading-01GripperTakeDetection" )
      I_Contact( "iA-Loading-02GripperTakeDetection" )
      { S7_Templates := "SrcType := Int" } EQ_Contact(in1 := "AutoProcessData".A_ScanRotate.PartStatus, in2 := 0)
      { S7_Templates := "SrcType := Int" } EQ_Contact(in1 := "AutoProcessData".F_Robot1Grip1.PartStatus, in2 := 0)
      { S7_Templates := "SrcType := Int" } EQ_Contact(in1 := "AutoProcessData".F_Robot1Grip2.PartStatus, in2 := 0)
      { S7_Templates := "SrcType := Int" } EQ_Contact(in1 := "AutoProcessData".B_Press1.PartStatus, in2 := 0)
      { S7_Templates := "SrcType := Int" } EQ_Contact(in1 := "AutoProcessData".C_Glue.PartStatus, in2 := 0)
      { S7_Templates := "SrcType := Int" } EQ_Contact(in1 := "AutoProcessData".F_Robot2Grip1.PartStatus, in2 := 0)
      { S7_Templates := "SrcType := Int" } EQ_Contact(in1 := "AutoProcessData".F_Robot2Grip2.PartStatus, in2 := 0)
      { S7_Templates := "SrcType := Int" } EQ_Contact(in1 := "AutoProcessData".C_GlueNGBuffer.PartStatus, in2 := 0)
      { S7_Templates := "SrcType := Int" } EQ_Contact(in1 := "AutoProcessData".C_MagnScanNGBuffer.PartStatus, in2 := 0)
      { S7_Templates := "SrcType := Int" } EQ_Contact(in1 := "AutoProcessData".B_Press2.PartStatus, in2 := 0)
      { S7_Templates := "SrcType := Int" } EQ_Contact(in1 := "AutoProcessData".F_Robot3Grip1.PartStatus, in2 := 0)
      { S7_Templates := "SrcType := Int" } EQ_Contact(in1 := "AutoProcessData".F_Robot3Grip2.PartStatus, in2 := 0)
      R_Coil( "ChangeOver_DB".Global.ManualModeFlag )
   END_RUNG
   RUNG wire#w1
      I_Contact( "Station_Sys".Auto.Mode )
      I_Contact( "ST10_GeneralData".FunctionDeSelect.Global.FunctionDeSelected_ScanFixture )
      wire#w2
      S_Coil( "ChangeOver_DB".Global.ScanFixtureFlag )
   END_RUNG
   RUNG wire#w1
      Contact( "ChangeOver_DB".Global.ChangeOverSelected )
   END_RUNG wire#w2
   RUNG wire#w1
      Contact( "ChangeOver_DB".Global.ScanFixtureFlag_ChangeOver )
   END_RUNG wire#w2
   RUNG wire#w1
      Contact( "ST10_GeneralData".FunctionDeSelect.Global.FunctionDeSelected_ScanFixture )
      I_Contact( "ChangeOver_DB".Global.ScanFixtureFlag_ChangeOver )
      I_Contact( "ChangeOver_DB".Global.ChangeOverSelected )
      I_Contact( "ChangeOver_DB".Global.ChangeOverRequest )
      R_Coil( "ChangeOver_DB".Global.ScanFixtureFlag )
   END_RUNG
   // the same network as SCL:
   IF "AlwaysTRUE" AND NOT "Station_Sys".Auto.Mode THEN
       "ChangeOver_DB".Global.ManualModeFlag := TRUE;
   END_IF;
   IF "AlwaysTRUE" AND "Station_Sys".Auto.Mode AND NOT "iA-Loading-01GripperTakeDetection" AND NOT "iA-Loading-02GripperTakeDetection" AND ("AutoProcessData".A_ScanRotate.PartStatus = 0) AND ("AutoProcessData".F_Robot1Grip1.PartStatus = 0) AND ("AutoProcessData".F_Robot1Grip2.PartStatus = 0) AND ("AutoProcessData".B_Press1.PartStatus = 0) AND ("AutoProcessData".C_Glue.PartStatus = 0) AND ("AutoProcessData".F_Robot2Grip1.PartStatus = 0) AND ("AutoProcessData".F_Robot2Grip2.PartStatus = 0) AND ("AutoProcessData".C_GlueNGBuffer.PartStatus = 0) AND ("AutoProcessData".C_MagnScanNGBuffer.PartStatus = 0) AND ("AutoProcessData".B_Press2.PartStatus = 0) AND ("AutoProcessData".F_Robot3Grip1.PartStatus = 0) AND ("AutoProcessData".F_Robot3Grip2.PartStatus = 0) THEN
       "ChangeOver_DB".Global.ManualModeFlag := FALSE;
   END_IF;
   IF "AlwaysTRUE" AND ((NOT "Station_Sys".Auto.Mode AND NOT "ST10_GeneralData".FunctionDeSelect.Global.FunctionDeSelected_ScanFixture) OR "ChangeOver_DB".Global.ChangeOverSelected OR "ChangeOver_DB".Global.ScanFixtureFlag_ChangeOver) THEN
       "ChangeOver_DB".Global.ScanFixtureFlag := TRUE;
   END_IF;
   IF "AlwaysTRUE" AND "ST10_GeneralData".FunctionDeSelect.Global.FunctionDeSelected_ScanFixture AND NOT "ChangeOver_DB".Global.ScanFixtureFlag_ChangeOver AND NOT "ChangeOver_DB".Global.ChangeOverSelected AND NOT "ChangeOver_DB".Global.ChangeOverRequest THEN
       "ChangeOver_DB".Global.ScanFixtureFlag := FALSE;
   END_IF;
END_REGION

REGION Network 4: ----------------------------- Manu Mode,All the part NG -------------------------------------------------------
END_REGION

REGION Network 5: A_ScanRotate
   RUNG wire#powerrail
      Contact( "AlwaysTRUE" )
      I_Contact( "Station_Sys".Auto.Mode )
      { S7_Templates := "SrcType := Int" } NE_Contact(in1 := "AutoProcessData".A_ScanRotate.PartStatus, in2 := 0)
      P_Trig( "AutoProcessControl".P[0] )
      Move(in := 151, out1 => "AutoProcessData".A_ScanRotate.PartStatus)
   END_RUNG
   // the same network as SCL:
   #_w1 := "AlwaysTRUE" AND NOT "Station_Sys".Auto.Mode AND ("AutoProcessData".A_ScanRotate.PartStatus <> 0);
   #_w2 := #_w1 AND NOT "AutoProcessControl".P[0];   // rising edge
   "AutoProcessControl".P[0] := #_w1;
   IF #_w2 THEN "AutoProcessData".A_ScanRotate.PartStatus := 151; END_IF;
END_REGION

REGION Network 6: F_Robot1Grip1
   RUNG wire#powerrail
      Contact( "AlwaysTRUE" )
      I_Contact( "Station_Sys".Auto.Mode )
      wire#w1
      { S7_Templates := "SrcType := Int" } NE_Contact(in1 := "AutoProcessData".F_Robot1Grip1.PartStatus, in2 := 0)
      P_Trig( "AutoProcessControl".P[1] )
      Move(in := 151, out1 => "AutoProcessData".F_Robot1Grip1.PartStatus)
   END_RUNG
   RUNG wire#w1
      Contact( "ST10Cylinder".Cy[13].In.HomePositionSensor )
      I_Contact( "ST10Cylinder".Cy[13].In.WorkPositionSensor )
      Move(in := 0, out1 => "AutoProcessData".F_Robot1Grip1.PartStatus)
   END_RUNG
   // the same network as SCL:
   #_w1 := "AlwaysTRUE" AND NOT "Station_Sys".Auto.Mode;
   #_w2 := #_w1 AND ("AutoProcessData".F_Robot1Grip1.PartStatus <> 0);
   #_w3 := #_w2 AND NOT "AutoProcessControl".P[1];   // rising edge
   "AutoProcessControl".P[1] := #_w2;
   IF #_w3 THEN "AutoProcessData".F_Robot1Grip1.PartStatus := 151; END_IF;
   IF #_w1 AND "ST10Cylinder".Cy[13].In.HomePositionSensor AND NOT "ST10Cylinder".Cy[13].In.WorkPositionSensor THEN
       "AutoProcessData".F_Robot1Grip1.PartStatus := 0;
   END_IF;
END_REGION

